# B&R Automation Studio project TD52 (part 147)

### Global_DI.typ
```iecst
TYPE
	Perm_DI_struct : 	STRUCT
		tCtr_ChCW_LT : _tGeACtrPara; (*Para controller charge temperature cooler*) (*OldName:REG9; Cycle:5;*)
		bCtr_ChCW_LT : BOOL; (*PARA [11872]: visibility charge temperature controller*) (*OldName:bPlantCtr9,reg0_visible; Cycle:5;*)
		tCtr_ChCW_HT : _tGeACtrPara; (*Para controller charge temperature cooler*) (*OldName:REG9; Cycle:5;*)
		bCtr_ChCW_HT : BOOL; (*PARA [11872]: visibility charge temperature controller*) (*OldName:bPlantCtr9,reg0_visible; Cycle:5;*)
		tCtr_ChCW_HT_LP : _tGeACtrPara; (*Para controller charge temperature cooler*) (*OldName:REG9; Cycle:5;*)
		bCtr_ChCW_HT_LP : BOOL; (*PARA [11872]: visibility charge temperature controller*) (*OldName:bPlantCtr9,reg0_visible; Cycle:5;*)
		tCtr_ChCW_HT_HP : _tGeACtrPara; (*Para controller charge temperature cooler*) (*OldName:REG9; Cycle:5;*)
		bCtr_ChCW_HT_HP : BOOL; (*PARA [11872]: visibility charge temperature controller*) (*OldName:bPlantCtr9,reg0_visible; Cycle:5;*)
		tCtr_ChCW_LT_LP : _tGeACtrPara; (*Para controller charge temperature cooler*) (*OldName:REG9; Cycle:5;*)
		bCtr_ChCW_LT_LP : BOOL; (*PARA [11872]: visibility charge temperature controller*) (*OldName:bPlantCtr9,reg0_visible; Cycle:5;*)
		tCtr_ChCW_LT_HP : _tGeACtrPara; (*Para controller charge temperature cooler*) (*OldName:REG9; Cycle:5;*)
		bCtr_ChCW_LT_HP : BOOL; (*PARA [11872]: visibility charge temperature controller*) (*OldName:bPlantCtr9,reg0_visible; Cycle:5;*)
		tCtr_ECW : _tGeACtrPara; (*Para controller  engine cooling water temperature cooler*) (*OldName:REG9; Cycle:5;*)
		bCtr_ECW : BOOL; (*PARA [11872]: visibility  engine cooling water temperature controller*) (*OldName:bPlantCtr9,reg0_visible; Cycle:5;*)
		tCtr_OCW : _tGeACtrPara; (*Para controller  oil cooling water temperature cooler*) (*OldName:REG9; Cycle:5;*)
		bCtr_OCW : BOOL; (*PARA [11872]: visibility  oil cooling water temperature controller*) (*OldName:bPlantCtr9,reg0_visible; Cycle:5;*)
		bT_ChCW_Re_LT : BOOL; (*visu aktiv Temp Ladekühlwasser Rücklauf NT*)
		bPr_ChCW_Re_LT : BOOL; (*visu aktiv Druck Ladekühlwasser Rücklauf NT*)
		bT_ChCW_Su_LT : BOOL; (*visu aktiv Temp Ladekühlwasser Vorlauf NT*)
		bPr_ChCW_Su_LT : BOOL; (*visu aktiv Druck Ladekühlwasser Vorlauf NT*)
		bT_ChCW_Re_HT : BOOL; (*visu aktiv Temp Ladekühlwasser Rücklauf NT*)
		bPr_ChCW_Re_HT : BOOL; (*visu aktiv Druck Ladekühlwasser Rücklauf HT*)
		bT_ChCW_Su_HT : BOOL; (*visu aktiv Temp Ladekühlwasser Vorlauf HT*)
		bPr_ChCW_Su_HT : BOOL; (*visu aktiv Druck Ladekühlwasser Vorlauf HT*)
		bT_ChCW_Re_HT_LP : BOOL; (*visu aktiv Temp Ladekühlwasser Rücklauf HT ND*)
		bPr_ChCW_Re_HT_LP : BOOL; (*visu aktiv Druck Ladekühlwasser Rücklauf HT ND*)
		bT_ChCW_Re_HT_HP : BOOL; (*visu aktiv Temp Ladekühlwasser Rücklauf HT HD*)
		bPr_ChCW_Re_HT_HP : BOOL; (*visu aktiv Druck Ladekühlwasser Rücklauf HT HD*)
		bT_ChCW_Su_HT_LP : BOOL; (*visu aktiv Temp Ladekühlwasser Vorlauf HT ND*)
		bPr_ChCW_Su_HT_LP : BOOL; (*visu aktiv Druck Ladekühlwasser Vorlauf HT ND*)
		bT_ChCW_Su_HT_HP : BOOL; (*visu aktiv Temp Ladekühlwasser Vorlauf HT HD*)
		bPr_ChCW_Su_HT_HP : BOOL; (*visu aktiv Druck Ladekühlwasser Vorlauf HT HD*)
		bT_ChCW_Re_LT_LP : BOOL; (*visu aktiv Temp Ladekühlwasser Rücklauf NT ND*)
		bPr_ChCW_Re_LT_LP : BOOL; (*visu aktiv Druck Ladekühlwasser Rücklauf NT ND*)
		bT_ChCW_Re_LT_HP : BOOL; (*visu aktiv Temp Ladekühlwasser Rücklauf NT HD*)
		bPr_ChCW_Re_LT_HP : BOOL; (*visu aktiv Druck Ladekühlwasser Rücklauf NT HD*)
		bT_ChCW_Su_LT_LP : BOOL; (*visu aktiv Temp Ladekühlwasser Vorlauf NT ND*)
		bPr_ChCW_Su_LT_LP : BOOL; (*visu aktiv Druck Ladekühlwasser Vorlauf NT ND*)
		bT_ChCW_Su_LT_HP : BOOL; (*visu aktiv Temp Ladekühlwasser Vorlauf NT HD*)
		bPr_ChCW_Su_LT_HP : BOOL; (*visu aktiv Druck Ladekühlwasser Vorlauf NT HD*)
		bT_OCW_Re : BOOL; (*visu aktiv Temp Ölkühlwasser Rücklauf*)
		bPr_OCW_Re : BOOL; (*visu aktiv Druck Ölkühlwasser Rücklauf*)
		bT_OCW_Su : BOOL; (*visu aktiv Temp Ölkühlwasser Vorlauf*)
		bPr_OCW_Su : BOOL; (*visu aktiv Druck Ölkühlwasser Vorlauf*)
		bT_ECW_Re : BOOL; (*visu aktiv Temp Motorkühlwasser Rücklauf*)
		bPr_ECW_Re : BOOL; (*visu aktiv Druck Motorkühlwasser Rücklauf*)
		bT_ECW_Su : BOOL; (*visu aktiv Temp Motorkühlwasser Vorlauf*)
		bPr_ECW_Su : BOOL; (*visu aktiv Druck Motorkühlwasser Vorlauf*)
		bVol_ChCW_Re_LT : BOOL; (*visu aktiv Durchfluss Ladekühlwasser Rücklauf NT*)
		bVol_ChCW_Su_LT : BOOL; (*visu aktiv Durchfluss Ladekühlwasser Vorlauf NT*)
		bVol_ChCW_Re_HT : BOOL; (*visu aktiv Durchfluss Ladekühlwasser Rücklauf HT*)
		bVol_ChCW_Su_HT : BOOL; (*visu aktiv Durchfluss Ladekühlwasser Vorlauf HT*)
		bVol_ChCW_Re_HT_LP : BOOL; (*visu aktiv Durchfluss Ladekühlwasser Rücklauf HT ND*)
		bVol_ChCW_Su_HT_LP : BOOL; (*visu aktiv Durchfluss Ladekühlwasser Vorlauf HT ND*)
		bVol_ChCW_Re_HT_HP : BOOL; (*visu aktiv Durchfluss Ladekühlwasser Rücklauf HT HD*)
		bVol_ChCW_Su_HT_HP : BOOL; (*visu aktiv Durchfluss Ladekühlwasser Vorlauf HT HD*)
		bVol_ChCW_Re_LT_LP : BOOL; (*visu aktiv Durchfluss Ladekühlwasser Rücklauf NT ND*)
		bVol_ChCW_Su_LT_LP : BOOL; (*visu aktiv Durchfluss Ladekühlwasser Vorlauf NT ND*)
		bVol_ChCW_Re_LT_HP : BOOL; (*visu aktiv Durchfluss Ladekühlwasser Rücklauf NT HD*)
		bVol_ChCW_Su_LT_HP : BOOL; (*visu aktiv Durchfluss Ladekühlwasser Vorlauf NT HD*)
		bVol_ECW_Re : BOOL; (*visu aktiv Durchfluss Motorkühlwasser Rücklauf*)
		bVol_ECW_Su : BOOL; (*visu aktiv Durchfluss Motorkühlwasser Vorlauf*)
		bVol_OCW_Re : BOOL; (*visu aktiv Durchfluss Ölkühlwasser Rücklauf*)
		bVol_OCW_Su : BOOL; (*visu aktiv Durchfluss Ölkühlwasser Vorlauf*)
		bT_ChCW_LT_IC_Re : BOOL; (*visu aktiv Temp Ladekühlewasser NT Zwischenkreis Rücklauf*)
		bPr_ChCW_LT_IC_Re : BOOL; (*visu aktiv Druck Ladekühlewasser NT Zwischenkreis Rücklauf*)
		bT_ChCW_HT_IC_Re : BOOL; (*visu aktiv Temp Ladekühlewasser HT Zwischenkreis Rücklauf*)
		bPr_ChCW_HT_IC_Re : BOOL; (*visu aktiv Druck Ladekühlewasser HT Zwischenkreis Rücklauf*)
		bT_ChCW_LT_LP_IC_Re : BOOL; (*visu aktiv Temp Ladekühlewasser NT ND Zwischenkreis Rücklauf*)
		bPr_ChCW_LT_LP_IC_Re : BOOL; (*visu aktiv Druck Ladekühlewasser NT ND Zwischenkreis Rücklauf*)
		bT_ChCW_LT_HP_IC_Re : BOOL; (*visu aktiv Temp Ladekühlewasser NT HD Zwischenkreis Rücklauf*)
		bPr_ChCW_LT_HP_IC_Re : BOOL; (*visu aktiv Druck Ladekühlewasser NT HD Zwischenkreis Rücklauf*)
		bT_ChCW_HT_LP_IC_Re : BOOL; (*visu aktiv Temp Ladekühlewasser HT ND Zwischenkreis Rücklauf*)
		bPr_ChCW_HT_LP_IC_Re : BOOL; (*visu aktiv Druck Ladekühlewasser HT ND Zwischenkreis Rücklauf*)
		bT_ChCW_HT_HP_IC_Re : BOOL; (*visu aktiv Temp Ladekühlewasser HT HD Zwischenkreis Rücklauf*)
		bPr_ChCW_HT_HP_IC_Re : BOOL; (*visu aktiv Druck Ladekühlewasser HT HD Zwischenkreis Rücklauf*)
		bT_ECW_IC_Re : BOOL; (*visu aktiv Temp Motorkühlwasser Zwischenkreis Rücklauf*)
		bPr_ECW_IC_Re : BOOL; (*visu aktiv Druck Motorkühlwasser Zwischenkreis Rücklauf*)
		bT_OCW_IC_Re : BOOL; (*visu aktiv Temp Ölkühlwasser Zwischenkreis Rücklauf*)
		bPr_OCW_IC_Re : BOOL; (*visu aktiv Druck Ölkühlwasser Zwischenkreis Rücklauf*)
		bT_ChCW_LT_IC_Su : BOOL; (*visu aktiv Temp Ladekühlewasser NT Zwischenkreis Rücklauf*)
		bPr_ChCW_LT_IC_Su : BOOL; (*visu aktiv Druck Ladekühlewasser NT Zwischenkreis Rücklauf*)
		bT_ChCW_HT_IC_Su : BOOL; (*visu aktiv Temp Ladekühlewasser HT Zwischenkreis Rücklauf*)
		bPr_ChCW_HT_IC_Su : BOOL; (*visu aktiv Druck Ladekühlewasser HT Zwischenkreis Rücklauf*)
		bT_ChCW_LT_LP_IC_Su : BOOL; (*visu aktiv Temp Ladekühlewasser NT ND Zwischenkreis Rücklauf*)
		bPr_ChCW_LT_LP_IC_Su : BOOL; (*visu aktiv Druck Ladekühlewasser NT ND Zwischenkreis Rücklauf*)
		bT_ChCW_LT_HP_IC_Su : BOOL; (*visu aktiv Temp Ladekühlewasser NT HD Zwischenkreis Rücklauf*)
		bPr_ChCW_LT_HP_IC_Su : BOOL; (*visu aktiv Druck Ladekühlewasser NT HD Zwischenkreis Rücklauf*)
		bT_ChCW_HT_LP_IC_Su : BOOL; (*visu aktiv Temp Ladekühlewasser HT ND Zwischenkreis Rücklauf*)
		bPr_ChCW_HT_LP_IC_Su : BOOL; (*visu aktiv Druck Ladekühlewasser HT ND Zwischenkreis Rücklauf*)
		bT_ChCW_HT_HP_IC_Su : BOOL; (*visu aktiv Temp Ladekühlewasser HT HD Zwischenkreis Rücklauf*)
		bPr_ChCW_HT_HP_IC_Su : BOOL; (*visu aktiv Druck Ladekühlewasser HT HD Zwischenkreis Rücklauf*)
		bT_ECW_IC_Su : BOOL; (*visu aktiv Temp Motorkühlwasser Zwischenkreis Rücklauf*)
		bPr_ECW_IC_Su : BOOL; (*visu aktiv Druck Motorkühlwasser Zwischenkreis Rücklauf*)
		bT_OCW_IC_Su : BOOL; (*visu aktiv Temp Ölkühlwasser Zwischenkreis Rücklauf*)
		bPr_OCW_IC_Su : BOOL; (*visu aktiv Druck Ölkühlwasser Zwischenkreis Vorlauf*)
		bT_Cooler_ChCW_LT_Re_1 : BOOL; (*visu aktiv Temp Kühler Ladekühlwasser NT Rücklauf*)
		bT_Cooler_ChCW_LT_Re_2 : BOOL; (*visu aktiv Temp Kühler Ladekühlwasser NT Rücklauf*)
		bT_Cooler_ChCW_HT_Re_1 : BOOL; (*visu aktiv Temp Kühler Ladekühlwasser HT Rücklauf*)
		bT_Cooler_ChCW_HT_Re_2 : BOOL; (*visu aktiv Temp Kühler Ladekühlwasser HT Rücklauf*)
		bT_Cooler_ChCW_LT_LP_Re_1 : BOOL; (*visu aktiv Temp Kühler Ladekühlwasser NT ND Rücklauf*)
		bT_Cooler_ChCW_LT_LP_Re_2 : BOOL; (*visu aktiv Temp Kühler Ladekühlwasser NT ND Rücklauf*)
		bT_Cooler_ChCW_LT_HP_Re_1 : BOOL; (*visu aktiv Temp Kühler Ladekühlwasser NT HD Rücklauf*)
		bT_Cooler_ChCW_LT_HP_Re_2 : BOOL; (*visu aktiv Temp Kühler Ladekühlwasser NT HD Rücklauf*)
		bT_Cooler_ChCW_HT_LP_Re_1 : BOOL; (*visu aktiv Temp Kühler Ladekühlwasser HT ND Rücklauf*)
		bT_Cooler_ChCW_HT_LP_Re_2 : BOOL; (*visu aktiv Temp Kühler Ladekühlwasser HT ND Rücklauf*)
		bT_Cooler_ChCW_HT_HP_Re_1 : BOOL; (*visu aktiv Temp Kühler Ladekühlwasser HT HD Rücklauf*)
		bT_Cooler_ChCW_HT_HP_Re_2 : BOOL; (*visu aktiv Temp Kühler Ladekühlwasser HT HD Rücklauf*)
		bT_Cooler_ECW_Re_1 : BOOL; (*visu aktiv Temp Kühler Motorkühlwasser Rücklauf*)
		bT_Cooler_ECW_Re_2 : BOOL; (*visu aktiv Temp Kühler Motorkühlwasser Rücklauf*)
		bT_Cooler_OCW_Re_1 : BOOL; (*visu aktiv Temp Kühler Ölkühlwasser Rücklauf*)
		bT_Cooler_OCW_Re_2 : BOOL; (*visu aktiv Temp Kühler Ölkühlwasser Rücklauf*)
		bPr_Cooler_ChCW_LT_Re_1 : BOOL; (*visu aktiv Druck Kühler Ladekühlwasser NT Rücklauf*)
		bPr_Cooler_ChCW_LT_Re_2 : BOOL; (*visu aktiv Druck Kühler Ladekühlwasser NT Rücklauf*)
		bPr_Cooler_ChCW_HT_Re_1 : BOOL; (*visu aktiv Druck Kühler Ladekühlwasser HT Rücklauf*)
		bPr_Cooler_ChCW_HT_Re_2 : BOOL; (*visu aktiv Druck Kühler Ladekühlwasser HT Rücklauf*)
		bPr_Cooler_ChCW_LT_LP_Re_1 : BOOL; (*visu aktiv Druck Kühler Ladekühlwasser NT ND Rücklauf*)
		bPr_Cooler_ChCW_LT_LP_Re_2 : BOOL; (*visu aktiv Druck Kühler Ladekühlwasser NT ND Rücklauf*)
		bPr_Cooler_ChCW_LT_HP_Re_1 : BOOL; (*visu aktiv Druck Kühler Ladekühlwasser NT HD Rücklauf*)
		bPr_Cooler_ChCW_LT_HP_Re_2 : BOOL; (*visu aktiv Druck Kühler Ladekühlwasser NT HD Rücklauf*)
		bPr_Cooler_ChCW_HT_LP_Re_1 : BOOL; (*visu aktiv Druck Kühler Ladekühlwasser HT ND Rücklauf*)
		bPr_Cooler_ChCW_HT_LP_Re_2 : BOOL; (*visu aktiv Druck Kühler Ladekühlwasser HT ND Rücklauf*)
		bPr_Cooler_ChCW_HT_HP_Re_1 : BOOL; (*visu aktiv Druck Kühler Ladekühlwasser HT HD Rücklauf*)
		bPr_Cooler_ChCW_HT_HP_Re_2 : BOOL; (*visu aktiv Druck Kühler Ladekühlwasser HT HD Rücklauf*)
		bPr_Cooler_ECW_Re_1 : BOOL; (*visu aktiv Druck Kühler Motorkühlwasser Rücklauf*)
		bPr_Cooler_ECW_Re_2 : BOOL; (*visu aktiv Druck Kühler Motorkühlwasser Rücklauf*)
		bPr_Cooler_OCW_Re_1 : BOOL; (*visu aktiv Druck Kühler Ölkühlwasser Rücklauf*)
		bPr_Cooler_OCW_Re_2 : BOOL; (*visu aktiv Druck Kühler Ölkühlwasser Rücklauf*)
		bT_Cooler_ChCW_LT_Su_1 : BOOL; (*visu aktiv Temp Kühler Ladekühlwasser NT Vorlauf*)
		bT_Cooler_ChCW_LT_Su_2 : BOOL; (*visu aktiv Temp Kühler Ladekühlwasser NT Vorlauf*)
		bT_Cooler_ChCW_HT_Su_1 : BOOL; (*visu aktiv Temp Kühler Ladekühlwasser HT Vorlauf*)
		bT_Cooler_ChCW_HT_Su_2 : BOOL; (*visu aktiv Temp Kühler Ladekühlwasser HT Vorlauf*)
		bT_Cooler_ChCW_LT_LP_Su_1 : BOOL; (*visu aktiv Temp Kühler Ladekühlwasser NT ND Vorlauf*)
		bT_Cooler_ChCW_LT_LP_Su_2 : BOOL; (*visu aktiv Temp Kühler Ladekühlwasser NT ND Vorlauf*)
		bT_Cooler_ChCW_LT_HP_Su_1 : BOOL; (*visu aktiv Temp Kühler Ladekühlwasser NT HD Vorlauf*)
		bT_Cooler_ChCW_LT_HP_Su_2 : BOOL; (*visu aktiv Temp Kühler Ladekühlwasser NT HD Vorlauf*)
		bT_Cooler_ChCW_HT_LP_Su_1 : BOOL; (*visu aktiv Temp Kühler Ladekühlwasser HT ND Vorlauf*)
		bT_Cooler_ChCW_HT_LP_Su_2 : BOOL; (*visu aktiv Temp Kühler Ladekühlwasser HT ND Vorlauf*)
		bT_Cooler_ChCW_HT_HP_Su_1 : BOOL; (*visu aktiv Temp Kühler Ladekühlwasser HT HD Vorlauf*)
		bT_Cooler_ChCW_HT_HP_Su_2 : BOOL; (*visu aktiv Temp Kühler Ladekühlwasser HT HD Vorlauf*)
		bT_Cooler_ECW_Su_1 : BOOL; (*visu aktiv Temp Kühler Motorkühlwasser Vorlauf*)
		bT_Cooler_ECW_Su_2 : BOOL; (*visu aktiv Temp Kühler Motorkühlwasser Vorlauf*)
		bT_Cooler_OCW_Su_1 : BOOL; (*visu aktiv Temp Kühler Ölkühlwasser Vorlauf*)
		bT_Cooler_OCW_Su_2 : BOOL; (*visu aktiv Temp Kühler Ölkühlwasser Vorlauf*)
		bPr_Cooler_ChCW_LT_Su_1 : BOOL; (*visu aktiv Druck Kühler Ladekühlwasser NT Vorlauf*)
		bPr_Cooler_ChCW_LT_Su_2 : BOOL; (*visu aktiv Druck Kühler Ladekühlwasser NT Vorlauf*)
		bPr_Cooler_ChCW_HT_Su_1 : BOOL; (*visu aktiv Druck Kühler Ladekühlwasser HT Vorlauf*)
		bPr_Cooler_ChCW_HT_Su_2 : BOOL; (*visu aktiv Druck Kühler Ladekühlwasser HT Vorlauf*)
		bPr_Cooler_ChCW_LT_LP_Su_1 : BOOL; (*visu aktiv Druck Kühler Ladekühlwasser NT ND Vorlauf*)
		bPr_Cooler_ChCW_LT_LP_Su_2 : BOOL; (*visu aktiv Druck Kühler Ladekühlwasser NT ND Vorlauf*)
		bPr_Cooler_ChCW_LT_HP_Su_1 : BOOL; (*visu aktiv Druck Kühler Ladekühlwasser NT HD Vorlauf*)
		bPr_Cooler_ChCW_LT_HP_Su_2 : BOOL; (*visu aktiv Druck Kühler Ladekühlwasser NT HD Vorlauf*)
		bPr_Cooler_ChCW_HT_LP_Su_1 : BOOL; (*visu aktiv Druck Kühler Ladekühlwasser HT ND Vorlauf*)
		bPr_Cooler_ChCW_HT_LP_Su_2 : BOOL; (*visu aktiv Druck Kühler Ladekühlwasser HT ND Vorlauf*)
		bPr_Cooler_ChCW_HT_HP_Su_1 : BOOL; (*visu aktiv Druck Kühler Ladekühlwasser HT HD Vorlauf*)
		bPr_Cooler_ChCW_HT_HP_Su_2 : BOOL; (*visu aktiv Druck Kühler Ladekühlwasser HT HD Vorlauf*)
		bPr_Cooler_ECW_Su_1 : BOOL; (*visu aktiv Druck Kühler Motorkühlwasser Vorlauf*)
		bPr_Cooler_ECW_Su_2 : BOOL; (*visu aktiv Druck Kühler Motorkühlwasser Vorlauf*)
		bPr_Cooler_OCW_Su_1 : BOOL; (*visu aktiv Druck Kühler Ölkühlwasser Vorlauf*)
		bPr_Cooler_OCW_Su_2 : BOOL; (*visu aktiv Druck Kühler Ölkühlwasser Vorlauf*)
		bT_ChCW_LT_bCV : BOOL; (*visu aktiv Temp Ladekühlwasser NT vor Regelventil*)
		bT_ChCW_LT_LP_bCV : BOOL; (*visu aktiv Temp Ladekühlwasser NT ND vor Regelventil*)
		bT_ChCW_LT_HP_bCV : BOOL; (*visu aktiv Temp Ladekühlwasser NT HD vor Regelventil*)
		bT_ChCW_HT_bCV : BOOL; (*visu aktiv Temp Ladekühlwasser NT vor Regelventil*)
		bT_ChCW_HT_LP_bCV : BOOL; (*visu aktiv Temp Ladekühlwasser NT ND vor Regelventil*)
		bT_ChCW_HT_HP_bCV : BOOL; (*visu aktiv Temp Ladekühlwasser NT HD vor Regelventil*)
		bT_ECW_bCV : BOOL; (*visu aktiv Temp Motorkühlwasser vor Regelventil*)
		bT_OCW_bCV : BOOL; (*visu aktiv Temp Ölkühlwasser vor Regelventil*)
		bT_RW_HE_Re : BOOL; (*visu aktiv Temp Rohwasser Wärmetausche Rücklauf*)
		bT_RW_HE_Su : BOOL; (*visu aktiv Temp Rohwasser Wärmetausche Vorlauf*)
		bPr_RW_HE_Re : BOOL; (*visu aktiv Druck Rohwasser Wärmetausche Rücklauf*)
		bPr_RW_HE_Su : BOOL; (*visu aktiv Druck Rohwasser Wärmetausche Vorlauf*)
		bCtr_RW_CV : BOOL; (*visu aktiv Regler Rohwasser Regelventil*)
		bCtr_RW_HE : BOOL; (*visu aktiv Regler Rohwasser Wärmetausche*)
		bFC_ChCW_LT_Pump : BOOL; (*visu aktiv FU Ladekühlewasser NT*)
		bFC_ChCW_HT_Pump : BOOL; (*visu aktiv FU Ladekühlewasser HT*)
		bFC_ChCW_LT_LP_Pump : BOOL; (*visu aktiv FU Ladekühlewasser NT ND*)
		bFC_ChCW_LT_HP_Pump : BOOL; (*visu aktiv FU Ladekühlewasser NT HD*)
		bFC_ChCW_HT_LP_Pump : BOOL; (*visu aktiv FU Ladekühlewasser HT ND*)
		bFC_ChCW_HT_HP_Pump : BOOL; (*visu aktiv FU Ladekühlewasser HT HD*)
		bFC_ECW_Pump : BOOL; (*visu aktiv FU Motorkühlwasser*)
		bFC_OCW_Pump : BOOL; (*visu aktiv FU Ölkühlwasser*)
		bFC_ChCW_LT_Cooler_1 : BOOL; (*visu aktiv FU Ladekühlwasser NT Kühler*)
		bFC_ChCW_LT_Cooler_2 : BOOL; (*visu aktiv FU Ladekühlwasser NT Kühler*)
		bFC_ChCW_HT_Cooler_1 : BOOL; (*visu aktiv FU Ladekühlwasser HT Kühler*)
		bFC_ChCW_HT_Cooler_2 : BOOL; (*visu aktiv FU Ladekühlwasser HT Kühler*)
		bFC_ChCW_LT_LP_Cooler_1 : BOOL; (*visu aktiv FU Ladekühlwasser NT ND Kühler*)
		bFC_ChCW_LT_LP_Cooler_2 : BOOL; (*visu aktiv FU Ladekühlwasser NT ND Kühler*)
		bFC_ChCW_LT_HP_Cooler_1 : BOOL; (*visu aktiv FU Ladekühlwasser NT HD Kühler*)
		bFC_ChCW_LT_HP_Cooler_2 : BOOL; (*visu aktiv FU Ladekühlwasser NT HD Kühler*)
		bFC_ChCW_HT_LP_Cooler_1 : BOOL; (*visu aktiv FU Ladekühlwasser HT ND Kühler*)
		bFC_ChCW_HT_LP_Cooler_2 : BOOL; (*visu aktiv FU Ladekühlwasser HT ND Kühler*)
		bFC_ChCW_HT_HP_Cooler_1 : BOOL; (*visu aktiv FU Ladekühlwasser HT HD Kühler*)
		bFC_ChCW_HT_HP_Cooler_2 : BOOL; (*visu aktiv FU Ladekühlwasser HT HD Kühler*)
		bFC_ECW_Cooler_1 : BOOL; (*visu aktiv FU Motorkühlwasser Kühler*)
		bFC_ECW_Cooler_2 : BOOL; (*visu aktiv FU Motorkühlwasser Kühler*)
		bFC_OCW_Cooler_1 : BOOL; (*visu aktiv FU Ölkühlwasser Kühler*)
		bFC_OCW_Cooler_2 : BOOL; (*visu aktiv FU Ölkühlwasser Kühler*)
		bPs_ChCW_LT_bEngine_Hi : BOOL; (*visu aktiv Druckschalter Ladekühlewasser NT vor Motor max*)
		bPs_ChCW_HT_bEngine_Hi : BOOL; (*visu aktiv Druckschalter Ladekühlewasser HT vor Motor max*)
		bPs_ChCW_LT_LP_bEngine_Hi : BOOL; (*visu aktiv Druckschalter Ladekühlewasser NT ND vor Motor max*)
		bPs_ChCW_LT_HP_bEngine_Hi : BOOL; (*visu aktiv Druckschalter Ladekühlewasser NT HD vor Motor max*)
		bPs_ChCW_HT_LP_bEngine_Hi : BOOL; (*visu aktiv Druckschalter Ladekühlewasser HT ND vor Motor max*)
		bPs_ChCW_HT_HP_bEngine_Hi : BOOL; (*visu aktiv Druckschalter Ladekühlewasser HT HD vor Motor max*)
		bPs_ECW_bEngine_Hi : BOOL; (*visu aktiv Druckschalter Motorkühlwasser vor Motor max*)
		bPs_OCW_bEngine_Hi : BOOL; (*visu aktiv Druckschalter Ölkühlwasser vor Motor max*)
		bPs_ChCW_LT_bPump_Low : BOOL; (*visu aktiv Druckschalter Ladekühlewasser NT vor Pumpe min*)
		bPs_ChCW_HT_bPump_Low : BOOL; (*visu aktiv Druckschalter Ladekühlewasser HT vor Pumpe min*)
		bPs_ChCW_LT_LP_bPump_Low : BOOL; (*visu aktiv Druckschalter Ladekühlewasser NT ND vor Pumpe min*)
		bPs_ChCW_LT_HP_bPump_Low : BOOL; (*visu aktiv Druckschalter Ladekühlewasser NT HD vor Pumpe min*)
		bPs_ChCW_HT_LP_bPump_Low : BOOL; (*visu aktiv Druckschalter Ladekühlewasser HT ND vor Pumpe min*)
		bPs_ChCW_HT_HP_bPump_Low : BOOL; (*visu aktiv Druckschalter Ladekühlewasser HT HD vor Pumpe min*)
		bPs_ECW_bPump_Low : BOOL; (*visu aktiv Druckschalter Motorkühlwasser vor Pumpe min*)
		bPs_OCW_bPump_Low : BOOL; (*visu aktiv Druckschalter Ölkühlwasser vor Pumpe min*)
		bTs_ChCW_LT_bEngine_Hi : BOOL; (*visu aktiv Temperaturschalter Ladekühlewasser NT vor Motor max*)
		bTs_ChCW_HT_bEngine_Hi : BOOL; (*visu aktiv Temperaturschalter Ladekühlewasser HT vor Motor max*)
		bTs_ChCW_LT_LP_bEngine_Hi : BOOL; (*visu aktiv Temperaturschalter Ladekühlewasser NT ND vor Motor max*)
		bTs_ChCW_LT_HP_bEngine_Hi : BOOL; (*visu aktiv Temperaturschalter Ladekühlewasser NT HD vor Motor max*)
		bTs_ChCW_HT_LP_bEngine_Hi : BOOL; (*visu aktiv Temperaturschalter Ladekühlewasser HT ND vor Motor max*)
		bTs_ChCW_HT_HP_bEngine_Hi : BOOL; (*visu aktiv Temperaturschalter Ladekühlewasser HT HD vor Motor max*)
		bTs_ECW_bEngine_Hi : BOOL; (*visu aktiv Temperaturschalter Motorkühlwasser vor Motor max*)
		bTs_OCW_bEngine_Hi : BOOL; (*visu aktiv Temperaturschalter Ölkühlwasser vor Motor max*)
		bDem_Cooler_ChCW_LT_1 : BOOL; (*visu aktiv Anforderung Kühler Ladekühlwasser NT*)
		bDem_Cooler_ChCW_LT_2 : BOOL; (*visu aktiv Anforderung Kühler Ladekühlwasser NT*)
		bDem_Cooler_ChCW_HT_1 : BOOL; (*visu aktiv Anforderung Kühler Ladekühlwasser HT*)
		bDem_Cooler_ChCW_HT_2 : BOOL; (*visu aktiv Anforderung Kühler Ladekühlwasser HT*)
		bDem_Cooler_ChCW_LT_LP_1 : BOOL; (*visu aktiv Anforderung Kühler Ladekühlwasser NT ND*)
		bDem_Cooler_ChCW_LT_LP_2 : BOOL; (*visu aktiv Anforderung Kühler Ladekühlwasser NT ND*)
		bDem_Cooler_ChCW_LT_HP_1 : BOOL; (*visu aktiv Anforderung Kühler Ladekühlwasser NT HD*)
		bDem_Cooler_ChCW_LT_HP_2 : BOOL; (*visu aktiv Anforderung Kühler Ladekühlwasser NT HD*)
		bDem_Cooler_ChCW_HT_LP_1 : BOOL; (*visu aktiv Anforderung Kühler Ladekühlwasser HT ND*)
		bDem_Cooler_ChCW_HT_LP_2 : BOOL; (*visu aktiv Anforderung Kühler Ladekühlwasser HT ND*)
		bDem_Cooler_ChCW_HT_HP_1 : BOOL; (*visu aktiv Anforderung Kühler Ladekühlwasser HT HD*)
		bDem_Cooler_ChCW_HT_HP_2 : BOOL; (*visu aktiv Anforderung Kühler Ladekühlwasser HT HD*)
		bDem_Cooler_ECW_1 : BOOL; (*visu aktiv Anforderung Kühler Motorkühlwasser*)
		bDem_Cooler_ECW_2 : BOOL; (*visu aktiv Anforderung Kühler Motorkühlwasser*)
		bDem_Cooler_OCW_1 : BOOL; (*visu aktiv Anforderung Kühler Ölkühlwasser*)
		bDem_Cooler_OCW_2 : BOOL; (*visu aktiv Anforderung Kühler Ölkühlwasser*)
		bDem_ChCW_LT_Pump : BOOL; (*visu aktiv Anforderung Ladekühlewasser NT Pumpe*)
		bDem_ChCW_HT_Pump : BOOL; (*visu aktiv Anforderung Ladekühlewasser HT Pumpe*)
		bDem_ChCW_LT_LP_Pump : BOOL; (*visu aktiv Anforderung Ladekühlewasser NT ND Pumpe*)
		bDem_ChCW_LT_HP_Pump : BOOL; (*visu aktiv Anforderung Ladekühlewasser NT HD Pumpe*)
		bDem_ChCW_HT_LP_Pump : BOOL; (*visu aktiv Anforderung Ladekühlewasser HT ND Pumpe*)
		bDem_ChCW_HT_HP_Pump : BOOL; (*visu aktiv Anforderung Ladekühlewasser HT HD Pumpe*)
		bDem_ECW_Pump : BOOL; (*visu aktiv Anforderung Motorkühlwasser Pumpe*)
		bDem_OCW_Pump : BOOL; (*visu aktiv Anforderung Ölkühlwasser Pumpe*)
		rT_CtrER_WexRun : REAL; (*engine room temperature controller external setpoint run*)
		rT_ACP_AirER_sp : REAL; (*Active cooling program setpoint temperature engine room ventilation*)
		rT_CtrER_WexStop : REAL; (*engine room temperature controller external setpoint stop*)
		bT_AirER1_Active : BOOL; (*Raumtemperatur 1 aktiv*)
		bT_AirER2_Active : BOOL; (*Raumtemperatur 2 aktiv*)
		bT_AirER3_Active : BOOL; (*Raumtemperatur 3 aktiv*)
		bT_AirER4_Active : BOOL; (*Raumtemperatur 4 aktiv*)
		bT_AirOutdoor_Active : BOOL; (*PARA [11885]: air outdoor temperature measurement enable *) (*OldName:ULT_a; Cycle:5;*)
		bIntakeAirCond : BOOL; (*Zuluftkonditionierung Aktiv*)
		bPrDiff_ER_Active : BOOL; (*Messung Raumdiffernzdruck aktiv*)
		bCtr_ER : BOOL; (*Raumlufttemperaturregler aktiv*)
		bCtr_OutlVE_RDP : BOOL; (*air outlet ventilation controller for room differential pressure enable*)
		tCtr_IntakeAir : _tGeACtrPara; (*Para Regler für Motor Ansaugluft*)
		tCtr_ER : _tGeACtrPara; (*Para controller engine room temperature*)
		tCtr_OutlVE_RDP : _tGeACtrPara; (*Para controller air outlet ventilation (for engine room differential pressure)*)
		tCtr_EG_Flap : _tGeACtrPara; (*Para Abgasklappenregler*)
		rLSCS_MV_Set : REAL; (*Vorgabe LSCS Mischventil*)
		rLSCS_GV_Set : REAL; (*Vorgabe LSCS Gasventil*)
		rSel_LSCS_MV : REAL; (*Vorgabe Koeffizient der Blende vom Mischventil*)
		rSel_LSCS_GV : REAL; (*Vorgabe Koeffizient der Blende vom Gasventil*)
		tCtr_GC_1 : _tGeACtrPara; (*Para Gaskompressorregler 1*)
		tCtr_GC_2 : _tGeACtrPara; (*Para Gaskompressorregler 2*)
		tCtr_MN_MG : _tGeACtrPara; (*Para Gas mischen regler*)
		bSG_active : BOOL; (*Sondergasstrecke aktiv*)
		tPreHeatWDay : ARRAY[0..7]OF PreHeatWDay; (*Variablen für die Zeitsteuerung für Vorwärmung*)
		bPreHeatWDay_CtrActive : BOOL; (*Allgemeine Aktivierung der Zeitsteurerung*)
		bLSCS_GV_active : BOOL; (*LSCS Gasventil aktiv*)
		bLSCS_MV_active : BOOL; (*LSCS Mischventil aktiv*)
		iSel_Cooling : INT; (*Auswahl Srt der Kühlung*)
		bGasCompActive : BOOL; (*Zähler Gascompressor aktiv*)
		bGasCntSensycalActive : BOOL; (*Gaszähler Sensycal aktiv*)
		bGasCntCalcActive : BOOL; (*Gaszähler berechnet aktiv*)
		rCnt_CompOpHoursW : REAL; (* compressor operating hours counter until warning *)
		bH2_Mode : BOOL; (* Gasstrecke 3, TRUE = H2 aktiv *)
		bGasFlowCtr : BOOL; (* Gas flow control via engine controller setpoints for transient mixgas*)
		bSG_MFC_Used : BOOL; (* Special gas MFC used *)
		bPG_MFC_Used : BOOL; (* propan gas MFC used *)
		bBatCtrActive : BOOL; (* Batterieüberwachung wird visualisiert *)
		bIncl_SG_Calc : BOOL; (*Include special gas for MN & CV calculation*)
		bSend_Cv2Eng : BOOL; (*Send calculated CV  to  engine*)
		iNumInlLou : INT; (*Number of Louvers*)
		iNumInlLouRoom : INT; (*Number of Louvers*)
		iNumOutlLou : INT; (*Number of Louvers*)
		iNumCircLou : INT; (*Number of Louvers*)
		iNumInlLouEng : INT; (*Number of Louvers*)
		iNumCircLouEng : INT; (*Number of Louvers*)
		iVisRoomLou : INT; (*indication of room ventilation*)
		bPr_EG_DeflagActive : BOOL; (*Abgasdruck auf Visu aktiv*)
		bEG_SRC_DPF_Active : BOOL; (*Abgasseite für SCR und DPF auf Visu aktiv*)
		rLevel_Oiltank_ScalY1 : REAL; (*Öltankstand min Skalierung*)
		rLevel_Oiltank_ScalY2 : REAL; (*Öltankstand max Skalierung*)
		bAirCondHeaterActive : BOOL; (*Zuluftkonditionierung Heizung aktiv*)
		bTs_bEngineHiActive : BOOL; (*Temperaturschalter Max vor Motor bei Wärmetauscher aktiv (gilt für alle Kühlkreise)*)
		bPs_bEngineHiActive : BOOL; (*Druckschalter Max vor Motor bei Wärmetauscher aktiv (gilt für alle Kühlkreise)*)
		bT_bCV_Active : BOOL; (*Temperatur vor Temperaturregelventil aktiv (gilt für alle Kühlkreise)*)
		bT_Cooler_Re_Active : BOOL; (*Temperatur Rücklauf beim Kühler aktiv (gilt für alle Kühlkreise)*)
		bT_Cooler_Su_Active : BOOL; (*Temperatur Vorlauf beim Kühler aktiv (gilt für alle Kühlkreise)*)
		bPr_Cooler_Re_Active : BOOL; (*Druck Rücklauf beim Kühler aktiv (gilt für alle Kühlkreise)*)
		bPr_Cooler_Su_Active : BOOL; (*Druck Vorlauf beim Kühler aktiv (gilt für alle Kühlkreise)*)
		bExtCtrNOX_Active : BOOL; (*Externe NOX Regelung aktiv*)
		bPs_RW_Active : BOOL; (*Druckschalter Rohwasser Sammelleitung aktiv*)
		bTs_RW_Active : BOOL; (*Temperaturschalter Rohwasser Sammelleitung aktiv*)
		bT_RW_Re_Active : BOOL; (*Temperatur Rohwasser Rücklauf Sammelleitung aktiv*)
		bT_RW_Su_Active : BOOL; (*Temperatur Rohwasser Vorlauf Sammelleitung aktiv*)
		bFB_CC_Active : BOOL; (*Rückmeldung Kühlkreis Regelventile aktiv*)
		bFB_Cooler_Active : BOOL; (*Rückmeldung Kühler aktiv*)
		bFB_AC_Heating_Active : BOOL; (*Rückmeldung Zuluftkonditionierung Heizkreisregelventil aktiv*)
		bFB_AC_Cooling_Active : BOOL; (*Rückmeldung Zuluftkonditionierung Kühlkreisregelventil aktiv*)
		bT_HW_Air_Re_Active : BOOL; (*Zuluftkonditionierung Heizkreitemp. Rücklauf aktiv*)
		bT_HW_Air_Su_Active : BOOL; (*Zuluftkonditionierung Heizkreitemp. Vorlauf aktiv*)
		bCtr_ChCW_LT_Eng : BOOL; (*Regler regelt mit der Temperatur vom Motor*)
		bCtr_ECW_Eng : BOOL; (*Regler regelt mit der Temperatur vom Motor*)
		bCtr_OCW_Eng : BOOL; (*Regler regelt mit der Temperatur vom Motor*)
		bPr_EG_DeflagFastActive : BOOL; (*Visu Abgasdruck schnell aktiv*)
		bPs_aEngineLowActive : BOOL; (*visu aktiv Druckschalter nach Motor min*)
		bPs_bPumpLowActive : BOOL; (*visu aktiv Druckschalter vor Pumpe min*)
		bCircLouActive : BOOL; (*visu aktiv Umluftjalousie im Motorraum*)
		bCircLouEngActive : BOOL; (*visu aktiv Umluftjalousie von Zuluftkonditionierung*)
		bChC_LT_Stages_Active : BOOL; (*Ladekühlerstufen NT Schaltstufen aktiv*)
		rChC_LT_Stages_MaxNum : REAL; (*Anzahl Ladekühlerstufen NT gesamt*)
		bChC_HT_Stages_Active : BOOL; (*Ladekühlerstufen HT Schaltstufen aktiv*)
		rChC_HT_Stages_MaxNum : REAL; (*Anzahl Ladekühlerstufen HT gesamt*)
		bECW_Stages_Active : BOOL; (*Motorkühlwasserstufen Schaltstufen aktiv*)
		rECW_Stages_MaxNum : REAL; (*Anzahl Motorkühlwasserstufen gesamt*)
		bOCW_Stages_Active : BOOL; (*Ölkühlwasserstufen Schaltstufen aktiv*)
		rOCW_Stages_MaxNum : REAL; (*Anzahl Ölkühlwasserstufen gesamt*)
		bT_AirER5_Active : BOOL; (*Raumtemperatur 5 aktiv*)
		bT_AirER6_Active : BOOL; (*Raumtemperatur 6 aktiv*)
		bEG_Flap2_Active : BOOL; (*2. Abgasgegendruckklappe aktiv*)
		bT_EG_PrReliefVa_Active : BOOL; (*Temperatur Abgas Auslassventil aktiv*)
		bFreshAirEngAB_Active : BOOL; (*Ansaugluft A und B Seite aktiv*)
		bPr_Cool_Air_Re_Active : BOOL; (*Druckmessung im Kühlregister aktiv*)
		bPr_HW_Air_Re_Active : BOOL; (*Druckmessung im Heizregister aktiv*)
		bT_Cool_Air_Re_Active : BOOL; (*Rücklauf Temp. Messung im Kühlregister aktiv*)
		bT_Cool_Air_Su_Active : BOOL; (*Vorlauf Temp. Messung im Kühlregister aktiv*)
		bT_CircAirEng_Active : BOOL; (*Umluft Temp. Messung aktiv*)
		rTB_Cust : ARRAY[1..19]OF REAL; (*Parameter die für Tests vom Prüfstand verwendet werden können*)
		rT_PCGAfComp_HiHi : REAL; (*Limit gas temperature after prechamber gascompressor maximum*)
		rT_PCGAfCooler_HiHi : REAL; (*Limit gas temperature after cooler prechamber gascompressor maximum*)
		bPr_GT_NG_used : BOOL; (*Gas pressure natural gas used*)
		bPr_GT_PG_used : BOOL; (*Gas pressure propan gas used*)
		bPr_GT_SG_used : BOOL; (*Gas pressure special gas used*)
		bT_GT_NG_used : BOOL; (*Gas temperature natural gas used*)
		bT_GT_PG_used : BOOL; (*Gas temperature propan gas used*)
		bT_GT_SG_used : BOOL; (*Gas temperature special gas used*)
		bFlow_GT_NG_used : BOOL; (*Gas flow/counter natural gas used*)
		bFlow_GT_PG_used : BOOL; (*Gas flow/counter propan gas used*)
		bFlow_GT_SG_used : BOOL; (*Gas flow/counter special gas used*)
		bPCGC_AirCooler : BOOL; (*Prechamber gascompressor with air-cooler used*)
	END_STRUCT;
	Para_DI_struct : 	STRUCT
		tCtr_ChCW_LT : _tGeACtrPara; (*Para controller charge temperature cooler*) (*OldName:REG9; Cycle:5;*)
		bCtr_ChCW_LT : BOOL; (*PARA [11872]: visibility charge temperature controller*) (*OldName:bPlantCtr9,reg0_visible; Cycle:5;*)
		tCtr_ChCW_HT : _tGeACtrPara; (*Para controller charge temperature cooler*) (*OldName:REG9; Cycle:5;*)
		bCtr_ChCW_HT : BOOL; (*PARA [11872]: visibility charge temperature controller*) (*OldName:bPlantCtr9,reg0_visible; Cycle:5;*)
		tCtr_ChCW_HT_LP : _tGeACtrPara; (*Para controller charge temperature cooler*) (*OldName:REG9; Cycle:5;*)
		bCtr_ChCW_HT_LP : BOOL; (*PARA [11872]: visibility charge temperature controller*) (*OldName:bPlantCtr9,reg0_visible; Cycle:5;*)
		tCtr_ChCW_HT_HP : _tGeACtrPara; (*Para controller charge temperature cooler*) (*OldName:REG9; Cycle:5;*)
		bCtr_ChCW_HT_HP : BOOL; (*PARA [11872]: visibility charge temperature controller*) (*OldName:bPlantCtr9,reg0_visible; Cycle:5;*)
		tCtr_ChCW_LT_LP : _tGeACtrPara; (*Para controller charge temperature cooler*) (*OldName:REG9; Cycle:5;*)
		bCtr_ChCW_LT_LP : BOOL; (*PARA [11872]: visibility charge temperature controller*) (*OldName:bPlantCtr9,reg0_visible; Cycle:5;*)
		tCtr_ChCW_LT_HP : _tGeACtrPara; (*Para controller charge temperature cooler*) (*OldName:REG9; Cycle:5;*)
		bCtr_ChCW_LT_HP : BOOL; (*PARA [11872]: visibility charge temperature controller*) (*OldName:bPlantCtr9,reg0_visible; Cycle:5;*)
		tCtr_ECW : _tGeACtrPara; (*Para controller  engine cooling water temperature cooler*) (*OldName:REG9; Cycle:5;*)
		bCtr_ECW : BOOL; (*PARA [11872]: visibility  engine cooling water temperature controller*) (*OldName:bPlantCtr9,reg0_visible; Cycle:5;*)
		tCtr_OCW : _tGeACtrPara; (*Para controller  oil cooling water temperature cooler*) (*OldName:REG9; Cycle:5;*)
		bCtr_OCW : BOOL; (*PARA [11872]: visibility  oil cooling water temperature controller*) (*OldName:bPlantCtr9,reg0_visible; Cycle:5;*)
		bT_ChCW_Re_LT : BOOL; (*visu aktiv Temp Ladekühlwasser Rücklauf NT*)
		bPr_ChCW_Re_LT : BOOL; (*visu aktiv Druck Ladekühlwasser Rücklauf NT*)
		bT_ChCW_Su_LT : BOOL; (*visu aktiv Temp Ladekühlwasser Vorlauf NT*)
		bPr_ChCW_Su_LT : BOOL; (*visu aktiv Druck Ladekühlwasser Vorlauf NT*)
		bT_ChCW_Re_HT : BOOL; (*visu aktiv Temp Ladekühlwasser Rücklauf NT*)
		bPr_ChCW_Re_HT : BOOL; (*visu aktiv Druck Ladekühlwasser Rücklauf HT*)
		bT_ChCW_Su_HT : BOOL; (*visu aktiv Temp Ladekühlwasser Vorlauf HT*)
		bPr_ChCW_Su_HT : BOOL; (*visu aktiv Druck Ladekühlwasser Vorlauf HT*)
		bT_ChCW_Re_HT_LP : BOOL; (*visu aktiv Temp Ladekühlwasser Rücklauf HT ND*)
		bPr_ChCW_Re_HT_LP : BOOL; (*visu aktiv Druck Ladekühlwasser Rücklauf HT ND*)
		bT_ChCW_Re_HT_HP : BOOL; (*visu aktiv Temp Ladekühlwasser Rücklauf HT HD*)
		bPr_ChCW_Re_HT_HP : BOOL; (*visu aktiv Druck Ladekühlwasser Rücklauf HT HD*)
		bT_ChCW_Su_HT_LP : BOOL; (*visu aktiv Temp Ladekühlwasser Vorlauf HT ND*)
		bPr_ChCW_Su_HT_LP : BOOL; (*visu aktiv Druck Ladekühlwasser Vorlauf HT ND*)
		bT_ChCW_Su_HT_HP : BOOL; (*visu aktiv Temp Ladekühlwasser Vorlauf HT HD*)
		bPr_ChCW_Su_HT_HP : BOOL; (*visu aktiv Druck Ladekühlwasser Vorlauf HT HD*)
		bT_ChCW_Re_LT_LP : BOOL; (*visu aktiv Temp Ladekühlwasser Rücklauf NT ND*)
		bPr_ChCW_Re_LT_LP : BOOL; (*visu aktiv Druck Ladekühlwasser Rücklauf NT ND*)
		bT_ChCW_Re_LT_HP : BOOL; (*visu aktiv Temp Ladekühlwasser Rücklauf NT HD*)
		bPr_ChCW_Re_LT_HP : BOOL; (*visu aktiv Druck Ladekühlwasser Rücklauf NT HD*)
		bT_ChCW_Su_LT_LP : BOOL; (*visu aktiv Temp Ladekühlwasser Vorlauf NT ND*)
		bPr_ChCW_Su_LT_LP : BOOL; (*visu aktiv Druck Ladekühlwasser Vorlauf NT ND*)
		bT_ChCW_Su_LT_HP : BOOL; (*visu aktiv Temp Ladekühlwasser Vorlauf NT HD*)
		bPr_ChCW_Su_LT_HP : BOOL; (*visu aktiv Druck Ladekühlwasser Vorlauf NT HD*)
		bT_OCW_Re : BOOL; (*visu aktiv Temp Ölkühlwasser Rücklauf*)
		bPr_OCW_Re : BOOL; (*visu aktiv Druck Ölkühlwasser Rücklauf*)
		bT_OCW_Su : BOOL; (*visu aktiv Temp Ölkühlwasser Vorlauf*)
		bPr_OCW_Su : BOOL; (*visu aktiv Druck Ölkühlwasser Vorlauf*)
		bT_ECW_Re : BOOL; (*visu aktiv Temp Motorkühlwasser Rücklauf*)
		bPr_ECW_Re : BOOL; (*visu aktiv Druck Motorkühlwasser Rücklauf*)
		bT_ECW_Su : BOOL; (*visu aktiv Temp Motorkühlwasser Vorlauf*)
		bPr_ECW_Su : BOOL; (*visu aktiv Druck Motorkühlwasser Vorlauf*)
		bVol_ChCW_Re_LT : BOOL; (*visu aktiv Durchfluss Ladekühlwasser Rücklauf NT*)
		bVol_ChCW_Su_LT : BOOL; (*visu aktiv Durchfluss Ladekühlwasser Vorlauf NT*)
		bVol_ChCW_Re_HT : BOOL; (*visu aktiv Durchfluss Ladekühlwasser Rücklauf HT*)
		bVol_ChCW_Su_HT : BOOL; (*visu aktiv Durchfluss Ladekühlwasser Vorlauf HT*)
		bVol_ChCW_Re_HT_LP : BOOL; (*visu aktiv Durchfluss Ladekühlwasser Rücklauf HT ND*)
		bVol_ChCW_Su_HT_LP : BOOL; (*visu aktiv Durchfluss Ladekühlwasser Vorlauf HT ND*)
		bVol_ChCW_Re_HT_HP : BOOL; (*visu aktiv Durchfluss Ladekühlwasser Rücklauf HT HD*)
		bVol_ChCW_Su_HT_HP : BOOL; (*visu aktiv Durchfluss Ladekühlwasser Vorlauf HT HD*)
		bVol_ChCW_Re_LT_LP : BOOL; (*visu aktiv Durchfluss Ladekühlwasser Rücklauf NT ND*)
		bVol_ChCW_Su_LT_LP : BOOL; (*visu aktiv Durchfluss Ladekühlwasser Vorlauf NT ND*)
		bVol_ChCW_Re_LT_HP : BOOL; (*visu aktiv Durchfluss Ladekühlwasser Rücklauf NT HD*)
		bVol_ChCW_Su_LT_HP : BOOL; (*visu aktiv Durchfluss Ladekühlwasser Vorlauf NT HD*)
		bVol_ECW_Re : BOOL; (*visu aktiv Durchfluss Motorkühlwasser Rücklauf*)
		bVol_ECW_Su : BOOL; (*visu aktiv Durchfluss Motorkühlwasser Vorlauf*)
		bVol_OCW_Re : BOOL; (*visu aktiv Durchfluss Ölkühlwasser Rücklauf*)
		bVol_OCW_Su : BOOL; (*visu aktiv Durchfluss Ölkühlwasser Vorlauf*)
		bT_ChCW_LT_IC_Re : BOOL; (*visu aktiv Temp Ladekühlewasser NT Zwischenkreis Rücklauf*)
		bPr_ChCW_LT_IC_Re : BOOL; (*visu aktiv Druck Ladekühlewasser NT Zwischenkreis Rücklauf*)
		bT_ChCW_HT_IC_Re : BOOL; (*visu aktiv Temp Ladekühlewasser HT Zwischenkreis Rücklauf*)
		bPr_ChCW_HT_IC_Re : BOOL; (*visu aktiv Druck Ladekühlewasser HT Zwischenkreis Rücklauf*)
		bT_ChCW_LT_LP_IC_Re : BOOL; (*visu aktiv Temp Ladekühlewasser NT ND Zwischenkreis Rücklauf*)
		bPr_ChCW_LT_LP_IC_Re : BOOL; (*visu aktiv Druck Ladekühlewasser NT ND Zwischenkreis Rücklauf*)
		bT_ChCW_LT_HP_IC_Re : BOOL; (*visu aktiv Temp Ladekühlewasser NT HD Zwischenkreis Rücklauf*)
		bPr_ChCW_LT_HP_IC_Re : BOOL; (*visu aktiv Druck Ladekühlewasser NT HD Zwischenkreis Rücklauf*)
		bT_ChCW_HT_LP_IC_Re : BOOL; (*visu aktiv Temp Ladekühlewasser HT ND Zwischenkreis Rücklauf*)
		bPr_ChCW_HT_LP_IC_Re : BOOL; (*visu aktiv Druck Ladekühlewasser HT ND Zwischenkreis Rücklauf*)
		bT_ChCW_HT_HP_IC_Re : BOOL; (*visu aktiv Temp Ladekühlewasser HT HD Zwischenkreis Rücklauf*)
		bPr_ChCW_HT_HP_IC_Re : BOOL; (*visu aktiv Druck Ladekühlewasser HT HD Zwischenkreis Rücklauf*)
		bT_ECW_IC_Re : BOOL; (*visu aktiv Temp Motorkühlwasser Zwischenkreis Rücklauf*)
		bPr_ECW_IC_Re : BOOL; (*visu aktiv Druck Motorkühlwasser Zwischenkreis Rücklauf*)
		bT_OCW_IC_Re : BOOL; (*visu aktiv Temp Ölkühlwasser Zwischenkreis Rücklauf*)
		bPr_OCW_IC_Re : BOOL; (*visu aktiv Druck Ölkühlwasser Zwischenkreis Rücklauf*)
		bT_ChCW_LT_IC_Su : BOOL; (*visu aktiv Temp Ladekühlewasser NT Zwischenkreis Rücklauf*)
		bPr_ChCW_LT_IC_Su : BOOL; (*visu aktiv Druck Ladekühlewasser NT Zwischenkreis Rücklauf*)
		bT_ChCW_HT_IC_Su : BOOL; (*visu aktiv Temp Ladekühlewasser HT Zwischenkreis Rücklauf*)
		bPr_ChCW_HT_IC_Su : BOOL; (*visu aktiv Druck Ladekühlewasser HT Zwischenkreis Rücklauf*)
		bT_ChCW_LT_LP_IC_Su : BOOL; (*visu aktiv Temp Ladekühlewasser NT ND Zwischenkreis Rücklauf*)
		bPr_ChCW_LT_LP_IC_Su : BOOL; (*visu aktiv Druck Ladekühlewasser NT ND Zwischenkreis Rücklauf*)
		bT_ChCW_LT_HP_IC_Su : BOOL; (*visu aktiv Temp Ladekühlewasser NT HD Zwischenkreis Rücklauf*)
		bPr_ChCW_LT_HP_IC_Su : BOOL; (*visu aktiv Druck Ladekühlewasser NT HD Zwischenkreis Rücklauf*)
		bT_ChCW_HT_LP_IC_Su : BOOL; (*visu aktiv Temp Ladekühlewasser HT ND Zwischenkreis Rücklauf*)
		bPr_ChCW_HT_LP_IC_Su : BOOL; (*visu aktiv Druck Ladekühlewasser HT ND Zwischenkreis Rücklauf*)
		bT_ChCW_HT_HP_IC_Su : BOOL; (*visu aktiv Temp Ladekühlewasser HT HD Zwischenkreis Rücklauf*)
		bPr_ChCW_HT_HP_IC_Su : BOOL; (*visu aktiv Druck Ladekühlewasser HT HD Zwischenkreis Rücklauf*)
		bT_ECW_IC_Su : BOOL; (*visu aktiv Temp Motorkühlwasser Zwischenkreis Rücklauf*)
		bPr_ECW_IC_Su : BOOL; (*visu aktiv Druck Motorkühlwasser Zwischenkreis Rücklauf*)
		bT_OCW_IC_Su : BOOL; (*visu aktiv Temp Ölkühlwasser Zwischenkreis Rücklauf*)
		bPr_OCW_IC_Su : BOOL; (*visu aktiv Druck Ölkühlwasser Zwischenkreis Vorlauf*)
		bT_Cooler_ChCW_LT_Re_1 : BOOL; (*visu aktiv Temp Kühler Ladekühlwasser NT Rücklauf*)
		bT_Cooler_ChCW_LT_Re_2 : BOOL; (*visu aktiv Temp Kühler Ladekühlwasser NT Rücklauf*)
		bT_Cooler_ChCW_HT_Re_1 : BOOL; (*visu aktiv Temp Kühler Ladekühlwasser HT Rücklauf*)
		bT_Cooler_ChCW_HT_Re_2 : BOOL; (*visu aktiv Temp Kühler Ladekühlwasser HT Rücklauf*)
		bT_Cooler_ChCW_LT_LP_Re_1 : BOOL; (*visu aktiv Temp Kühler Ladekühlwasser NT ND Rücklauf*)
		bT_Cooler_ChCW_LT_LP_Re_2 : BOOL; (*visu aktiv Temp Kühler Ladekühlwasser NT ND Rücklauf*)
		bT_Cooler_ChCW_LT_HP_Re_1 : BOOL; (*visu aktiv Temp Kühler Ladekühlwasser NT HD Rücklauf*)
		bT_Cooler_ChCW_LT_HP_Re_2 : BOOL; (*visu aktiv Temp Kühler Ladekühlwasser NT HD Rücklauf*)
		bT_Cooler_ChCW_HT_LP_Re_1 : BOOL; (*visu aktiv Temp Kühler Ladekühlwasser HT ND Rücklauf*)
		bT_Cooler_ChCW_HT_LP_Re_2 : BOOL; (*visu aktiv Temp Kühler Ladekühlwasser HT ND Rücklauf*)
		bT_Cooler_ChCW_HT_HP_Re_1 : BOOL; (*visu aktiv Temp Kühler Ladekühlwasser HT HD Rücklauf*)
		bT_Cooler_ChCW_HT_HP_Re_2 : BOOL; (*visu aktiv Temp Kühler Ladekühlwasser HT HD Rücklauf*)
		bT_Cooler_ECW_Re_1 : BOOL; (*visu aktiv Temp Kühler Motorkühlwasser Rücklauf*)
		bT_Cooler_ECW_Re_2 : BOOL; (*visu aktiv Temp Kühler Motorkühlwasser Rücklauf*)
		bT_Cooler_OCW_Re_1 : BOOL; (*visu aktiv Temp Kühler Ölkühlwasser Rücklauf*)
		bT_Cooler_OCW_Re_2 : BOOL; (*visu aktiv Temp Kühler Ölkühlwasser Rücklauf*)
		bPr_Cooler_ChCW_LT_Re_1 : BOOL; (*visu aktiv Druck Kühler Ladekühlwasser NT Rücklauf*)
		bPr_Cooler_ChCW_LT_Re_2 : BOOL; (*visu aktiv Druck Kühler Ladekühlwasser NT Rücklauf*)
		bPr_Cooler_ChCW_HT_Re_1 : BOOL; (*visu aktiv Druck Kühler Ladekühlwasser HT Rücklauf*)
		bPr_Cooler_ChCW_HT_Re_2 : BOOL; (*visu aktiv Druck Kühler Ladekühlwasser HT Rücklauf*)
		bPr_Cooler_ChCW_LT_LP_Re_1 : BOOL; (*visu aktiv Druck Kühler Ladekühlwasser NT ND Rücklauf*)
		bPr_Cooler_ChCW_LT_LP_Re_2 : BOOL; (*visu aktiv Druck Kühler Ladekühlwasser NT ND Rücklauf*)
		bPr_Cooler_ChCW_LT_HP_Re_1 : BOOL; (*visu aktiv Druck Kühler Ladekühlwasser NT HD Rücklauf*)
		bPr_Cooler_ChCW_LT_HP_Re_2 : BOOL; (*visu aktiv Druck Kühler Ladekühlwasser NT HD Rücklauf*)
		bPr_Cooler_ChCW_HT_LP_Re_1 : BOOL; (*visu aktiv Druck Kühler Ladekühlwasser HT ND Rücklauf*)
		bPr_Cooler_ChCW_HT_LP_Re_2 : BOOL; (*visu aktiv Druck Kühler Ladekühlwasser HT ND Rücklauf*)
		bPr_Cooler_ChCW_HT_HP_Re_1 : BOOL; (*visu aktiv Druck Kühler Ladekühlwasser HT HD Rücklauf*)
		bPr_Cooler_ChCW_HT_HP_Re_2 : BOOL; (*visu aktiv Druck Kühler Ladekühlwasser HT HD Rücklauf*)
		bPr_Cooler_ECW_Re_1 : BOOL; (*visu aktiv Druck Kühler Motorkühlwasser Rücklauf*)
		bPr_Cooler_ECW_Re_2 : BOOL; (*visu aktiv Druck Kühler Motorkühlwasser Rücklauf*)
		bPr_Cooler_OCW_Re_1 : BOOL; (*visu aktiv Druck Kühler Ölkühlwasser Rücklauf*)
		bPr_Cooler_OCW_Re_2 : BOOL; (*visu aktiv Druck Kühler Ölkühlwasser Rücklauf*)
		bT_Cooler_ChCW_LT_Su_1 : BOOL; (*visu aktiv Temp Kühler Ladekühlwasser NT Vorlauf*)
		bT_Cooler_ChCW_LT_Su_2 : BOOL; (*visu aktiv Temp Kühler Ladekühlwasser NT Vorlauf*)
		bT_Cooler_ChCW_HT_Su_1 : BOOL; (*visu aktiv Temp Kühler Ladekühlwasser HT Vorlauf*)
		bT_Cooler_ChCW_HT_Su_2 : BOOL; (*visu aktiv Temp Kühler Ladekühlwasser HT Vorlauf*)
		bT_Cooler_ChCW_LT_LP_Su_1 : BOOL; (*visu aktiv Temp Kühler Ladekühlwasser NT ND Vorlauf*)
		bT_Cooler_ChCW_LT_LP_Su_2 : BOOL; (*visu aktiv Temp Kühler Ladekühlwasser NT ND Vorlauf*)
		bT_Cooler_ChCW_LT_HP_Su_1 : BOOL; (*visu aktiv Temp Kühler Ladekühlwasser NT HD Vorlauf*)
		bT_Cooler_ChCW_LT_HP_Su_2 : BOOL; (*visu aktiv Temp Kühler Ladekühlwasser NT HD Vorlauf*)
		bT_Cooler_ChCW_HT_LP_Su_1 : BOOL; (*visu aktiv Temp Kühler Ladekühlwasser HT ND Vorlauf*)
		bT_Cooler_ChCW_HT_LP_Su_2 : BOOL; (*visu aktiv Temp Kühler Ladekühlwasser HT ND Vorlauf*)
		bT_Cooler_ChCW_HT_HP_Su_1 : BOOL; (*visu aktiv Temp Kühler Ladekühlwasser HT HD Vorlauf*)
		bT_Cooler_ChCW_HT_HP_Su_2 : BOOL; (*visu aktiv Temp Kühler Ladekühlwasser HT HD Vorlauf*)
		bT_Cooler_ECW_Su_1 : BOOL; (*visu aktiv Temp Kühler Motorkühlwasser Vorlauf*)
		bT_Cooler_ECW_Su_2 : BOOL; (*visu aktiv Temp Kühler Motorkühlwasser Vorlauf*)
		bT_Cooler_OCW_Su_1 : BOOL; (*visu aktiv Temp Kühler Ölkühlwasser Vorlauf*)
		bT_Cooler_OCW_Su_2 : BOOL; (*visu aktiv Temp Kühler Ölkühlwasser Vorlauf*)
		bPr_Cooler_ChCW_LT_Su_1 : BOOL; (*visu aktiv Druck Kühler Ladekühlwasser NT Vorlauf*)
		bPr_Cooler_ChCW_LT_Su_2 : BOOL; (*visu aktiv Druck Kühler Ladekühlwasser NT Vorlauf*)
		bPr_Cooler_ChCW_HT_Su_1 : BOOL; (*visu aktiv Druck Kühler Ladekühlwasser HT Vorlauf*)
		bPr_Cooler_ChCW_HT_Su_2 : BOOL; (*visu aktiv Druck Kühler Ladekühlwasser HT Vorlauf*)
		bPr_Cooler_ChCW_LT_LP_Su_1 : BOOL; (*visu aktiv Druck Kühler Ladekühlwasser NT ND Vorlauf*)
		bPr_Cooler_ChCW_LT_LP_Su_2 : BOOL; (*visu aktiv Druck Kühler Ladekühlwasser NT ND Vorlauf*)
		bPr_Cooler_ChCW_LT_HP_Su_1 : BOOL; (*visu aktiv Druck Kühler Ladekühlwasser NT HD Vorlauf*)
		bPr_Cooler_ChCW_LT_HP_Su_2 : BOOL; (*visu aktiv Druck Kühler Ladekühlwasser NT HD Vorlauf*)
		bPr_Cooler_ChCW_HT_LP_Su_1 : BOOL; (*visu aktiv Druck Kühler Ladekühlwasser HT ND Vorlauf*)
		bPr_Cooler_ChCW_HT_LP_Su_2 : BOOL; (*visu aktiv Druck Kühler Ladekühlwasser HT ND Vorlauf*)
		bPr_Cooler_ChCW_HT_HP_Su_1 : BOOL; (*visu aktiv Druck Kühler Ladekühlwasser HT HD Vorlauf*)
		bPr_Cooler_ChCW_HT_HP_Su_2 : BOOL; (*visu aktiv Druck Kühler Ladekühlwasser HT HD Vorlauf*)
		bPr_Cooler_ECW_Su_1 : BOOL; (*visu aktiv Druck Kühler Motorkühlwasser Vorlauf*)
		bPr_Cooler_ECW_Su_2 : BOOL; (*visu aktiv Druck Kühler Motorkühlwasser Vorlauf*)
		bPr_Cooler_OCW_Su_1 : BOOL; (*visu aktiv Druck Kühler Ölkühlwasser Vorlauf*)
		bPr_Cooler_OCW_Su_2 : BOOL; (*visu aktiv Druck Kühler Ölkühlwasser Vorlauf*)
		bT_ChCW_LT_bCV : BOOL; (*visu aktiv Temp Ladekühlwasser NT vor Regelventil*)
		bT_ChCW_LT_LP_bCV : BOOL; (*visu aktiv Temp Ladekühlwasser NT ND vor Regelventil*)
		bT_ChCW_LT_HP_bCV : BOOL; (*visu aktiv Temp Ladekühlwasser NT HD vor Regelventil*)
		bT_ChCW_HT_bCV : BOOL; (*visu aktiv Temp Ladekühlwasser NT vor Regelventil*)
		bT_ChCW_HT_LP_bCV : BOOL; (*visu aktiv Temp Ladekühlwasser NT ND vor Regelventil*)
		bT_ChCW_HT_HP_bCV : BOOL; (*visu aktiv Temp Ladekühlwasser NT HD vor Regelventil*)
		bT_ECW_bCV : BOOL; (*visu aktiv Temp Motorkühlwasser vor Regelventil*)
		bT_OCW_bCV : BOOL; (*visu aktiv Temp Ölkühlwasser vor Regelventil*)
		bT_RW_HE_Re : BOOL; (*visu aktiv Temp Rohwasser Wärmetausche Rücklauf*)
		bT_RW_HE_Su : BOOL; (*visu aktiv Temp Rohwasser Wärmetausche Vorlauf*)
		bPr_RW_HE_Re : BOOL; (*visu aktiv Druck Rohwasser Wärmetausche Rücklauf*)
		bPr_RW_HE_Su : BOOL; (*visu aktiv Druck Rohwasser Wärmetausche Vorlauf*)
		bCtr_RW_CV : BOOL; (*visu aktiv Regler Rohwasser Regelventil*)
		bCtr_RW_HE : BOOL; (*visu aktiv Regler Rohwasser Wärmetausche*)
		bFC_ChCW_LT_Pump : BOOL; (*visu aktiv FU Ladekühlewasser NT*)
		bFC_ChCW_HT_Pump : BOOL; (*visu aktiv FU Ladekühlewasser HT*)
		bFC_ChCW_LT_LP_Pump : BOOL; (*visu aktiv FU Ladekühlewasser NT ND*)
		bFC_ChCW_LT_HP_Pump : BOOL; (*visu aktiv FU Ladekühlewasser NT HD*)
		bFC_ChCW_HT_LP_Pump : BOOL; (*visu aktiv FU Ladekühlewasser HT ND*)
		bFC_ChCW_HT_HP_Pump : BOOL; (*visu aktiv FU Ladekühlewasser HT HD*)
		bFC_ECW_Pump : BOOL; (*visu aktiv FU Motorkühlwasser*)
		bFC_OCW_Pump : BOOL; (*visu aktiv FU Ölkühlwasser*)
		bFC_ChCW_LT_Cooler_1 : BOOL; (*visu aktiv FU Ladekühlwasser NT Kühler*)
		bFC_ChCW_LT_Cooler_2 : BOOL; (*visu aktiv FU Ladekühlwasser NT Kühler*)
		bFC_ChCW_HT_Cooler_1 : BOOL; (*visu aktiv FU Ladekühlwasser HT Kühler*)
		bFC_ChCW_HT_Cooler_2 : BOOL; (*visu aktiv FU Ladekühlwasser HT Kühler*)
		bFC_ChCW_LT_LP_Cooler_1 : BOOL; (*visu aktiv FU Ladekühlwasser NT ND Kühler*)
		bFC_ChCW_LT_LP_Cooler_2 : BOOL; (*visu aktiv FU Ladekühlwasser NT ND Kühler*)
		bFC_ChCW_LT_HP_Cooler_1 : BOOL; (*visu aktiv FU Ladekühlwasser NT HD Kühler*)
		bFC_ChCW_LT_HP_Cooler_2 : BOOL; (*visu aktiv FU Ladekühlwasser NT HD Kühler*)
		bFC_ChCW_HT_LP_Cooler_1 : BOOL; (*visu aktiv FU Ladekühlwasser HT ND Kühler*)
		bFC_ChCW_HT_LP_Cooler_2 : BOOL; (*visu aktiv FU Ladekühlwasser HT ND Kühler*)
		bFC_ChCW_HT_HP_Cooler_1 : BOOL; (*visu aktiv FU Ladekühlwasser HT HD Kühler*)
		bFC_ChCW_HT_HP_Cooler_2 : BOOL; (*visu aktiv FU Ladekühlwasser HT HD Kühler*)
		bFC_ECW_Cooler_1 : BOOL; (*visu aktiv FU Motorkühlwasser Kühler*)
		bFC_ECW_Cooler_2 : BOOL; (*visu aktiv FU Motorkühlwasser Kühler*)
		bFC_OCW_Cooler_1 : BOOL; (*visu aktiv FU Ölkühlwasser Kühler*)
		bFC_OCW_Cooler_2 : BOOL; (*visu aktiv FU Ölkühlwasser Kühler*)
		bPs_ChCW_LT_bEngine_Hi : BOOL; (*visu aktiv Druckschalter Ladekühlewasser NT vor Motor max*)
		bPs_ChCW_HT_bEngine_Hi : BOOL; (*visu aktiv Druckschalter Ladekühlewasser HT vor Motor max*)
		bPs_ChCW_LT_LP_bEngine_Hi : BOOL; (*visu aktiv Druckschalter Ladekühlewasser NT ND vor Motor max*)
		bPs_ChCW_LT_HP_bEngine_Hi : BOOL; (*visu aktiv Druckschalter Ladekühlewasser NT HD vor Motor max*)
		bPs_ChCW_HT_LP_bEngine_Hi : BOOL; (*visu aktiv Druckschalter Ladekühlewasser HT ND vor Motor max*)
		bPs_ChCW_HT_HP_bEngine_Hi : BOOL; (*visu aktiv Druckschalter Ladekühlewasser HT HD vor Motor max*)
		bPs_ECW_bEngine_Hi : BOOL; (*visu aktiv Druckschalter Motorkühlwasser vor Motor max*)
		bPs_OCW_bEngine_Hi : BOOL; (*visu aktiv Druckschalter Ölkühlwasser vor Motor max*)
		bPs_ChCW_LT_bPump_Low : BOOL; (*visu aktiv Druckschalter Ladekühlewasser NT vor Pumpe min*)
		bPs_ChCW_HT_bPump_Low : BOOL; (*visu aktiv Druckschalter Ladekühlewasser HT vor Pumpe min*)
		bPs_ChCW_LT_LP_bPump_Low : BOOL; (*visu aktiv Druckschalter Ladekühlewasser NT ND vor Pumpe min*)
		bPs_ChCW_LT_HP_bPump_Low : BOOL; (*visu aktiv Druckschalter Ladekühlewasser NT HD vor Pumpe min*)
		bPs_ChCW_HT_LP_bPump_Low : BOOL; (*visu aktiv Druckschalter Ladekühlewasser HT ND vor Pumpe min*)
		bPs_ChCW_HT_HP_bPump_Low : BOOL; (*visu aktiv Druckschalter Ladekühlewasser HT HD vor Pumpe min*)
		bPs_ECW_bPump_Low : BOOL; (*visu aktiv Druckschalter Motorkühlwasser vor Pumpe min*)
		bPs_OCW_bPump_Low : BOOL; (*visu aktiv Druckschalter Ölkühlwasser vor Pumpe min*)
		bTs_ChCW_LT_bEngine_Hi : BOOL; (*visu aktiv Temperaturschalter Ladekühlewasser NT vor Motor max*)
		bTs_ChCW_HT_bEngine_Hi : BOOL; (*visu aktiv Temperaturschalter Ladekühlewasser HT vor Motor max*)
		bTs_ChCW_LT_LP_bEngine_Hi : BOOL; (*visu aktiv Temperaturschalter Ladekühlewasser NT ND vor Motor max*)
		bTs_ChCW_LT_HP_bEngine_Hi : BOOL; (*visu aktiv Temperaturschalter Ladekühlewasser NT HD vor Motor max*)
		bTs_ChCW_HT_LP_bEngine_Hi : BOOL; (*visu aktiv Temperaturschalter Ladekühlewasser HT ND vor Motor max*)
		bTs_ChCW_HT_HP_bEngine_Hi : BOOL; (*visu aktiv Temperaturschalter Ladekühlewasser HT HD vor Motor max*)
		bTs_ECW_bEngine_Hi : BOOL; (*visu aktiv Temperaturschalter Motorkühlwasser vor Motor max*)
		bTs_OCW_bEngine_Hi : BOOL; (*visu aktiv Temperaturschalter Ölkühlwasser vor Motor max*)
		bDem_Cooler_ChCW_LT_1 : BOOL; (*visu aktiv Anforderung Kühler Ladekühlwasser NT*)
		bDem_Cooler_ChCW_LT_2 : BOOL; (*visu aktiv Anforderung Kühler Ladekühlwasser NT*)
		bDem_Cooler_ChCW_HT_1 : BOOL; (*visu aktiv Anforderung Kühler Ladekühlwasser HT*)
		bDem_Cooler_ChCW_HT_2 : BOOL; (*visu aktiv Anforderung Kühler Ladekühlwasser HT*)
		bDem_Cooler_ChCW_LT_LP_1 : BOOL; (*visu aktiv Anforderung Kühler Ladekühlwasser NT ND*)
		bDem_Cooler_ChCW_LT_LP_2 : BOOL; (*visu aktiv Anforderung Kühler Ladekühlwasser NT ND*)
		bDem_Cooler_ChCW_LT_HP_1 : BOOL; (*visu aktiv Anforderung Kühler Ladekühlwasser NT HD*)
		bDem_Cooler_ChCW_LT_HP_2 : BOOL; (*visu aktiv Anforderung Kühler Ladekühlwasser NT HD*)
		bDem_Cooler_ChCW_HT_LP_1 : BOOL; (*visu aktiv Anforderung Kühler Ladekühlwasser HT ND*)
		bDem_Cooler_ChCW_HT_LP_2 : BOOL; (*visu aktiv Anforderung Kühler Ladekühlwasser HT ND*)
		bDem_Cooler_ChCW_HT_HP_1 : BOOL; (*visu aktiv Anforderung Kühler Ladekühlwasser HT HD*)
		bDem_Cooler_ChCW_HT_HP_2 : BOOL; (*visu aktiv Anforderung Kühler Ladekühlwasser HT HD*)
		bDem_Cooler_ECW_1 : BOOL; (*visu aktiv Anforderung Kühler Motorkühlwasser*)
		bDem_Cooler_ECW_2 : BOOL; (*visu aktiv Anforderung Kühler Motorkühlwasser*)
		bDem_Cooler_OCW_1 : BOOL; (*visu aktiv Anforderung Kühler Ölkühlwasser*)
		bDem_Cooler_OCW_2 : BOOL; (*visu aktiv Anforderung Kühler Ölkühlwasser*)
		bDem_ChCW_LT_Pump : BOOL; (*visu aktiv Anforderung Ladekühlewasser NT Pumpe*)
		bDem_ChCW_HT_Pump : BOOL; (*visu aktiv Anforderung Ladekühlewasser HT Pumpe*)
		bDem_ChCW_LT_LP_Pump : BOOL; (*visu aktiv Anforderung Ladekühlewasser NT ND Pumpe*)
		bDem_ChCW_LT_HP_Pump : BOOL; (*visu aktiv Anforderung Ladekühlewasser NT HD Pumpe*)
		bDem_ChCW_HT_LP_Pump : BOOL; (*visu aktiv Anforderung Ladekühlewasser HT ND Pumpe*)
		bDem_ChCW_HT_HP_Pump : BOOL; (*visu aktiv Anforderung Ladekühlewasser HT HD Pumpe*)
		bDem_ECW_Pump : BOOL; (*visu aktiv Anforderung Motorkühlwasser Pumpe*)
		bDem_OCW_Pump : BOOL; (*visu aktiv Anforderung Ölkühlwasser Pumpe*)
		rT_CtrER_WexRun : REAL; (*engine room temperature controller external setpoint run*)
		rT_ACP_AirER_sp : REAL; (*Active cooling program setpoint temperature engine room ventilation*)
		rT_CtrER_WexStop : REAL; (*engine room temperature controller external setpoint stop*)
		bT_AirER1_Active : BOOL; (*Raumtemperatur 1 aktiv*)
		bT_AirER2_Active : BOOL; (*Raumtemperatur 2 aktiv*)
		bT_AirER3_Active : BOOL; (*Raumtemperatur 3 aktiv*)
		bT_AirER4_Active : BOOL; (*Raumtemperatur 4 aktiv*)
		bT_AirOutdoor_Active : BOOL; (*PARA [11885]: air outdoor temperature measurement enable *) (*OldName:ULT_a; Cycle:5;*)
		bIntakeAirCond : BOOL; (*Zuluftkonditionierung Aktiv*)
		bPrDiff_ER_Active : BOOL; (*Messung Raumdiffernzdruck aktiv*)
		bCtr_ER : BOOL; (*Raumlufttemperaturregler aktiv*)
		bCtr_OutlVE_RDP : BOOL; (*air outlet ventilation controller for room differential pressure enable*)
		tCtr_IntakeAir : _tGeACtrPara; (*Para Regler für Motor Ansaugluft*)
		tCtr_ER : _tGeACtrPara; (*Para controller engine room temperature*)
		tCtr_OutlVE_RDP : _tGeACtrPara; (*Para controller air outlet ventilation (for engine room differential pressure)*)
		tCtr_EG_Flap : _tGeACtrPara; (*Para Abgasklappenregler*)
		rLSCS_MV_Set : REAL; (*Vorgabe LSCS Mischventil*)
		rLSCS_GV_Set : REAL; (*Vorgabe LSCS Gasventil*)
		rSel_LSCS_MV : REAL; (*Vorgabe Koeffizient der Blende vom Mischventil*)
		rSel_LSCS_GV : REAL; (*Vorgabe Koeffizient der Blende vom Gasventil*)
		tCtr_GC_1 : _tGeACtrPara; (*Para Gaskompressorregler 1*)
		tCtr_GC_2 : _tGeACtrPara; (*Para Gaskompressorregler 2*)
		tCtr_MN_MG : _tGeACtrPara; (*Para Gas mischen regler*)
		bSG_active : BOOL; (*Sondergasstrecke aktiv*)
		tPreHeatWDay : ARRAY[0..7]OF PreHeatWDay; (*Variablen für die Zeitsteuerung für Vorwärmung*)
		bPreHeatWDay_CtrActive : BOOL; (*Allgemeine Aktivierung der Zeitsteurerung*)
		bLSCS_GV_active : BOOL; (*LSCS Gasventil aktiv*)
		bLSCS_MV_active : BOOL; (*LSCS Mischventil aktiv*)
		iSel_Cooling : INT; (*Auswahl Srt der Kühlung*)
		bGasCompActive : BOOL; (*Zähler Gascompressor aktiv*)
		bGasCntSensycalActive : BOOL; (*Gaszähler Sensycal aktiv*)
		bGasCntCalcActive : BOOL; (*Gaszähler berechnet aktiv*)
		rCnt_CompOpHoursW : REAL; (* compressor operating hours counter until warning *)
		bH2_Mode : BOOL; (* Gasstrecke 3, TRUE = H2 aktiv *)
		bGasFlowCtr : BOOL; (* Gas flow control via engine controller setpoints for transient mixgas*)
		bSG_MFC_Used : BOOL; (* Special gas MFC used *)
		bPG_MFC_Used : BOOL; (* propan gas MFC used *)
		bBatCtrActive : BOOL; (* Batterieüberwachung wird visualisiert *)
		bIncl_SG_Calc : BOOL; (*Include special gas for MN & CV calculation*)
		bSend_Cv2Eng : BOOL; (*Send calculated CV  to  engine*)
		iNumInlLou : INT; (*Number of Louvers*)
		iNumInlLouRoom : INT; (*Number of Louvers*)
		iNumOutlLou : INT; (*Number of Louvers*)
		iNumCircLou : INT; (*Number of Louvers*)
		iNumInlLouEng : INT; (*Number of Louvers*)
		iNumCircLouEng : INT; (*Number of Louvers*)
		iVisRoomLou : INT; (*indication of room ventilation*)
		bPr_EG_DeflagActive : BOOL; (*Abgasdruck auf Visu aktiv*)
		bEG_SRC_DPF_Active : BOOL; (*Abgasseite für SCR und DPF auf Visu aktiv*)
		rLevel_Oiltank_ScalY1 : REAL; (*Öltankstand min Skalierung*)
		rLevel_Oiltank_ScalY2 : REAL; (*Öltankstand max Skalierung*)
		bAirCondHeaterActive : BOOL; (*Zuluftkonditionierung Heizung aktiv*)
		bTs_bEngineHiActive : BOOL; (*Temperaturschalter Max vor Motor bei Wärmetauscher aktiv (gilt für alle Kühlkreise)*)
		bPs_bEngineHiActive : BOOL; (*Druckschalter Max vor Motor bei Wärmetauscher aktiv (gilt für alle Kühlkreise)*)
		bT_bCV_Active : BOOL; (*Temperatur vor Temperaturregelventil aktiv (gilt für alle Kühlkreise)*)
		bT_Cooler_Re_Active : BOOL; (*Temperatur Rücklauf beim Kühler aktiv (gilt für alle Kühlkreise)*)
		bT_Cooler_Su_Active : BOOL; (*Temperatur Vorlauf beim Kühler aktiv (gilt für alle Kühlkreise)*)
		bPr_Cooler_Re_Active : BOOL; (*Druck Rücklauf beim Kühler aktiv (gilt für alle Kühlkreise)*)
		bPr_Cooler_Su_Active : BOOL; (*Druck Vorlauf beim Kühler aktiv (gilt für alle Kühlkreise)*)
		bExtCtrNOX_Active : BOOL; (*Externe NOX Regelung aktiv*)
		bPs_RW_Active : BOOL; (*Druckschalter Rohwasser Sammelleitung aktiv*)
		bTs_RW_Active : BOOL; (*Temperaturschalter Rohwasser Sammelleitung aktiv*)
		bT_RW_Re_Active : BOOL; (*Temperatur Rohwasser Rücklauf Sammelleitung aktiv*)
		bT_RW_Su_Active : BOOL; (*Temperatur Rohwasser Vorlauf Sammelleitung aktiv*)
		bFB_CC_Active : BOOL; (*Rückmeldung Kühlkreis Regelventile aktiv*)
		bFB_Cooler_Active : BOOL; (*Rückmeldung Kühler aktiv*)
		bFB_AC_Heating_Active : BOOL; (*Rückmeldung Zuluftkonditionierung Heizkreisregelventil aktiv*)
		bFB_AC_Cooling_Active : BOOL; (*Rückmeldung Zuluftkonditionierung Kühlkreisregelventil aktiv*)
		bT_HW_Air_Re_Active : BOOL; (*Zuluftkonditionierung Heizkreitemp. Rücklauf aktiv*)
		bT_HW_Air_Su_Active : BOOL; (*Zuluftkonditionierung Heizkreitemp. Vorlauf aktiv*)
		bCtr_ChCW_LT_Eng : BOOL; (*Regler regelt mit der Temperatur vom Motor*)
		bCtr_ECW_Eng : BOOL; (*Regler regelt mit der Temperatur vom Motor*)
		bCtr_OCW_Eng : BOOL; (*Regler regelt mit der Temperatur vom Motor*)
		bPr_EG_DeflagFastActive : BOOL; (*Visu Abgasdruck schnell aktiv*)
		bPs_aEngineLowActive : BOOL; (*visu aktiv Druckschalter nach Motor min*)
		bPs_bPumpLowActive : BOOL; (*visu aktiv Druckschalter vor Pumpe min*)
		bCircLouActive : BOOL; (*visu aktiv Umluftjalousie im Motorraum*)
		bCircLouEngActive : BOOL; (*visu aktiv Umluftjalousie von Zuluftkonditionierung*)
		bChC_LT_Stages_Active : BOOL; (*Ladekühlerstufen NT Schaltstufen aktiv*)
		rChC_LT_Stages_MaxNum : REAL; (*Anzahl Ladekühlerstufen NT gesamt*)
		bChC_HT_Stages_Active : BOOL; (*Ladekühlerstufen HT Schaltstufen aktiv*)
		rChC_HT_Stages_MaxNum : REAL; (*Anzahl Ladekühlerstufen HT gesamt*)
		bECW_Stages_Active : BOOL; (*Motorkühlwasserstufen Schaltstufen aktiv*)
		rECW_Stages_MaxNum : REAL; (*Anzahl Motorkühlwasserstufen gesamt*)
		bOCW_Stages_Active : BOOL; (*Ölkühlwasserstufen Schaltstufen aktiv*)
		rOCW_Stages_MaxNum : REAL; (*Anzahl Ölkühlwasserstufen gesamt*)
		bT_AirER5_Active : BOOL; (*Raumtemperatur 5 aktiv*)
		bT_AirER6_Active : BOOL; (*Raumtemperatur 6 aktiv*)
		bEG_Flap2_Active : BOOL; (*2. Abgasgegendruckklappe aktiv*)
		bT_EG_PrReliefVa_Active : BOOL; (*Temperatur Abgas Auslassventil aktiv*)
		bFreshAirEngAB_Active : BOOL; (*Ansaugluft A und B Seite aktiv*)
		bPr_Cool_Air_Re_Active : BOOL; (*Druckmessung im Kühlregister aktiv*)
		bPr_HW_Air_Re_Active : BOOL; (*Druckmessung im Heizregister aktiv*)
		bT_Cool_Air_Re_Active : BOOL; (*Rücklauf Temp. Messung im Kühlregister aktiv*)
		bT_Cool_Air_Su_Active : BOOL; (*Vorlauf Temp. Messung im Kühlregister aktiv*)
		bT_CircAirEng_Active : BOOL; (*Umluft Temp. Messung aktiv*)
		rTB_Cust : ARRAY[1..19]OF REAL; (*Parameter die für Tests vom Prüfstand verwendet werden können*)
		rT_PCGAfComp_HiHi : REAL; (*Limit gas temperature after prechamber gascompressor maximum*)
		rT_PCGAfCooler_HiHi : REAL; (*Limit gas temperature after cooler prechamber gascompressor maximum*)
		bPr_GT_NG_used : BOOL; (*Gas pressure natural gas used*)
		bPr_GT_PG_used : BOOL; (*Gas pressure propan gas used*)
		bPr_GT_SG_used : BOOL; (*Gas pressure special gas used*)
		bT_GT_NG_used : BOOL; (*Gas temperature natural gas used*)
		bT_GT_PG_used : BOOL; (*Gas temperature propan gas used*)
		bT_GT_SG_used : BOOL; (*Gas temperature special gas used*)
		bFlow_GT_NG_used : BOOL; (*Gas flow/counter natural gas used*)
		bFlow_GT_PG_used : BOOL; (*Gas flow/counter propan gas used*)
		bFlow_GT_SG_used : BOOL; (*Gas flow/counter special gas used*)
		bPCGC_AirCooler : BOOL; (*Prechamber gascompressor with air-cooler used*)
	END_STRUCT;
	MM2VIS_DI_struct : 	STRUCT
		stDI_Version : STRING[6]; (*DataInterface Version*)
		rT_ChCW_Re_LT : REAL; (*Temp. Ladekühlwasser Rücklauf Niedertemp. skaliert*)
		rPr_ChCW_Re_LT : REAL; (*Druck Ladekühlwasser Rücklauf Niedertemp. skaliert*)
		rT_ChCW_Su_LT : REAL; (*Temp. Ladekühlwasser Vorlauf Nidertemp. skaliert*)
		rPr_ChCW_Su_LT : REAL; (*Druck Ladekühlwasser Vorlauf Nidertemp. skaliert*)
		rT_ChCW_Re_HT : REAL; (*Temp. Ladekühlwasser Rücklauf Hochtemp. skaliert*)
		rPr_ChCW_Re_HT : REAL; (*Druck Ladekühlwasser Rücklauf Hochtemp. skaliert*)
		rT_ChCW_Su_HT : REAL; (*Temp. Ladekühlwasser Vorlauf Hochtemp. skaliert*)
		rPr_ChCW_Su_HT : REAL; (*Druck Ladekühlwasser Vorlauf Hochtemp. skaliert*)
		rT_ChCW_Re_HT_LP : REAL; (*Temp. Ladekühlwasser Rücklauf Hochtemp. Niederdruck skaliert*)
		rPr_ChCW_Re_HT_LP : REAL; (*Druck Ladekühlwasser Rücklauf Hochtemp. Niederdruck skaliert*)
		rT_ChCW_Re_HT_HP : REAL; (*Temp. Ladekühlwasser Rücklauf Hochtemp. Hochdruck skaliert*)
		rPr_ChCW_Re_HT_HP : REAL; (*Druck Ladekühlwasser Rücklauf Hochtemp. Hochdruck skaliert*)
		rT_ChCW_Su_HT_LP : REAL; (*Temp. Ladekühlwasser Vorlauf Hochtemp. Niederdruck skaliert*)
		rPr_ChCW_Su_HT_LP : REAL; (*Druck Ladekühlwasser Vorlauf Hochtemp. Niederdruck skaliert*)
		rT_ChCW_Su_HT_HP : REAL; (*Temp. Ladekühlwasser Vorlauf Hochtemp. Hochdruck skaliert*)
		rPr_ChCW_Su_HT_HP : REAL; (*Druck Ladekühlwasser Vorlauf Hochtemp. Hochdruck skaliert*)
		rT_ChCW_Re_LT_LP : REAL; (*Temp. Ladekühlwasser Rücklauf Niedertemp. Niederdruck skaliert*)
		rPr_ChCW_Re_LT_LP : REAL; (*Druck Ladekühlwasser Rücklauf Niedertemp. Niederdruck skaliert*)
		rT_ChCW_Re_LT_HP : REAL; (*Temp. Ladekühlwasser Rücklauf Niedertemp. Hochdruck skaliert*)
		rPr_ChCW_Re_LT_HP : REAL; (*Druck Ladekühlwasser Rücklauf Niedertemp. Hochdruck skaliert*)
		rT_ChCW_Su_LT_LP : REAL; (*Temp. Ladekühlwasser Vorlauf Niedertemp. Niederdruck skaliert*)
		rPr_ChCW_Su_LT_LP : REAL; (*Druck Ladekühlwasser Vorlauf Niedertemp. Niederdruck skaliert*)
		rT_ChCW_Su_LT_HP : REAL; (*Temp. Ladekühlwasser Vorlauf Niedertemp. Hochdruck skaliert*)
		rPr_ChCW_Su_LT_HP : REAL; (*Druck Ladekühlwasser Vorlauf Niedertemp. Hochdruck skaliert*)
		rT_OCW_Re : REAL; (*Temp. Ölkühlwasser Rücklauf skaliert*)
		rPr_OCW_Re : REAL; (*Druck Ölkühlwasser Rücklauf skaliert*)
		rT_OCW_Su : REAL; (*Temp. Ölkühlwasser Vorlauf skaliert*)
		rPr_OCW_Su : REAL; (*Druck Ölkühlwasser Vorlauf skaliert*)
		rT_ECW_Re : REAL; (*Temp. Motorkühlwasser Rücklauf skaliert*)
		rPr_ECW_Re : REAL; (*Druck Motorkühlwasser Rücklauf skaliert*)
		rT_ECW_Su : REAL; (*Temp. Motorkühlwasser Vorlauf skaliert*)
		rPr_ECW_Su : REAL; (*Druck Motorkühlwasser Vorlauf skaliert*)
		rVol_ChCW_Re_LT : REAL; (*Durchfluss Ladekühlwasser Rücklauf Niedertemp. scaliert*)
		rVol_ChCW_Su_LT : REAL; (*Durchfluss Ladekühlwasser Vorlauf Niedertemp. scaliert*)
		rVol_ChCW_Re_HT : REAL; (*Durchfluss Ladekühlwasser Rücklauf Hochtemp. scaliert*)
		rVol_ChCW_Su_HT : REAL; (*Durchfluss Ladekühlwasser Vorlauf Hochtemp. scaliert*)
		rVol_ChCW_Re_HT_LP : REAL; (*Durchfluss Ladekühlwasser Rücklauf Hochtemp. Niederdruck scaliert*)
		rVol_ChCW_Su_HT_LP : REAL; (*Durchfluss Ladekühlwasser Vorlauf Hochtemp. Niederdruck scaliert*)
		rVol_ChCW_Re_HT_HP : REAL; (*Durchfluss Ladekühlwasser Rücklauf Hochtemp. Hochdruck scaliert*)
		rVol_ChCW_Su_HT_HP : REAL; (*Durchfluss Ladekühlwasser Vorlauf Hochtemp. Hochdruck scaliert*)
		rVol_ChCW_Re_LT_LP : REAL; (*Durchfluss Ladekühlwasser Rücklauf Niedertemp. Niederdruck scaliert*)
		rVol_ChCW_Su_LT_LP : REAL; (*Durchfluss Ladekühlwasser Vorlauf Niedertemp. Niederdruck scaliert*)
		rVol_ChCW_Re_LT_HP : REAL; (*Durchfluss Ladekühlwasser Rücklauf Niedertemp. Hochdruck scaliert*)
		rVol_ChCW_Su_LT_HP : REAL; (*Durchfluss Ladekühlwasser Vorlauf Niedertemp. Hochdruck scaliert*)
		rVol_ECW_Re : REAL; (*Durchfluss Motorkühlwasser Rücklauf scaliert*)
		rVol_ECW_Su : REAL; (*Durchfluss Motorkühlwasser Vorlauf scaliert*)
		rVol_OCW_Re : REAL; (*Durchfluss Ölkühlwasser Rücklauf skaliert*)
		rVol_OCW_Su : REAL; (*Durchfluss Ölkühlwasser Vorlauf skaliert*)
		rCtr_ChCW_LT_In_X : REAL; (*Regler In X für Anzeige auf Visu*)
		tCtr_ChCW_LT_Out : _tGeACtrOut; (*charge cooler*)
		rCtr_ChCW_HT_In_X : REAL; (*Regler In X für Anzeige auf Visu*)
		tCtr_ChCW_HT_Out : _tGeACtrOut; (*charge cooler*)
		rCtr_ChCW_HT_LP_In_X : REAL; (*Regler In X für Anzeige auf Visu*)
		tCtr_ChCW_HT_LP_Out : _tGeACtrOut; (*charge cooler*)
		rCtr_ChCW_HT_HP_In_X : REAL; (*Regler In X für Anzeige auf Visu*)
		tCtr_ChCW_HT_HP_Out : _tGeACtrOut; (*charge cooler*)
		rCtr_ChCW_LT_LP_In_X : REAL; (*Regler In X für Anzeige auf Visu*)
		tCtr_ChCW_LT_LP_Out : _tGeACtrOut; (*charge cooler*)
		rCtr_ChCW_LT_HP_In_X : REAL; (*Regler In X für Anzeige auf Visu*)
		tCtr_ChCW_LT_HP_Out : _tGeACtrOut; (*charge cooler*)
		rCtr_ECW_In_X : REAL; (*Regler In X für Anzeige auf Visu*)
		tCtr_ECW_Out : _tGeACtrOut; (*engine cooling water cooler*)
		rCtr_OCW_In_X : REAL; (*Regler In X für Anzeige auf Visu*)
		tCtr_OCW_Out : _tGeACtrOut; (*oil cooling water cooler*)
		rT_ChCW_LT_IC_Re : REAL; (*Temp Laderkühlwasser Niedertemp Zwischenkreis Rücklauf skaliert*)
		rPr_ChCW_LT_IC_Re : REAL; (*Druck Laderkühlwasser Niedertemp Zwischenkreis Rücklauf skaliert*)
		rT_ChCW_HT_IC_Re : REAL; (*Temp Laderkühlwasser Hochtemp Zwischenkreis Rücklauf skaliert*)
		rPr_ChCW_HT_IC_Re : REAL; (*Druck Laderkühlwasser Hochtemp Zwischenkreis Rücklauf skaliert*)
		rT_ChCW_LT_LP_IC_Re : REAL; (*Temp Laderkühlwasser Niedertemp Niederdruck Zwischenkreis Rücklauf skaliert*)
		rPr_ChCW_LT_LP_IC_Re : REAL; (*Druck Laderkühlwasser Niedertemp Niederdruck Zwischenkreis Rücklauf skaliert*)
		rT_ChCW_LT_HP_IC_Re : REAL; (*Temp Laderkühlwasser Niedertemp Hochdruck Zwischenkreis Rücklauf skaliert*)
		rPr_ChCW_LT_HP_IC_Re : REAL; (*Druck Laderkühlwasser Niedertemp Hochdruck Zwischenkreis Rücklauf skaliert*)
		rT_ChCW_HT_LP_IC_Re : REAL; (*Temp Laderkühlwasser Hochtemp Niederdruck Zwischenkreis Rücklauf skaliert*)
		rPr_ChCW_HT_LP_IC_Re : REAL; (*Druck Laderkühlwasser Hochtemp Niederdruck Zwischenkreis Rücklauf skaliert*)
		rT_ChCW_HT_HP_IC_Re : REAL; (*Temp Laderkühlwasser Hochdruck Hochtemp Zwischenkreis Rücklauf skaliert*)
		rPr_ChCW_HT_HP_IC_Re : REAL; (*Druck Laderkühlwasser Hochtemp Hochdruck Zwischenkreis Rücklauf skaliert*)
		rT_ECW_IC_Re : REAL; (*Temp Motorkühlwasser Zwischenkreis Rücklauf skaliert*)
		rPr_ECW_IC_Re : REAL; (*Druck Motorkühlwasser Zwischenkreis Rücklauf skaliert*)
		rT_OCW_IC_Re : REAL; (*Temp Ölühlwasser Zwischenkreis Rücklauf skaliert*)
		rPr_OCW_IC_Re : REAL; (*Druck Ölühlwasser Zwischenkreis Rücklauf skaliert*)
		rT_ChCW_LT_IC_Su : REAL; (*Temp Laderkühlwasser Niedertemp Zwischenkreis Vorlauf skaliert*)
		rPr_ChCW_LT_IC_Su : REAL; (*Druck Laderkühlwasser Niedertemp Zwischenkreis Vorlauf skaliert*)
		rT_ChCW_HT_IC_Su : REAL; (*Temp Laderkühlwasser Hochtemp Zwischenkreis Vorlauf skaliert*)
		rPr_ChCW_HT_IC_Su : REAL; (*Druck Laderkühlwasser Hochtemp Zwischenkreis Vorlauf skaliert*)
		rT_ChCW_LT_LP_IC_Su : REAL; (*Temp Laderkühlwasser Niedertemp Niederdruck Zwischenkreis Vorlauf skaliert*)
		rPr_ChCW_LT_LP_IC_Su : REAL; (*Druck Laderkühlwasser Niedertemp Niederdruck Zwischenkreis Vorlauf skaliert*)
		rT_ChCW_LT_HP_IC_Su : REAL; (*Temp Laderkühlwasser Niedertemp Hochdruck Zwischenkreis Vorlauf skaliert*)
		rPr_ChCW_LT_HP_IC_Su : REAL; (*Druck Laderkühlwasser Niedertemp Hochdruck Zwischenkreis Vorlauf skaliert*)
		rT_ChCW_HT_LP_IC_Su : REAL; (*Temp Laderkühlwasser Hochtemp Niederdruck Zwischenkreis Vorlauf skaliert*)
		rPr_ChCW_HT_LP_IC_Su : REAL; (*Druck Laderkühlwasser Hochtemp Niederdruck Zwischenkreis Vorlauf skaliert*)
		rT_ChCW_HT_HP_IC_Su : REAL; (*Temp Laderkühlwasser Hochdruck Hochtemp Zwischenkreis Vorlauf skaliert*)
		rPr_ChCW_HT_HP_IC_Su : REAL; (*Druck Laderkühlwasser Hochtemp Hochdruck Zwischenkreis Vorlauf skaliert*)
		rT_ECW_IC_Su : REAL; (*Temp Motorkühlwasser Zwischenkreis Vorlauf skaliert*)
		rPr_ECW_IC_Su : REAL; (*Druck Motorkühlwasser Zwischenkreis Vorlauf skaliert*)
		rT_OCW_IC_Su : REAL; (*Temp Ölkühlwasser Zwischenkreis Vorlauf skaliert*)
		rPr_OCW_IC_Su : REAL; (*Druck Ölkühlwasser Zwischenkreis Vorlauf skaliert*)
		rT_Cooler_ChCW_LT_Re_1 : REAL; (*Temp Ladekühler 1 NT Rücklauf skaliert*)
		rT_Cooler_ChCW_HT_Re_1 : REAL; (*Temp Ladekühler 1 HT Rücklauf skaliert*)
		rT_Cooler_ChCW_LT_LP_Re_1 : REAL; (*Temp Ladekühler 1 NT ND Rücklauf skaliert*)
		rT_Cooler_ChCW_LT_HP_Re_1 : REAL; (*Temp Ladekühler 1 NT HD Rücklauf skaliert*)
		rT_Cooler_ChCW_HT_LP_Re_1 : REAL; (*Temp Ladekühler 1 HT ND Rücklauf skaliert*)
		rT_Cooler_ChCW_HT_HP_Re_1 : REAL; (*Temp Ladekühler 1 HT HD Rücklauf skaliert*)
		rT_Cooler_ChCW_LT_Re_2 : REAL; (*Temp Ladekühler 2 NT Rücklauf skaliert*)
		rT_Cooler_ChCW_HT_Re_2 : REAL; (*Temp Ladekühler 2 HT Rücklauf skaliert*)
		rT_Cooler_ChCW_LT_LP_Re_2 : REAL; (*Temp Ladekühler 2 NT ND Rücklauf skaliert*)
		rT_Cooler_ChCW_LT_HP_Re_2 : REAL; (*Temp Ladekühler 2 NT HD Rücklauf skaliert*)
		rT_Cooler_ChCW_HT_LP_Re_2 : REAL; (*Temp Ladekühler 2 HT ND Rücklauf skaliert*)
		rT_Cooler_ChCW_HT_HP_Re_2 : REAL; (*Temp Ladekühler 2 HT HD Rücklauf skaliert*)
		rPr_Cooler_ChCW_LT_Re_1 : REAL; (*Druck Ladekühler 1 NT Rücklauf skaliert*)
		rPr_Cooler_ChCW_HT_Re_1 : REAL; (*Druck Ladekühler 1 HT Rücklauf skaliert*)
		rPr_Cooler_ChCW_LT_LP_Re_1 : REAL; (*Druck Ladekühler 1 NT ND Rücklauf skaliert*)
		rPr_Cooler_ChCW_LT_HP_Re_1 : REAL; (*Druck Ladekühler 1 NT HD Rücklauf skaliert*)
		rPr_Cooler_ChCW_HT_LP_Re_1 : REAL; (*Druck Ladekühler 1 HT ND Rücklauf skaliert*)
		rPr_Cooler_ChCW_HT_HP_Re_1 : REAL; (*Druck Ladekühler 1 HT HD Rücklauf skaliert*)
		rPr_Cooler_ChCW_LT_Re_2 : REAL; (*Druck Ladekühler 2 NT Rücklauf skaliert*)
		rPr_Cooler_ChCW_HT_Re_2 : REAL; (*Druck Ladekühler 2 HT Rücklauf skaliert*)
		rPr_Cooler_ChCW_LT_LP_Re_2 : REAL; (*Druck Ladekühler 2 NT ND Rücklauf skaliert*)
		rPr_Cooler_ChCW_LT_HP_Re_2 : REAL; (*Druck Ladekühler 2 NT HD Rücklauf skaliert*)
		rPr_Cooler_ChCW_HT_LP_Re_2 : REAL; (*Druck Ladekühler 2 HT ND Rücklauf skaliert*)
		rPr_Cooler_ChCW_HT_HP_Re_2 : REAL; (*Druck Ladekühler 2 HT HD Rücklauf skaliert*)
		rT_Cooler_ChCW_LT_Su_1 : REAL; (*Temp Ladekühler 1 NT Vorlauf skaliert*)
		rT_Cooler_ChCW_HT_Su_1 : REAL; (*Temp Ladekühler 1 HT Vorlauf skaliert*)
		rT_Cooler_ChCW_LT_LP_Su_1 : REAL; (*Temp Ladekühler 1 NT ND Vorlauf skaliert*)
		rT_Cooler_ChCW_LT_HP_Su_1 : REAL; (*Temp Ladekühler 1 NT HD Vorlauf skaliert*)
		rT_Cooler_ChCW_HT_LP_Su_1 : REAL; (*Temp Ladekühler 1 HT ND Vorlauf skaliert*)
		rT_Cooler_ChCW_HT_HP_Su_1 : REAL; (*Temp Ladekühler 1 HT HD Vorlauf skaliert*)
		rT_Cooler_ChCW_LT_Su_2 : REAL; (*Temp Ladekühler 2 NT Vorlauf skaliert*)
		rT_Cooler_ChCW_HT_Su_2 : REAL; (*Temp Ladekühler 2 HT Vorlauf skaliert*)
		rT_Cooler_ChCW_LT_LP_Su_2 : REAL; (*Temp Ladekühler 2 NT ND Vorlauf skaliert*)
		rT_Cooler_ChCW_LT_HP_Su_2 : REAL; (*Temp Ladekühler 2 NT HD Vorlauf skaliert*)
		rT_Cooler_ChCW_HT_LP_Su_2 : REAL; (*Temp Ladekühler 2 HT ND Vorlauf skaliert*)
		rT_Cooler_ChCW_HT_HP_Su_2 : REAL; (*Temp Ladekühler 2 HT HD Vorlauf skaliert*)
		rPr_Cooler_ChCW_LT_Su_1 : REAL; (*Druck Ladekühler 1 NT Vorlauf skaliert*)
		rPr_Cooler_ChCW_HT_Su_1 : REAL; (*Druck Ladekühler 1 HT Vorlauf skaliert*)
		rPr_Cooler_ChCW_LT_LP_Su_1 : REAL; (*Druck Ladekühler 1 NT ND Vorlauf skaliert*)
		rPr_Cooler_ChCW_LT_HP_Su_1 : REAL; (*Druck Ladekühler 1 NT HD Vorlauf skaliert*)
		rPr_Cooler_ChCW_HT_LP_Su_1 : REAL; (*Druck Ladekühler 1 HT ND Vorlauf skaliert*)
		rPr_Cooler_ChCW_HT_HP_Su_1 : REAL; (*Druck Ladekühler 1 HT HD Vorlauf skaliert*)
		rPr_Cooler_ChCW_LT_Su_2 : REAL; (*Druck Ladekühler 2 NT Vorlauf skaliert*)
		rPr_Cooler_ChCW_HT_Su_2 : REAL; (*Druck Ladekühler 2 HT Vorlauf skaliert*)
		rPr_Cooler_ChCW_LT_LP_Su_2 : REAL; (*Druck Ladekühler 2 NT ND Vorlauf skaliert*)
		rPr_Cooler_ChCW_LT_HP_Su_2 : REAL; (*Druck Ladekühler 2 NT HD Vorlauf skaliert*)
		rPr_Cooler_ChCW_HT_LP_Su_2 : REAL; (*Druck Ladekühler 2 HT ND Vorlauf skaliert*)
		rPr_Cooler_ChCW_HT_HP_Su_2 : REAL; (*Druck Ladekühler 2 HT HD Vorlauf skaliert*)
		rT_Cooler_ECW_Re_1 : REAL; (*Temp Motorkühlwasserkühler 1 Rücklauf skaliert*)
		rT_Cooler_ECW_Re_2 : REAL; (*Temp Motorkühlwasserkühler 2 Rücklauf skaliert*)
		rT_Cooler_OCW_Re_1 : REAL; (*Temp Ölkühlwasserkühler 1 Rücklauf skaliert*)
		rT_Cooler_OCW_Re_2 : REAL; (*Temp Ölkühlwasserkühler 2 Rücklauf skaliert*)
		rT_Cooler_ECW_Su_1 : REAL; (*Temp Motorkühlwasserkühler 1 Vorlauf skaliert*)
		rT_Cooler_ECW_Su_2 : REAL; (*Temp Motorkühlwasserkühler 2 Vorlauf skaliert*)
		rT_Cooler_OCW_Su_1 : REAL; (*Temp Ölkühlwasserkühler 1 Vorlauf skaliert*)
		rT_Cooler_OCW_Su_2 : REAL; (*Temp Ölkühlwasserkühler 2 Vorlauf skaliert*)
		rT_ChCW_LT_bCV : REAL; (*Temp Ladekühlwasser NT vor Regelventil skaliert*)
		rT_RW_HE_Re : REAL; (*Temp Rohwasser Wärmetauscher Rücklauf skaliert*)
		rT_RW_HE_Su : REAL; (*Temp Rohwasser Wärmetauscher Vorlauf skaliert*)
		rT_RW_Re : REAL; (*Temp Rohwasser NT Rücklauf skaliert*)
		rT_RW_Su : REAL; (*Temp Rohwasser NT Vorlauf skaliert*)
		rT_RW_LT_Re_1 : REAL; (*Temp Rohwasser NT 1 Rücklauf skaliert*)
		rT_RW_LT_Re_2 : REAL; (*Temp Rohwasser NT 2 Rücklauf skaliert*)
		rT_RW_HT_Re_1 : REAL; (*Temp Rohwasser HT 1 Rücklauf skaliert*)
		rT_RW_HT_Re_2 : REAL; (*Temp Rohwasser HT 2 Rücklauf skaliert*)
		rT_RW_ECW_Re_1 : REAL; (*Temp Rohwasser MKW 1 Rücklauf skaliert*)
		rT_RW_ECW_Re_2 : REAL; (*Temp Rohwasser MKW 2 Rücklauf skaliert*)
		rT_RW_OCW_Re_1 : REAL; (*Temp Rohwasser OKW 1 Rücklauf skaliert*)
		rT_RW_OCW_Re_2 : REAL; (*Temp Rohwasser OKW 2 Rücklauf skaliert*)
		rPr_Cooler_ECW_Re_1 : REAL; (*Temp Motorkühlwasserkühler 1 Rücklauf skaliert*)
		rPr_Cooler_ECW_Re_2 : REAL; (*Temp Motorkühlwasserkühler 2 Rücklauf skaliert*)
		rPr_Cooler_OCW_Re_1 : REAL; (*Temp Ölkühlwasserkühler 1 Rücklauf skaliert*)
		rPr_Cooler_OCW_Re_2 : REAL; (*Temp Ölkühlwasserkühler 2 Rücklauf skaliert*)
		rPr_Cooler_ECW_Su_1 : REAL; (*Temp Motorkühlwasserkühler 1 Vorlauf skaliert*)
		rPr_Cooler_ECW_Su_2 : REAL; (*Temp Motorkühlwasserkühler 2 Vorlauf skaliert*)
		rPr_Cooler_OCW_Su_1 : REAL; (*Temp Ölkühlwasserkühler 1 Vorlauf skaliert*)
		rPr_Cooler_OCW_Su_2 : REAL; (*Temp Ölkühlwasserkühler 2 Vorlauf skaliert*)
		rPr_RW_HE_Re : REAL; (*Druck Rohwasser Wärmetauscher Rücklauf skaliert*)
		rPr_RW_HE_Su : REAL; (*Druck Rohwasser Wärmetauscher Vorlauf skaliert*)
		rPr_RW_LT_Re_1 : REAL; (*Druck Rohwasser NT Rücklauf skaliert*)
		rPr_RW_LT_Su_1 : REAL; (*Druck Rohwasser NT Vorlauf skaliert*)
		rPr_RW_HT_Re_1 : REAL; (*Druck Rohwarser HT Rücklauf skaliert*)
		rPr_RW_HT_Su_1 : REAL; (*Druck Rohwasser HT Vorlauf skaliert*)
		rPr_RW_LT_Re_2 : REAL; (*Druck Rohwasser NT Rücklauf skaliert*)
		rPr_RW_LT_Su_2 : REAL; (*Druck Rohwasser NT Vorlauf skaliert*)
		rPr_RW_HT_Re_2 : REAL; (*Druck Rohwarser HT Rücklauf skaliert*)
		rPr_RW_HT_Su_2 : REAL; (*Druck Rohwasser HT Vorlauf skaliert*)
		rPr_RW_ECW_Re_1 : REAL; (*Druck Rohwasser Motorkühlwasser Rücklauf skaliert*)
		rPr_RW_ECW_Su_1 : REAL; (*Druck Rohwasser Motorkühlwasser Vorlauf skaliert*)
		rPr_RW_OCW_Re_1 : REAL; (*Druck Rohwasser Ölkühlwasser Rücklauf skaliert*)
		rPr_RW_OCW_Su_1 : REAL; (*Druck Rohwasser Ölkühlwasser Vorlauf skaliert*)
		rPr_RW_ECW_Re_2 : REAL; (*Druck Rohwasser Motorkühlwasser Rücklauf skaliert*)
		rPr_RW_ECW_Su_2 : REAL; (*Druck Rohwasser Motorkühlwasser Vorlauf skaliert*)
		rPr_RW_OCW_Re_2 : REAL; (*Druck Rohwasser Ölkühlwasser Rücklauf skaliert*)
		rPr_RW_OCW_Su_2 : REAL; (*Druck Rohwasser Ölkühlwasser Vorlauf skaliert*)
		rCtr_ChCW_LT_Set : REAL; (*Regler Ladekühlwasser Niedertemp. skaliert*)
		rCtr_ChCW_HT_Set : REAL; (*Regler Ladekühlwasser Hochtemp. skaliert*)
		rCtr_ChCW_HT_LP_Set : REAL; (*Regler Ladekühlwasser Hochtemp. Niederdruck skaliert*)
		rCtr_ChCW_HT_HP_Set : REAL; (*Regler Ladekühlwasser Hochtemp. Hochdruck skaliert*)
		rCtr_ChCW_LT_LP_Set : REAL; (*Regler Ladekühlwasser Niedertemp. Niederdruck skaliert*)
		rCtr_ChCW_LT_HP_Set : REAL; (*Regler Ladekühlwasser Niedertemp. Hochdruck skaliert*)
		rCtr_OCW_Set : REAL; (*Regler Kühlkreis Öltemp. skaliert*)
		rCtr_RW_CV : REAL; (*Kühlkreis Regelventil Rohwassser skaliert*)
		rCtr_RW_HE : REAL; (*Kühlkreis Regelventil Rohwasser Wärmetauscher skaliert*)
		rFC_ChCW_LT_Pump : REAL; (*FU Ladekühwasser Niedertemp. Pumpe skaliert*)
		rFC_ChCW_HT_Pump : REAL; (*FU Ladekühwasser Hochtemp. Pumpe skaliert*)
		rFC_ChCW_LT_LP_Pump : REAL; (*FU Ladekühwasser Niedertemp. Niederdruck Pumpe skaliert*)
		rFC_ChCW_LT_HP_Pump : REAL; (*FU Ladekühwasser Niedertemp. Hochdruck Pumpe skaliert*)
		rFC_ChCW_HT_LP_Pump : REAL; (*FU Ladekühwasser Hochtemp. Niederdruck Pumpe skaliert*)
		rFC_ChCW_HT_HP_Pump : REAL; (*FU Ladekühwasser Hochtemp. Hochdruck Pumpe skaliert*)
		rFC_ECW_Pump : REAL; (*FU Motorkühlwasser Pumpe skaliert*)
		rFC_OCW_Pump : REAL; (*FU Ölkühlwasser Pumpe skaliert*)
		rFC_ChCW_LT_Cooler_1 : REAL; (*FU Ladekühwasser Niedertemp. Kühler skaliert*)
		rFC_ChCW_HT_Cooler_1 : REAL; (*FU Ladekühwasser Hochtemp. Kühler skaliert*)
		rFC_ChCW_LT_LP_Cooler_1 : REAL; (*FU Ladekühwasser Niedertemp. Niederdruck Kühler skaliert*)
		rFC_ChCW_LT_HP_Cooler_1 : REAL; (*FU Ladekühwasser Niedertemp. Hochdruck Kühler skaliert*)
		rFC_ChCW_HT_LP_Cooler_1 : REAL; (*FU Ladekühwasser Hochtemp. Niederdruck Kühler skaliert*)
		rFC_ChCW_HT_HP_Cooler_1 : REAL; (*FU Ladekühwasser Hochtemp. Hochdruck Kühler skaliert*)
		rFC_ChCW_LT_Cooler_2 : REAL; (*FU Ladekühwasser Niedertemp. Kühler skaliert*)
		rFC_ChCW_HT_Cooler_2 : REAL; (*FU Ladekühwasser Hochtemp. Kühler skaliert*)
		rFC_ChCW_LT_LP_Cooler_2 : REAL; (*FU Ladekühwasser Niedertemp. Niederdruck Kühler skaliert*)
		rFC_ChCW_LT_HP_Cooler_2 : REAL; (*FU Ladekühwasser Niedertemp. Hochdruck Kühler skaliert*)
		rFC_ChCW_HT_LP_Cooler_2 : REAL; (*FU Ladekühwasser Hochtemp. Niederdruck Kühler skaliert*)
		rFC_ChCW_HT_HP_Cooler_2 : REAL; (*FU Ladekühwasser Hochtemp. Hochdruck Kühler skaliert*)
		rFC_ECW_Cooler_1 : REAL; (*FU Motorkühlwasser Kühler skaliert*)
		rFC_OCW_Cooler_1 : REAL; (*FU Ölkühlwasser Kühler skaliert*)
		rFC_ECW_Cooler_2 : REAL; (*FU Motorkühlwasser Kühler skaliert*)
		rFC_OCW_Cooler_2 : REAL; (*FU Ölkühlwasser Kühler skaliert*)
		bDem_Cooler_ChCW_LT_1 : BOOL; (*visu aktiv Anforderung Kühler Ladekühlwasser NT*)
		bDem_Cooler_ChCW_LT_2 : BOOL; (*visu aktiv Anforderung Kühler Ladekühlwasser NT*)
		bDem_Cooler_ChCW_HT_1 : BOOL; (*visu aktiv Anforderung Kühler Ladekühlwasser HT*)
		bDem_Cooler_ChCW_HT_2 : BOOL; (*visu aktiv Anforderung Kühler Ladekühlwasser HT*)
		bDem_Cooler_ChCW_LT_LP_1 : BOOL; (*visu aktiv Anforderung Kühler Ladekühlwasser NT ND*)
		bDem_Cooler_ChCW_LT_LP_2 : BOOL; (*visu aktiv Anforderung Kühler Ladekühlwasser NT ND*)
		bDem_Cooler_ChCW_LT_HP_1 : BOOL; (*visu aktiv Anforderung Kühler Ladekühlwasser NT HD*)
		bDem_Cooler_ChCW_LT_HP_2 : BOOL; (*visu aktiv Anforderung Kühler Ladekühlwasser NT HD*)
		bDem_Cooler_ChCW_HT_LP_1 : BOOL; (*visu aktiv Anforderung Kühler Ladekühlwasser HT ND*)
		bDem_Cooler_ChCW_HT_LP_2 : BOOL; (*visu aktiv Anforderung Kühler Ladekühlwasser HT ND*)
		bDem_Cooler_ChCW_HT_HP_1 : BOOL; (*visu aktiv Anforderung Kühler Ladekühlwasser HT HD*)
		bDem_Cooler_ChCW_HT_HP_2 : BOOL; (*visu aktiv Anforderung Kühler Ladekühlwasser HT HD*)
		bDem_Cooler_ECW_1 : BOOL; (*visu aktiv Anforderung Kühler Motorkühlwasser*)
		bDem_Cooler_ECW_2 : BOOL; (*visu aktiv Anforderung Kühler Motorkühlwasser*)
		bDem_Cooler_OCW_1 : BOOL; (*visu aktiv Anforderung Kühler Ölkühlwasser*)
		bDem_Cooler_OCW_2 : BOOL; (*visu aktiv Anforderung Kühler Ölkühlwasser*)
		bDem_ChCW_LT_Pump : BOOL; (*visu aktiv Anforderung Ladekühlwasser NT Pumpe*)
		bDem_ChCW_HT_Pump : BOOL; (*visu aktiv Anforderung Ladekühlwasser HT Pumpe*)
		bDem_ChCW_LT_LP_Pump : BOOL; (*visu aktiv Anforderung Ladekühlwasser NT ND Pumpe*)
		bDem_ChCW_LT_HP_Pump : BOOL; (*visu aktiv Anforderung Ladekühlwasser NT HD Pumpe*)
		bDem_ChCW_HT_LP_Pump : BOOL; (*visu aktiv Anforderung Ladekühlwasser HT ND Pumpe*)
		bDem_ChCW_HT_HP_Pump : BOOL; (*visu aktiv Anforderung Ladekühlwasser HT HD Pumpe*)
		bDem_ECW_Pump : BOOL; (*visu aktiv Anforderung Motorkühlwasser Pumpe*)
		bDem_OCW_Pump : BOOL; (*visu aktiv Anforderung Ölkühlwasser Pumpe*)
		bPs_ChCW_LT_bEngine_Hi : BOOL; (*Druckschalter Ladekühwasser LT vor Motor ausgelöst*)
		bPs_ChCW_HT_bEngine_Hi : BOOL; (*Druckschalter Ladekühwasser HT vor Motor ausgelöst*)
		bPs_ChCW_LT_LP_bEngine_Hi : BOOL; (*Druckschalter Ladekühwasser NT ND vor Motor ausgelöst*)
		bPs_ChCW_LT_HP_bEngine_Hi : BOOL; (*Druckschalter Ladekühwasser NT HD vor Motor ausgelöst*)
		bPs_ChCW_HT_LP_bEngine_Hi : BOOL; (*Druckschalter Ladekühwasser HT ND vor Motor ausgelöst*)
		bPs_ChCW_HT_HP_bEngine_Hi : BOOL; (*Druckschalter Ladekühwasser HT HD vor Motor ausgelöst*)
		bPs_ECW_bEngine_Hi : BOOL; (*Druckschalter Motorkühlwasser vor Motor ausgelöst*)
		bPs_OCW_bEngine_Hi : BOOL; (*Druckschalter Ölkühlwasser vor Motor ausgelöst*)
		bPs_ChCW_LT_aEngine_Low : BOOL; (*Druckschalter Ladekühwasser NT nach Motor ausgelöst*)
		bPs_ChCW_HT_aEngine_Low : BOOL; (*Druckschalter Ladekühwasser HT nach Motor ausgelöst*)
		bPs_ChCW_LT_LP_aEngine_Low : BOOL; (*Druckschalter Ladekühwasser NT ND nach Motor ausgelöst*)
		bPs_ChCW_LT_HP_aEngine_Low : BOOL; (*Druckschalter Ladekühwasser NT HD nach Motor ausgelöst*)
		bPs_ChCW_HT_LP_aEngine_Low : BOOL; (*Druckschalter Ladekühwasser HT ND nach Motor ausgelöst*)
		bPs_ChCW_HT_HP_aEngine_Low : BOOL; (*Druckschalter Ladekühwasser HT HD nach Motor ausgelöst*)
		bPs_ECW_aEngine_Low : BOOL; (*Druckschalter Motorkühlwasser nach Motor ausgelöst*)
		bPs_OCW_aEngine_Low : BOOL; (*Druckschalter Ölkühlwasser nach Motor ausgelöst*)
		bPs_ChCW_LT_bPump_Low : BOOL; (*Druckschalter Ladekühwasser NT vor Pumpe ausgelöst*)
		bPs_ChCW_HT_bPump_Low : BOOL; (*Druckschalter Ladekühwasser HT vor Pumpe ausgelöst*)
		bPs_ChCW_LT_LP_bPump_Low : BOOL; (*Druckschalter Ladekühwasser NT ND vor Pumpe ausgelöst*)
		bPs_ChCW_LT_HP_bPump_Low : BOOL; (*Druckschalter Ladekühwasser NT HD vor Pumpe ausgelöst*)
		bPs_ChCW_HT_LP_bPump_Low : BOOL; (*Druckschalter Ladekühwasser HT ND vor Pumpe ausgelöst*)
		bPs_ChCW_HT_HP_bPump_Low : BOOL; (*Druckschalter Ladekühwasser HT HD vor Pumpe ausgelöst*)
		bPs_ECW_bPump_Low : BOOL; (*Druckschalter Motorkühlwasser vor Pumpe ausgelöst*)
		bPs_OCW_bPump_Low : BOOL; (*Druckschalter Ölkühlwasser vor Pumpe ausgelöst*)
		bPs_RW_Low : BOOL; (*Druckschalter Rohwasser zu nieder*)
		bTs_ChCW_LT_bEngine_Hi : BOOL; (*Temperaturschalter Ladekühwasser NT vor Motor ausgelöst*)
		bTs_ChCW_HT_bEngine_Hi : BOOL; (*Temperaturschalter Ladekühwasser HT vor Motor ausgelöst*)
		bTs_ChCW_LT_LP_bEngine_Hi : BOOL; (*Temperaturschalter Ladekühwasser NT ND vor Motor ausgelöst*)
		bTs_ChCW_LT_HP_bEngine_Hi : BOOL; (*Temperaturschalter Ladekühwasser NT HD vor Motor ausgelöst*)
		bTs_ChCW_HT_LP_bEngine_Hi : BOOL; (*Temperaturschalter Ladekühwasser HT ND vor Motor ausgelöst*)
		bTs_ChCW_HT_HP_bEngine_Hi : BOOL; (*Temperaturschalter Ladekühwasser HT HD vor Motor ausgelöst*)
		bTs_ECW_bEngine_Hi : BOOL; (*Temperaturschalter Motorkühlwasser vor Motor ausgelöst*)
		bTs_OCW_bEngine_Hi : BOOL; (*Temperaturschalter Ölkühlwasser vor Motor ausgelöst*)
		bTs_RW_Hi : BOOL; (*Temperaturschalter Rohwasser zu hoch*)
		bCooler_ChCW_LT_1_Op : BOOL; (*Status Kühler Ladekühlwasser NT in Betrieb*)
		bCooler_ChCW_LT_2_Op : BOOL; (*Status Kühler Ladekühlwasser NT in Betrieb*)
		bCooler_ChCW_HT_1_Op : BOOL; (*Status Kühler Ladekühlwasser HT in Betrieb*)
		bCooler_ChCW_HT_2_Op : BOOL; (*Status Kühler Ladekühlwasser HT in Betrieb*)
		bCooler_ChCW_LT_LP_1_Op : BOOL; (*Status Kühler Ladekühlwasser NT ND in Betrieb*)
		bCooler_ChCW_LT_LP_2_Op : BOOL; (*Status Kühler Ladekühlwasser NT ND in Betrieb*)
		bCooler_ChCW_LT_HP_1_Op : BOOL; (*Status Kühler Ladekühlwasser NT ND in Betrieb*)
		bCooler_ChCW_LT_HP_2_Op : BOOL; (*Status Kühler Ladekühlwasser NT HD in Betrieb*)
		bCooler_ChCW_HT_LP_1_Op : BOOL; (*Status Kühler Ladekühlwasser HT ND in Betrieb*)
		bCooler_ChCW_HT_LP_2_Op : BOOL; (*Status Kühler Ladekühlwasser HT ND in Betrieb*)
		bCooler_ChCW_HT_HP_1_Op : BOOL; (*Status Kühler Ladekühlwasser HT HD in Betrieb*)
		bCooler_ChCW_HT_HP_2_Op : BOOL; (*Status Kühler Ladekühlwasser HT HD in Betrieb*)
		bCooler_ECW_1_Op : BOOL; (*Status Kühler Motorkühlwasser in Betrieb*)
		bCooler_ECW_2_Op : BOOL; (*Status Kühler Motorkühlwasser in Betrieb*)
		bCooler_OCW_1_Op : BOOL; (*Status Kühler Ölkühlwasser in Betrieb*)
		bCooler_OCW_2_Op : BOOL; (*Status Kühler Ölkühlwasser in Betrieb*)
		rT_ChCW_LT_LP_bCV : REAL; (*Temp Ladekühlwasser NT ND vor Regelventil skaliert*)
		rT_ChCW_LT_HP_bCV : REAL; (*Temp Ladekühlwasser NT HD vor Regelventil skaliert*)
		rT_ChCW_HT_bCV : REAL; (*Temp Ladekühlwasser HT vor Regelventil skaliert*)
		rT_ChCW_HT_LP_bCV : REAL; (*Temp Ladekühlwasser HT ND vor Regelventil skaliert*)
		rT_ChCW_HT_HP_bCV : REAL; (*Temp Ladekühlwasser HT HD vor Regelventil skaliert*)
		rT_ECW_bCV : REAL; (*Temp Motorkühlwasser vor Regelventil skaliert*)
		rT_OCW_bCV : REAL; (*Temp Ölkühlwasser vor Regelventil skaliert*)
		rPosAct_ChCW_LT : REAL; (*Regler Ladekühlwasser Niedertemp. Rückmeldung*)
		rPosAct_ChCW_HT : REAL; (*Regler Ladekühlwasser Hochtemp. Rückmeldung*)
		rPosAct_ChCW_HT_LP : REAL; (*Regler Ladekühlwasser Hochtemp. Niederdruck Rückmeldung*)
		rPosAct_ChCW_HT_HP : REAL; (*Regler Ladekühlwasser Hochtemp. Hochdruck Rückmeldung*)
		rPosAct_ChCW_LT_LP : REAL; (*Regler Ladekühlwasser Niedertemp. Niederdruck Rückmeldung*)
		rPosAct_ChCW_LT_HP : REAL; (*Regler Ladekühlwasser Niedertemp. Hochdruck Rückmeldung*)
		rPosAct_ECW : REAL; (*Regler Motorkühlwasser Rückmeldung*)
		rPosAct_OCW : REAL; (*Regler Ölkühlwasser Rückmeldung*)
		rPosAct_RW_CV : REAL; (*Regler Rohwasser Regelventil Rückmeldung*)
		rPosAct_RW_HE : REAL; (*Regler Rohwasser Wärmetauscher Rückmeldung*)
		rPosAct_RW_LT_1 : REAL; (*Regler Rohwasser NT Rückmeldung*)
		rPosAct_RW_HT_1 : REAL; (*Regler Rohwasser HT Rückmeldung*)
		rPosAct_RW_LT_2 : REAL; (*Regler Rohwasser NT Rückmeldung*)
		rPosAct_RW_HT_2 : REAL; (*Regler Rohwasser HT Rückmeldung*)
		rPosAct_RW_ECW_1 : REAL; (*Regler Rohwasser Motorkühlwasser Rückmeldung*)
		rPosAct_RW_OCW_1 : REAL; (*Regler Rohwasser Ölkühlwasser Rückmeldung*)
		rPosAct_RW_ECW_2 : REAL; (*Regler Rohwasser Motorkühlwasser Rückmeldung*)
		rPosAct_RW_OCW_2 : REAL; (*Regler Rohwasser Ölkühlwasser Rückmeldung*)
		rSumChC_LT_Stages : REAL; (*Summer der Kühlerstufen NT*)
		rSumChC_HT_Stages : REAL; (*Summer der Kühlerstufen HT*)
		rSumECW_Stages : REAL; (*Summer der Motorkühlwasser Kühlerstufen*)
		rSumOCW_Stages : REAL; (*Summer der Ölkühlwasser Kühlerstufen*)
		rT_SecCirc_Su : REAL; (*Temperatur Sekundärkreis Vorlauf*)
		rT_BoilerHouse_Su : REAL; (*Temperatur Heizhaus Vorlauf*)
		rT_Cooler_ChCW_HT_Re_1_1 : REAL; (*Temp Ladekühler 1 1 HT Rücklauf*)
		rT_Cooler_ChCW_HT_Re_1_2 : REAL; (*Temp Ladekühler 1 2 HT Rücklauf*)
		rT_Cooler_ChCW_HT_Re_1_3 : REAL; (*Temp Ladekühler 1 3 HT Rücklauf*)
		rT_Cooler_ChCW_HT_Re_1_4 : REAL; (*Temp Ladekühler 1 4 HT Rücklauf*)
		rT_Cooler_OCW_Re_1_1 : REAL; (*Temp Ölkühler 1 1 Rücklauf*)
		rT_Cooler_OCW_Re_1_2 : REAL; (*Temp Ölkühler 1 2 Rücklauf*)
		rT_Cooler_ECW_Re_1_1 : REAL; (*Temp Motorkühlwasserkühler 1 1 Rücklauf*)
		rT_Cooler_ECW_Re_1_2 : REAL; (*Temp Motorkühlwasserkühler 1 2 Rücklauf*)
		rT_Cooler_ChCW_LT_Re_1_1 : REAL; (*Temp Ladekühler 1 1 NT Rücklauf*)
		rT_Cooler_ChCW_LT_Re_1_2 : REAL; (*Temp Ladekühler 1 2 NT Rücklauf*)
		bFlow_BoilerHouse_Lo : BOOL; (*DI Durchfluss Heizhaus zu nieder*)
		bPs_BoilerHouse_Hi : BOOL; (*DI Druck Heizhaus zu hoch*)
		bPs_BoilerHouse_Lo : BOOL; (*DI Druck Heizhaus zu nieder*)
		bTs_BoilerHouse_Hi : BOOL; (*DI Temp. Heizhaus zu hoch*)
		bFlow_SecCirc_Lo : BOOL; (*DI Durchfluss Sekundärkreis zu nieder*)
		bPs_SecCirc_Hi : BOOL; (*DI Druck Sekundärkreis zu hoch*)
		bPs_SecCirc_Lo : BOOL; (*DI Druck Sekundärkreis zu nieder*)
		bTs_SecCirc_Hi : BOOL; (*DI Temp. Sekundärkreis zu hoch*)
		bDem_BoilerHouse_Pump : BOOL; (*DO Anforderung Heizhauspumpe*)
		bDem_SecCirc_Pump : BOOL; (*DO Anforderung Sekundärkreispumpe*)
		rPr_RW_Su : REAL; (*Druck Rohwasser Vorlauf*)
		rT_Cooler_ChCW_HT_Re_3 : REAL; (*Temp Ladekühler 3 HT Rücklauf*)
		rT_Cooler_ChCW_HT_Re_4 : REAL; (*Temp Ladekühler 4 HT Rücklauf*)
		rT_Cooler_ChCW_HT_Re_5 : REAL; (*Temp Ladekühler 4 HT Rücklauf*)
		rT_Cooler_ChCW_HT_Su_3 : REAL; (*Temp Ladekühler 3 HT Vorlauf*)
		rT_Cooler_ChCW_HT_Su_4 : REAL; (*Temp Ladekühler 4 HT Vorlauf*)
		rT_Cooler_ChCW_HT_Su_5 : REAL; (*Temp Ladekühler 5 HT Vorlauf*)
		rT_CoolerCabinet_HT_1 : REAL; (*Temp Kühler Schaltschrank HT 1*)
		rT_CoolerCabinet_HT_2 : REAL; (*Temp Kühler Schaltschrank HT 2*)
		rT_CoolerCabinet_HT_3 : REAL; (*Temp Kühler Schaltschrank HT 3*)
		rT_CoolerCabinet_HT_4 : REAL; (*Temp Kühler Schaltschrank HT 4*)
		rT_CoolerCabinet_HT_5 : REAL; (*Temp Kühler Schaltschrank HT 5*)
		rT_Cooler_OCW_Re_3 : REAL; (*Temp Ölkühlwasserkühler 3 Rücklauf*)
		rT_Cooler_OCW_Su_3 : REAL; (*Temp Ölkühlwasserkühler 3 Vorlauf*)
		rT_CoolerCabinet_OCW_1 : REAL; (*Temp Ölkühlwasserkühler Schaltschrank 1*)
		rT_CoolerCabinet_OCW_2 : REAL; (*Temp Ölkühlwasserkühler Schaltschrank 2*)
		rT_CoolerCabinet_OCW_3 : REAL; (*Temp Ölkühlwasserkühler Schaltschrank 3*)
		rT_Cooler_ECW_Re_3 : REAL; (*Temp Motorkühlwasserkühler 3 Rücklauf*)
		rT_Cooler_ECW_Re_4 : REAL; (*Temp Motorkühlwasserkühler 4 Rücklauf*)
		rT_Cooler_ECW_Su_3 : REAL; (*Temp Motorkühlwasserkühler 3 Vorlauf*)
		rT_Cooler_ECW_Su_4 : REAL; (*Temp Motorkühlwasserkühler 4 Vorlauf*)
		rT_CoolerCabinet_ECW_1 : REAL; (*Temp Motorkühlwasserkühler Schaltschrank 1*)
		rT_CoolerCabinet_ECW_2 : REAL; (*Temp Motorkühlwasserkühler Schaltschrank 2*)
		rT_CoolerCabinet_ECW_3 : REAL; (*Temp Motorkühlwasserkühler Schaltschrank 3*)
		rT_CoolerCabinet_ECW_4 : REAL; (*Temp Motorkühlwasserkühler Schaltschrank 4*)
		rT_Cooler_ChCW_LT_Re_3 : REAL; (*Temp Ladekühler 3 NT Rücklauf*)
		rT_Cooler_ChCW_LT_Re_4 : REAL; (*Temp Ladekühler 4 NT Rücklauf*)
		rT_Cooler_ChCW_LT_Re_5 : REAL; (*Temp Ladekühler 5 NT Rücklauf*)
		rT_Cooler_ChCW_LT_Su_3 : REAL; (*Temp Ladekühler 3 NT Vorlauf*)
		rT_Cooler_ChCW_LT_Su_4 : REAL; (*Temp Ladekühler 4 NT Vorlauf*)
		rT_Cooler_ChCW_LT_Su_5 : REAL; (*Temp Ladekühler 5 NT Vorlauf*)
		rT_CoolerCabinet_LT_1 : REAL; (*Temp Kühler Schaltschrank NT 1*)
		rT_CoolerCabinet_LT_2 : REAL; (*Temp Kühler Schaltschrank NT 2*)
		rT_CoolerCabinet_LT_3 : REAL; (*Temp Kühler Schaltschrank NT 3*)
		rT_CoolerCabinet_LT_4 : REAL; (*Temp Kühler Schaltschrank NT 4*)
		rT_CoolerCabinet_LT_5 : REAL; (*Temp Kühler Schaltschrank NT 5*)
		bDem_LT_HP_PreHeat : BOOL; (*Anforderung Vorwärmung NT HD Kühlkreis*)
		bDem_LT_LP_PreHeat : BOOL; (*Anforderung Vorwärmung NT ND Kühlkreis*)
		bLT_HP_Flap_C : BOOL; (*Rückmeldung NT HD Klappe geschlossen*)
		bLT_HP_Flap_O : BOOL; (*Rückmeldung NT ND Klappe offen*)
		bLT_LP_Flap_C : BOOL; (*Rückmeldung NT HD Klappe geschlossen*)
		bLT_LP_Flap_O : BOOL; (*Rückmeldung NT ND Klappe offen*)
		bMsg7000 : BOOL; (*OPC-Verbindung zum Prüfstand ist unterbrochen*)
		bMsg7001 : BOOL; (*Temp. Ladekühlwasser Rücklauf Niedertemp. max Warnung*)
		bMsg7002 : BOOL; (*Temp. Ladekühlwasser Rücklauf Niedertemp. max Abstellung*)
		bMsg7003 : BOOL; (*Temp. Ladekühlwasser Vorlauf Niedertemp. max Warnung*)
		bMsg7004 : BOOL; (*Temp. Ladekühlwasser Vorlauf Niedertemp. max Abstellung*)
		bMsg7005 : BOOL; (*Temp. Ladekühlwasser Rücklauf Hochtemp. max Warnung*)
		bMsg7006 : BOOL; (*Temp. Ladekühlwasser Rücklauf Hochtemp. max Abstellung*)
		bMsg7007 : BOOL; (*Temp. Ladekühlwasser Vorlauf Hochtemp. max Warnung*)
		bMsg7008 : BOOL; (*Temp. Ladekühlwasser Vorlauf Hochtemp. max Abstellung*)
		bMsg7009 : BOOL; (*Temp. Ladekühlwasser Rücklauf Hochtemp. Niederdruck max Warnung*)
		bMsg7010 : BOOL; (*Temp. Ladekühlwasser Rücklauf Hochtemp. Niederdruck max Abstellung*)
		bMsg7011 : BOOL; (*Temp. Ladekühlwasser Rücklauf Hochtemp. Hochdruck max Warnung*)
		bMsg7012 : BOOL; (*Temp. Ladekühlwasser Rücklauf Hochtemp. Hochdruck max Abstellung*)
		bMsg7013 : BOOL; (*Temp. Ladekühlwasser Vorlauf Hochtemp. Niederdruck max Warnung*)
		bMsg7014 : BOOL; (*Temp. Ladekühlwasser Vorlauf Hochtemp. Niederdruck max Abstellung*)
		bMsg7015 : BOOL; (*Temp. Ladekühlwasser Vorlauf Hochtemp. Hochdruck max Warnung*)
		bMsg7016 : BOOL; (*Temp. Ladekühlwasser Vorlauf Hochtemp. Hochdruck max Abstellung*)
		bMsg7017 : BOOL; (*Temp. Ladekühlwasser Rücklauf Niedertemp. Niederdruck max Warnung*)
		bMsg7018 : BOOL; (*Temp. Ladekühlwasser Rücklauf Niedertemp. Niederdruck max Abstellung*)
		bMsg7019 : BOOL; (*Temp. Ladekühlwasser Rücklauf Niedertemp. Hochdruck max Warnung*)
		bMsg7020 : BOOL; (*Temp. Ladekühlwasser Rücklauf Niedertemp. Hochdruck max Abstellung*)
		bMsg7021 : BOOL; (*Temp. Ladekühlwasser Vorlauf Niedertemp. Niederdruck max Warnung*)
		bMsg7022 : BOOL; (*Temp. Ladekühlwasser Vorlauf Niedertemp. Niederdruck max Abstellung*)
		bMsg7023 : BOOL; (*Temp. Ladekühlwasser Vorlauf Niedertemp. Hochdruck max Warnung*)
		bMsg7024 : BOOL; (*Temp. Ladekühlwasser Vorlauf Niedertemp. Hochdruck max Abstellung*)
		bMsg7025 : BOOL; (*Temp. Ölkühlwasser Rücklauf max Warnung*)
		bMsg7026 : BOOL; (*Temp. Ölkühlwasser Rücklauf max Abstellung*)
		bMsg7027 : BOOL; (*Temp. Ölkühlwasser Vorlauf max Warnung*)
		bMsg7028 : BOOL; (*Temp. Ölkühlwasser Vorlauf max Abstellung*)
		bMsg7029 : BOOL; (*Temp. Motorkühlwasser Rücklauf max Warnung*)
		bMsg7030 : BOOL; (*Temp. Motorkühlwasser Rücklauf max Abstellung*)
		bMsg7031 : BOOL; (*Temp. Motorkühlwasser Vorlauf max Warnung*)
		bMsg7032 : BOOL; (*Temp. Motorkühlwasser Vorlauf max Abstellung*)
		bMsg7033 : BOOL; (*Druck min Rohwasserkühler 1 LT Warnung*)
		bMsg7034 : BOOL; (*Druck min Rohwasserkühler 1 HT Warnung*)
		bMsg7035 : BOOL; (*Temp. max Rohwasser Warnung*)
		bMsg7036 : BOOL; (*Temp. max Rohwasser Abstellung*)
		bMsg7037 : BOOL; (*Diff-Drucküberwachung der Kühler HT HP 1*)
		bMsg7038 : BOOL; (*Diff-Drucküberwachung der Kühler HT HP 2*)
		bMsg7039 : BOOL; (*Diff-Drucküberwachung der Kühler HT LP 1*)
		bMsg7040 : BOOL; (*Diff-Drucküberwachung der Kühler HT LP 2*)
		bMsg7041 : BOOL; (*Diff-Drucküberwachung der Kühler LT HP 1*)
		bMsg7042 : BOOL; (*Diff-Drucküberwachung der Kühler LT HP 2*)
		bMsg7043 : BOOL; (*Diff-Drucküberwachung der Kühler LT LP 1*)
		bMsg7044 : BOOL; (*Diff-Drucküberwachung der Kühler LT LP 2*)
		bMsg7045 : BOOL; (*Diff-Drucküberwachung der Kühler HT 1*)
		bMsg7046 : BOOL; (*Diff-Drucküberwachung der Kühler HT 2*)
		bMsg7047 : BOOL; (*Diff-Drucküberwachung der Kühler LT 1*)
		bMsg7048 : BOOL; (*Diff-Drucküberwachung der Kühler LT 2*)
		bMsg7049 : BOOL; (*Diff-Drucküberwachung der Kühler ECW 1*)
		bMsg7050 : BOOL; (*Diff-Drucküberwachung der Kühler ECW 2*)
		bMsg7051 : BOOL; (*Diff-Drucküberwachung der Kühler OCW 1*)
		bMsg7052 : BOOL; (*Diff-Drucküberwachung der Kühler OCW 2*)
		bMsg7053 : BOOL; (*Diff-Drucküberwachung des Rohwasserkühler LT 1*)
		bMsg7054 : BOOL; (*Diff-Drucküberwachung des Rohwasserkühler HT 1*)
		bMsg7055 : BOOL; (*Messsignalstörung Ladekühlwassertemp. Rücklauf NT*)
		bMsg7056 : BOOL; (*Messsignalstörung Ladekühlwasserdruck Rücklauf NT*)
		bMsg7057 : BOOL; (*Messsignalstörung Ladekühlwassertemp. Rücklauf HT*)
		bMsg7058 : BOOL; (*Messsignalstörung Ladekühlwasserdruck Rücklauf HT*)
		bMsg7059 : BOOL; (*Messsignalstörung Ladekühlwassertemp. Rücklauf HT ND*)
		bMsg7060 : BOOL; (*Messsignalstörung Ladekühlwasserdruck Rücklauf HT ND*)
		bMsg7061 : BOOL; (*Messsignalstörung Ladekühlwassertemp. Rücklauf HT HD*)
		bMsg7062 : BOOL; (*Messsignalstörung Ladekühlwasserdruck Rücklauf HT HD*)
		bMsg7063 : BOOL; (*Messsignalstörung Ladekühlwassertemp. Rücklauf NT ND*)
		bMsg7064 : BOOL; (*Messsignalstörung Ladekühlwasserdruck Rücklauf NT ND*)
		bMsg7065 : BOOL; (*Messsignalstörung Ladekühlwassertemp. Rücklauf NT HD*)
		bMsg7066 : BOOL; (*Messsignalstörung Ladekühlwasserdruck Rücklauf NT HD*)
		bMsg7067 : BOOL; (*Messsignalstörung Ölkühlwassertemp. Rücklauf*)
		bMsg7068 : BOOL; (*Messsignalstörung Ölkühlwasserdruck Rücklauf*)
		bMsg7069 : BOOL; (*Messsignalstörung Motorkühlwassertemp. Rücklauf*)
		bMsg7070 : BOOL; (*Messsignalstörung Motorkühlwasserdruck Rücklauf*)
		bMsg7071 : BOOL; (*Diff-Drucküberwachung des Rohwasserkühler LT 2*)
		bMsg7072 : BOOL; (*Diff-Drucküberwachung des Rohwasserkühler HT 2*)
		bMsg7073 : BOOL; (*Druckschalter Ladekühlwasser HT vor Motor ausgelöst*)
		bMsg7074 : BOOL; (*Druckschalter Ladekühlwasser NT ND vor Motor ausgelöst*)
		bMsg7075 : BOOL; (*Druckschalter Ladekühlwasser NT HD vor Motor ausgelöst*)
		bMsg7076 : BOOL; (*Druckschalter Ladekühlwasser HT ND vor Motor ausgelöst*)
		bMsg7077 : BOOL; (*Druckschalter Ladekühlwasser HT HD vor Motor ausgelöst*)
		bMsg7078 : BOOL; (*Druckschalter Ladekühlwasser NT vor Motor ausgelöst*)
		bMsg7079 : BOOL; (*Druckschalter Kühlwasser vor Motor ausgelöst*)
		bMsg7080 : BOOL; (*Druckschalter Motorkühlwasser vor Motor ausgelöst*)
		bMsg7081 : BOOL; (*Druckschalter Ölkühlwasser vor Motor ausgelöst*)
		bMsg7082 : BOOL; (*Druckschalter Ladekühlwasser NT vor Pumpe ausgelöst*)
		bMsg7083 : BOOL; (*Druckschalter Ladekühlwasser HT vor Pumpe ausgelöst*)
		bMsg7084 : BOOL; (*Druckschalter Ladekühlwasser NT ND vor Pumpe ausgelöst*)
		bMsg7085 : BOOL; (*Druckschalter Ladekühlwasser NT HD vor Pumpe ausgelöst*)
		bMsg7086 : BOOL; (*Druckschalter Ladekühlwasser HT ND vor Pumpe ausgelöst*)
		bMsg7087 : BOOL; (*Druckschalter Ladekühlwasser HT HD vor Pumpe ausgelöst*)
		bMsg7088 : BOOL; (*Temperatur max Rohwasser LT 1*)
		bMsg7089 : BOOL; (*Druckschalter Motorkühlwasser vor Pumpe ausgelöst*)
		bMsg7090 : BOOL; (*Druckschalter Ölkühlwasser vor Pumpe ausgelöst*)
		bMsg7091 : BOOL; (*Temperaturschalter Ladekühlwasser NT vor Motor ausgelöst*)
		bMsg7092 : BOOL; (*Temperaturschalter Ladekühlwasser HT vor Motor ausgelöst*)
		bMsg7093 : BOOL; (*Temperaturschalter Ladekühlwasser NT ND vor Motor ausgelöst*)
		bMsg7094 : BOOL; (*Temperaturschalter Ladekühlwasser NT HD vor Motor ausgelöst*)
		bMsg7095 : BOOL; (*Temperaturschalter Ladekühlwasser HT ND vor Motor ausgelöst*)
		bMsg7096 : BOOL; (*Temperaturschalter Ladekühlwasser HT HD vor Motor ausgelöst*)
		bMsg7097 : BOOL; (*Temperatur max Rohwasser LT 2*)
		bMsg7098 : BOOL; (*Temperaturschalter Motorkühlwasser vor Motor ausgelöst*)
		bMsg7099 : BOOL; (*Temperaturschalter Ölkühlwasser vor Motor ausgelöst*)
		bMsg7100 : BOOL; (*Ruhestromschleife vom Heizkreis nicht unterbrochen*)
		bMsg7101 : BOOL; (*Betriebsmedlung Ladekühlwasserkühler NT 1 fehlt*)
		bMsg7102 : BOOL; (*Störung Ladekühlwasserkühler NT 1*)
		bMsg7103 : BOOL; (*Betriebsmedlung Ladekühlwasserkühler NT 2 fehlt*)
		bMsg7104 : BOOL; (*Störung Ladekühlwasserkühler NT 2*)
		bMsg7105 : BOOL; (*Betriebsmedlung Ladekühlwasserkühler HT 1 fehlt*)
		bMsg7106 : BOOL; (*Störung Ladekühlwasserkühler HT 1*)
		bMsg7107 : BOOL; (*Betriebsmedlung Ladekühlwasserkühler HT 2 fehlt*)
		bMsg7108 : BOOL; (*Störung Ladekühlwasserkühler HT 2*)
		bMsg7109 : BOOL; (*Betriebsmedlung Ladekühlwasserkühler NT 3 fehlt*)
		bMsg7110 : BOOL; (*Störung Ladekühlwasserkühler NT 3*)
		bMsg7111 : BOOL; (*Betriebsmedlung Ladekühlwasserkühler NT 4 fehlt*)
		bMsg7112 : BOOL; (*Störung Ladekühlwasserkühler NT 4*)
		bMsg7113 : BOOL; (*Betriebsmedlung Ladekühlwasserkühler NT 5 fehlt*)
		bMsg7114 : BOOL; (*Störung Ladekühlwasserkühler NT 5*)
		bMsg7115 : BOOL; (*Betriebsmedlung Ladekühlwasserkühler HT 3 fehlt*)
		bMsg7116 : BOOL; (*Störung Ladekühlwasserkühler HT 3*)
		bMsg7117 : BOOL; (*Betriebsmedlung Ladekühlwasserkühler HT 4 fehlt*)
		bMsg7118 : BOOL; (*Störung Ladekühlwasserkühler HT 4*)
		bMsg7119 : BOOL; (*Betriebsmedlung Ladekühlwasserkühler HT 5 fehlt*)
		bMsg7120 : BOOL; (*Störung Ladekühlwasserkühler HT 5*)
		bMsg7121 : BOOL; (*Betriebsmedlung Motorkühlwasserkühler 3 fehlt*)
		bMsg7122 : BOOL; (*Störung Motorkühlwasserkühler 3*)
		bMsg7123 : BOOL; (*Betriebsmedlung Motorkühlwasserkühler 4 fehlt*)
		bMsg7124 : BOOL; (*Störung Motorkühlwasserkühler 4*)
		bMsg7125 : BOOL; (*Diff-Drucküberwachung des Rohwasserkühler Motorkühlwasser 1*)
		bMsg7126 : BOOL; (*Diff-Drucküberwachung des Rohwasserkühler Motorkühlwasser 2*)
		bMsg7127 : BOOL; (*Diff-Drucküberwachung des Rohwasserkühler Ölkühlwasser 1*)
		bMsg7128 : BOOL; (*Diff-Drucküberwachung des Rohwasserkühler Ölkühlwasser 2*)
		bMsg7129 : BOOL; (*Betriebsmedlung Motorkühlwasserkühler 1 fehlt*)
		bMsg7130 : BOOL; (*Störung Motorkühlwasserkühler 1*)
		bMsg7131 : BOOL; (*Betriebsmedlung Motorkühlwasserkühler 2 fehlt*)
		bMsg7132 : BOOL; (*Störung Motorkühlwasserkühler 2*)
		bMsg7133 : BOOL; (*Betriebsmedlung Ölkühlwasserkühler 1 fehlt*)
		bMsg7134 : BOOL; (*Störung Ölkühlwasserkühler 1*)
		bMsg7135 : BOOL; (*Betriebsmedlung Ölkühlwasserkühler 2 fehlt*)
		bMsg7136 : BOOL; (*Störung Ölkühlwasserkühler 2*)
		bMsg7137 : BOOL; (*Druck min Rohwasserkühler 2 LT Rücklauf Warnung*)
		bMsg7138 : BOOL; (*Druck min Rohwasserkühler 2 HT Rücklauf Warnung*)
		bMsg7139 : BOOL; (*Druck min Rohwasserkühler 1 Motorkühlwasser Warnung*)
		bMsg7140 : BOOL; (*Druck min Rohwasserkühler 1 Ölkühlwasser Warnung*)
		bMsg7141 : BOOL; (*Druck min Rohwasserkühler 2 Motorkühlwasser Warnung*)
		bMsg7142 : BOOL; (*Druck min Rohwasserkühler 2 Ölkühlwasser Warnung*)
		bMsg7143 : BOOL; (*Temp. Ladekühlwasser NT nach Rohwasserregelventil max Warnung*)
		bMsg7144 : BOOL; (*Temp. Ladekühlwasser NT nach Rohwasserregelventil max Abstellung*)
		bMsg7145 : BOOL; (*Temp. Rohwasser Wärmetauscher Rücklauf max Warnung*)
		bMsg7146 : BOOL; (*Temp. Rohwasser Wärmetauscher Rücklauf max Abstellung*)
		bMsg7147 : BOOL; (*Temp. Wärmetauscher Vorlauf max Warnung*)
		bMsg7148 : BOOL; (*Temp. Wärmetauscher Vorlauf max Abstellung*)
		bMsg7149 : BOOL; (*Druck Ladekühlwasser Rücklauf Niedertemp. min Warnung*)
		bMsg7150 : BOOL; (*Druck Ladekühlwasser Rücklauf Niedertemp. min Abstellung*)
		bMsg7151 : BOOL; (*Druck Ladekühlwasser Rücklauf Niedertemp. max Warnung*)
		bMsg7152 : BOOL; (*Druck Ladekühlwasser Rücklauf Niedertemp. max Abstellung*)
		bMsg7153 : BOOL; (*Druck Ladekühlwasser Vorlauf Niedertemp. min Warnung*)
		bMsg7154 : BOOL; (*Druck Ladekühlwasser Vorlauf Niedertemp. min Abstellung*)
		bMsg7155 : BOOL; (*Druck Ladekühlwasser Vorlauf Niedertemp. max Warnung*)
		bMsg7156 : BOOL; (*Druck Ladekühlwasser Vorlauf Niedertemp. max Abstellung*)
		bMsg7157 : BOOL; (*Druck Ladekühlwasser Rücklauf Hochtemp. min Warnung*)
		bMsg7158 : BOOL; (*Druck Ladekühlwasser Rücklauf Hochtemp. min Abstellung*)
		bMsg7159 : BOOL; (*Druck Ladekühlwasser Rücklauf Hochtemp. max Warnung*)
		bMsg7160 : BOOL; (*Druck Ladekühlwasser Rücklauf Hochtemp. max Abstellung*)
		bMsg7161 : BOOL; (*Druck Ladekühlwasser Vorlauf Hochtemp. min Warnung*)
		bMsg7162 : BOOL; (*Druck Ladekühlwasser Vorlauf Hochtemp. min Abstellung*)
		bMsg7163 : BOOL; (*Druck Ladekühlwasser Vorlauf Hochtemp. max Warnung*)
		bMsg7164 : BOOL; (*Druck Ladekühlwasser Vorlauf Hochtemp. max Abstellung*)
		bMsg7165 : BOOL; (*Druck Ladekühlwasser Rücklauf Hochtemp. Niederdruck min Warnung*)
		bMsg7166 : BOOL; (*Druck Ladekühlwasser Rücklauf Hochtemp. Niederdruck min Abstellung*)
		bMsg7167 : BOOL; (*Druck Ladekühlwasser Rücklauf Hochtemp. Niederdruck max Warnung*)
		bMsg7168 : BOOL; (*Druck Ladekühlwasser Rücklauf Hochtemp. Niederdruck max Abstellung*)
		bMsg7169 : BOOL; (*Druck Ladekühlwasser Rücklauf Hochtemp. Hochdruck min Warnung*)
		bMsg7170 : BOOL; (*Druck Ladekühlwasser Rücklauf Hochtemp. Hochdruck min Abstellung*)
		bMsg7171 : BOOL; (*Druck Ladekühlwasser Rücklauf Hochtemp. Hochdruck max Warnung*)
		bMsg7172 : BOOL; (*Druck Ladekühlwasser Rücklauf Hochtemp. Hochdruck max Abstellung*)
		bMsg7173 : BOOL; (*Druck Ladekühlwasser Vorlauf Hochtemp. Niederdruck min Warnung*)
		bMsg7174 : BOOL; (*Druck Ladekühlwasser Vorlauf Hochtemp. Niederdruck min Abstellung*)
		bMsg7175 : BOOL; (*Druck Ladekühlwasser Vorlauf Hochtemp. Niederdruck max Warnung*)
		bMsg7176 : BOOL; (*Druck Ladekühlwasser Vorlauf Hochtemp. Niederdruck max Abstellung*)
		bMsg7177 : BOOL; (*Druck Ladekühlwasser Vorlauf Hochtemp. Hochdruck min Warnung*)
		bMsg7178 : BOOL; (*Druck Ladekühlwasser Vorlauf Hochtemp. Hochdruck min Abstellung*)
		bMsg7179 : BOOL; (*Druck Ladekühlwasser Vorlauf Hochtemp. Hochdruck max Warnung*)
		bMsg7180 : BOOL; (*Druck Ladekühlwasser Vorlauf Hochtemp. Hochdruck max Abstellung*)
		bMsg7181 : BOOL; (*Druck Ladekühlwasser Rücklauf Niedertemp. Niederdruck min Warnung*)
		bMsg7182 : BOOL; (*Druck Ladekühlwasser Rücklauf Niedertemp. Niederdruck min Abstellung*)
		bMsg7183 : BOOL; (*Druck Ladekühlwasser Rücklauf Niedertemp. Niederdruck max Warnung*)
		bMsg7184 : BOOL; (*Druck Ladekühlwasser Rücklauf Niedertemp. Niederdruck max Abstellung*)
		bMsg7185 : BOOL; (*Druck Ladekühlwasser Rücklauf Niedertemp. Hochdruck min Warnung*)
		bMsg7186 : BOOL; (*Druck Ladekühlwasser Rücklauf Niedertemp. Hochdruck min Abstellung*)
		bMsg7187 : BOOL; (*Druck Ladekühlwasser Rücklauf Niedertemp. Hochdruck max Warnung*)
		bMsg7188 : BOOL; (*Druck Ladekühlwasser Rücklauf Niedertemp. Hochdruck max Abstellung*)
		bMsg7189 : BOOL; (*Druck Ladekühlwasser Vorlauf Niedertemp. Niederdruck min Warnung*)
		bMsg7190 : BOOL; (*Druck Ladekühlwasser Vorlauf Niedertemp. Niederdruck min Abstellung*)
		bMsg7191 : BOOL; (*Druck Ladekühlwasser Vorlauf Niedertemp. Niederdruck max Warnung*)
		bMsg7192 : BOOL; (*Druck Ladekühlwasser Vorlauf Niedertemp. Niederdruck max Abstellung*)
		bMsg7193 : BOOL; (*Druck Ladekühlwasser Vorlauf Niedertemp. Hochdruck min Warnung*)
		bMsg7194 : BOOL; (*Druck Ladekühlwasser Vorlauf Niedertemp. Hochdruck min Abstellung*)
		bMsg7195 : BOOL; (*Druck Ladekühlwasser Vorlauf Niedertemp. Hochdruck max Warnung*)
		bMsg7196 : BOOL; (*Druck Ladekühlwasser Vorlauf Niedertemp. Hochdruck max Abstellung*)
		bMsg7197 : BOOL; (*Druck Ölkühlwasser Rücklauf min Warnung*)
		bMsg7198 : BOOL; (*Druck Ölkühlwasser Rücklauf min Abstellung*)
		bMsg7199 : BOOL; (*Druck Ölkühlwasser Rücklauf max Warnung*)
		bMsg7200 : BOOL; (*Druck Ölkühlwasser Rücklauf max Abstellung*)
		bMsg7201 : BOOL; (*Druck Ölkühlwasser Vorlauf min Warnung*)
		bMsg7202 : BOOL; (*Druck Ölkühlwasser Vorlauf min Abstellung*)
		bMsg7203 : BOOL; (*Druck Ölkühlwasser Vorlauf max Warnung*)
		bMsg7204 : BOOL; (*Druck Ölkühlwasser Vorlauf max Abstellung*)
		bMsg7205 : BOOL; (*Druck Motorkühlwasser Rücklauf min Warnung*)
		bMsg7206 : BOOL; (*Druck Motorkühlwasser Rücklauf min Abstellung*)
		bMsg7207 : BOOL; (*Druck Motorkühlwasser Rücklauf max Warnung*)
		bMsg7208 : BOOL; (*Druck Motorkühlwasser Rücklauf max Abstellung*)
		bMsg7209 : BOOL; (*Druck Motorkühlwasser Vorlauf min Warnung*)
		bMsg7210 : BOOL; (*Druck Motorkühlwasser Vorlauf min Abstellung*)
		bMsg7211 : BOOL; (*Druck Motorkühlwasser Vorlauf max Warnung*)
		bMsg7212 : BOOL; (*Druck Motorkühlwasser Vorlauf max Abstellung*)
		bMsg7213 : BOOL; (*Positionsfehler Rohwasserkühler Ventil NT 1*)
		bMsg7214 : BOOL; (*Positionsfehler Rohwasserkühler Ventil NT 2*)
		bMsg7215 : BOOL; (*Positionsfehler Rohwasserkühler Ventil HT 1*)
		bMsg7216 : BOOL; (*Positionsfehler Rohwasserkühler Ventil HT 2*)
		bMsg7217 : BOOL; (*Positionsfehler Rohwasserkühler Ventil MKW 1*)
		bMsg7218 : BOOL; (*Positionsfehler Rohwasserkühler Ventil MKW 2*)
		bMsg7219 : BOOL; (*Positionsfehler Rohwasserkühler Ventil OKW 1*)
		bMsg7220 : BOOL; (*Positionsfehler Rohwasserkühler Ventil OKW 2*)
		bMsg7221 : BOOL; (*Betriebsmedlung Ölkühlwasserkühler 3 fehlt*)
		bMsg7222 : BOOL; (*Störung Ökühlwasserkühler 3*)
		bMsg7223 : BOOL; (*400V Versorgung Ladekühler fehlt*)
		bMsg7224 : BOOL; (*400V Versorgung OKW MKW Kühler fehlt*)
		bMsg7225 : BOOL; (*NT HD Klappe für Vorwärmung nicht geschlossen*)
		bMsg7226 : BOOL; (*NT ND Klappe für Vorwärmung nicht geschlossen*)
		bMsg7227 : BOOL; (*NT HD Klappe für Motorbetrieb nicht offen*)
		bMsg7228 : BOOL; (*NT ND Klappe für Motorbetrieb nicht offen*)
		bMsg7229 : BOOL; (*Störung Vorwärmung NT HD*)
		bMsg7230 : BOOL; (*Störung Vorwärmung NT ND*)
		bMsg7231 : BOOL; (*Druck Ladekühlwasser NT LP Zwischenkreis Rücklauf max Warnung*)
		bMsg7232 : BOOL; (*Druck Ladekühlwasser NT LP Zwischenkreis Rücklauf max Abstellung*)
		bMsg7233 : BOOL; (*Druck Ladekühlwasser NT HP Zwischenkreis Rücklauf min Warnung*)
		bMsg7234 : BOOL; (*Druck Ladekühlwasser NT HP Zwischenkreis Rücklauf min Abstellung*)
		bMsg7235 : BOOL; (*Druck Ladekühlwasser NT HP Zwischenkreis Rücklauf max Warnung*)
		bMsg7236 : BOOL; (*Druck Ladekühlwasser NT HP Zwischenkreis Rücklauf max Abstellung*)
		bMsg7237 : BOOL; (*Druck Ladekühlwasser HT LP Zwischenkreis Rücklauf min Warnung*)
		bMsg7238 : BOOL; (*Druck Ladekühlwasser HT LP Zwischenkreis Rücklauf min Abstellung*)
		bMsg7239 : BOOL; (*Druck Ladekühlwasser HT LP Zwischenkreis Rücklauf max Warnung*)
		bMsg7240 : BOOL; (*Druck Ladekühlwasser HT LP Zwischenkreis Rücklauf max Abstellung*)
		bMsg7241 : BOOL; (*Druck Ladekühlwasser HT HP Zwischenkreis Rücklauf min Warnung*)
		bMsg7242 : BOOL; (*Druck Ladekühlwasser HT HP Zwischenkreis Rücklauf min Abstellung*)
		bMsg7243 : BOOL; (*Druck Ladekühlwasser HT HP Zwischenkreis Rücklauf max Warnung*)
		bMsg7244 : BOOL; (*Druck Ladekühlwasser HT HP Zwischenkreis Rücklauf max Abstellung*)
		bMsg7245 : BOOL; (*Temperatur max Rohwasser HT 1*)
		bMsg7246 : BOOL; (*Temperatur max Rohwasser HT 2*)
		bMsg7247 : BOOL; (*Temperatur max Rohwasser MKW 1*)
		bMsg7248 : BOOL; (*Temperatur max Rohwasser MKW 2*)
		bMsg7249 : BOOL; (*Druck Motorkühlwasser Zwischenkreis Rücklauf min Warnung*)
		bMsg7250 : BOOL; (*Druck Motorkühlwasser Zwischenkreis Rücklauf min Abstellung*)
		bMsg7251 : BOOL; (*Druck Motorkühlwasser Zwischenkreis Rücklauf max Warnung*)
		bMsg7252 : BOOL; (*Druck Motorkühlwasser Zwischenkreis Rücklauf max Abstellung*)
		bMsg7253 : BOOL; (*Druck Ölkühlwasser Zwischenkreis Rücklauf min Warnung*)
		bMsg7254 : BOOL; (*Druck Ölkühlwasser Zwischenkreis Rücklauf min Abstellung*)
		bMsg7255 : BOOL; (*Druck Ölkühlwasser Zwischenkreis Rücklauf max Warnung*)
		bMsg7256 : BOOL; (*Druck Ölkühlwasser Zwischenkreis Rücklauf max Abstellung*)
		bMsg7257 : BOOL; (*Messsignalstörung Ladekühlwassertemp. NT Zwischenkreis Rücklauf*)
		bMsg7258 : BOOL; (*Messsignalstörung Ladekühlwassertemp. HT Zwischenkreis Rücklauf*)
		bMsg7259 : BOOL; (*Messsignalstörung Ladekühlwassertemp. NT ND Zwischenkreis Rücklauf*)
		bMsg7260 : BOOL; (*Messsignalstörung Ladekühlwassertemp. NT HD Zwischenkreis Rücklauf*)
		bMsg7261 : BOOL; (*Messsignalstörung Ladekühlwassertemp. HT ND Zwischenkreis Rücklauf*)
		bMsg7262 : BOOL; (*Messsignalstörung Ladekühlwassertemp. HT ND Zwischenkreis Rücklauf*)
		bMsg7263 : BOOL; (*Temperatur max Rohwasser OKW 1*)
		bMsg7264 : BOOL; (*Messsignalstörung Motorkühlwassertemp. Zwischenkreis Rücklauf*)
		bMsg7265 : BOOL; (*Messsignalstörung Ölkühlwassertemp. Zwischenkreis Rücklauf*)
		bMsg7266 : BOOL; (*FU Ladekühlwasser NT nicht bereit*)
		bMsg7267 : BOOL; (*FU Ladekühlwasser HT nicht bereit*)
		bMsg7268 : BOOL; (*FU Ladekühlwasser NT ND nicht bereit*)
		bMsg7269 : BOOL; (*FU Ladekühlwasser NT HD nicht bereit*)
		bMsg7270 : BOOL; (*FU Ladekühlwasser HT ND nicht bereit*)
		bMsg7271 : BOOL; (*FU Ladekühlwasser HT HD nicht bereit*)
		bMsg7272 : BOOL; (*FU Motorkühlwasser nicht bereit*)
		bMsg7273 : BOOL; (*FU Ölkühlwasser nicht bereit*)
		bMsg7274 : BOOL; (*Temperatur max Rohwasser OKW 2*)
		bMsg7275 : BOOL; (*Ausdehnungsautomat Ladekühlwasser NT ausgelöst*)
		bMsg7276 : BOOL; (*Ausdehnungsautomat Ladekühlwasser HT ausgelöst*)
		bMsg7277 : BOOL; (*Ausdehnungsautomat Ladekühlwasser NT ND ausgelöst*)
		bMsg7278 : BOOL; (*Ausdehnungsautomat Ladekühlwasser NT HD ausgelöst*)
		bMsg7279 : BOOL; (*Ausdehnungsautomat Ladekühlwasser HT ND ausgelöst*)
		bMsg7280 : BOOL; (*Ausdehnungsautomat Ladekühlwasser HT HD ausgelöst*)
		bMsg7281 : BOOL; (*Ausdehnungsautomat Motorkühlwasser ausgelöst*)
		bMsg7282 : BOOL; (*Ausdehnungsautomat Ölkühlwasser ausgelöst*)
		bMsg7283 : BOOL; (*Druckschalter Rohwasser zu nieder*)
		bMsg7284 : BOOL; (*Temperaturschalter Rohwasser zu hoch*)
		bMsg7285 : BOOL; (*Druckschalter Ladekühlwasser NT nach Motor ausgelöst*)
		bMsg7286 : BOOL; (*Druckschalter Ladekühlwasser HT nach Motor ausgelöst*)
		bMsg7287 : BOOL; (*Druckschalter Ladekühlwasser NT ND nach Motor ausgelöst*)
		bMsg7288 : BOOL; (*Druckschalter Ladekühlwasser NT HD nach Motor ausgelöst*)
		bMsg7289 : BOOL; (*Druckschalter Ladekühlwasser HT ND nach Motor ausgelöst*)
		bMsg7290 : BOOL; (*Druckschalter Ladekühlwasser HT HD nach Motor ausgelöst*)
		bMsg7291 : BOOL; (*Druckschalter Motorkühlwasser nach Motor ausgelöst*)
		bMsg7292 : BOOL; (*Druckschalter Ölkühlwasser nach Motor ausgelöst*)
		bMsg7293 : BOOL; (*Störung Ladekühlwasserventilatoren NT*)
		bMsg7294 : BOOL; (*Störung Ladekühlwasserventilatoren HT*)
		bMsg7295 : BOOL; (*Störung Motorkühlwasserventilatoren*)
		bMsg7296 : BOOL; (*Störung Ölkühlwasserventilatoren*)
		bMsg7297 : BOOL; (*Störung Sekundärkreis Pumpe*)
		bMsg7298 : BOOL; (*Störung Heizhaus Pumpe*)
		bMsg7299 : BOOL; (*Störung NT Pumpe*)
		bMsg7300 : BOOL; (*Störung HT Pumpe*)
		bMsg7301 : BOOL; (*Störung MKW Pumpe*)
		bMsg7302 : BOOL; (*Störung OKW Pumpe*)
		bMsg7303 : BOOL; (*Durchfluss Heizhaus zu nieder*)
		bMsg7304 : BOOL; (*Druck Heizhaus zu hoch*)
		bMsg7305 : BOOL; (*Druck Heizhaus zu nieder*)
		bMsg7306 : BOOL; (*Temp. Heizhaus zu hoch*)
		bMsg7307 : BOOL; (*Durchfluss Sekundärkreis zu nieder*)
		bMsg7308 : BOOL; (*Druck Sekundärkreis zu hoch*)
		bMsg7309 : BOOL; (*Druck Sekundärkreis zu nieder*)
		bMsg7310 : BOOL; (*Temp. Sekundärkreis zu hoch*)
		bMsg7311 : BOOL;
		bMsg7312 : BOOL;
		bMsg7313 : BOOL;
		bMsg7314 : BOOL;
		bMsg7315 : BOOL;
		bMsg7316 : BOOL;
		bMsg7317 : BOOL;
		bMsg7318 : BOOL;
		bMsg7319 : BOOL;
		bMsg7320 : BOOL;
		bMsg7321 : BOOL;
		bMsg7322 : BOOL;
		bMsg7323 : BOOL;
		bMsg7324 : BOOL;
		bMsg7325 : BOOL;
		bMsg7326 : BOOL;
		bMsg7327 : BOOL;
		bMsg7328 : BOOL;
		bMsg7329 : BOOL;
		bMsg7330 : BOOL;
		bMsg7331 : BOOL;
		bMsg7332 : BOOL;
		bMsg7333 : BOOL;
		bMsg7334 : BOOL;
		bMsg7335 : BOOL;
		bMsg7336 : BOOL;
		bMsg7337 : BOOL;
		bMsg7338 : BOOL;
		bMsg7339 : BOOL;
		bMsg7340 : BOOL;
		bMsg7341 : BOOL;
		bMsg7342 : BOOL;
		bMsg7343 : BOOL;
		bMsg7344 : BOOL;
		bMsg7345 : BOOL;
		bMsg7346 : BOOL;
		bMsg7347 : BOOL;
		bMsg7348 : BOOL;
		bMsg7349 : BOOL;
		bMsg7350 : BOOL;
		bMsg7351 : BOOL;
		bMsg7352 : BOOL;
		bMsg7353 : BOOL;
		bMsg7354 : BOOL;
		bMsg7355 : BOOL;
		bMsg7356 : BOOL;
		bMsg7357 : BOOL;
		bMsg7358 : BOOL;
		bMsg7359 : BOOL;
		bMsg7360 : BOOL;
		bMsg7361 : BOOL;
		bMsg7362 : BOOL;
		bMsg7363 : BOOL;
		bMsg7364 : BOOL;
		bMsg7365 : BOOL;
		bMsg7366 : BOOL;
		bMsg7367 : BOOL;
		bMsg7368 : BOOL;
		bMsg7369 : BOOL;
		bMsg7370 : BOOL;
		bMsg7371 : BOOL;
		bMsg7372 : BOOL;
		bMsg7373 : BOOL;
		bMsg7374 : BOOL;
		bMsg7375 : BOOL;
		bMsg7376 : BOOL;
		bMsg7377 : BOOL;
		bMsg7378 : BOOL;
		bMsg7379 : BOOL;
		bMsg7380 : BOOL;
		bMsg7381 : BOOL;
		bMsg7382 : BOOL;
		bMsg7383 : BOOL;
		bMsg7384 : BOOL;
		bMsg7385 : BOOL;
		bMsg7386 : BOOL;
		bMsg7387 : BOOL;
		bMsg7388 : BOOL;
		bMsg7389 : BOOL;
		bMsg7390 : BOOL;
		bMsg7391 : BOOL;
		bMsg7392 : BOOL;
		bMsg7393 : BOOL;
		bMsg7394 : BOOL;
		bMsg7395 : BOOL;
		bMsg7396 : BOOL;
		bMsg7397 : BOOL;
		bMsg7398 : BOOL;
		bMsg7399 : BOOL;
		rSet_InLou : REAL; (*Sollwert Zuluftjalousie*)
		rSet_InLouRoom : REAL; (*Sollwert Zuluftjalousie Raum*)
		rSet_OutLou : REAL; (*Sollwert Abluftjalousie*)
		rSet_CircLou : REAL; (*Sollwert Umluftjalousie*)
		rSet_InLouEng : REAL; (*Sollwert Zuluftjalousie Motor*)
		rSet_CircLouEng : REAL; (*Sollwert Umluftjalousie Motor*)
		rCtr_InER_FC : REAL; (*Sollwert Frequnzumrichter Zuluftventilator 1-4*)
		rCtr_OutER_FC : REAL; (*Sollwert Frequnzumrichter Abluftventilator 1-4*)
		rCtr_InEngER_FC : REAL; (*Sollwert Frequnzumrichter Motor Frischluft Ventilator*)
		rCtr_CV_InAirHeat : REAL; (*Sollwert Motor Frischluft Temperaturregelventil Heizkreis*)
		rCtr_CV_InAirCool : REAL; (*Sollwert Motor Frischluft Temperaturregelventil Kühlkreis*)
		bInAirER_Fan1DemOn : BOOL; (*Anforderung Freuquenzumformer Zuluftventilatoren*)
		bOutAirER_Fan1DemOn : BOOL; (*Anforderung Freuquenzumformer Abluftventilatoren*)
		bInAirEng_FanDemOn : BOOL; (*Anforderung Freuquenzumformer Motor Frischluftventilator*)
		bDem_HeaterInAirEng : BOOL; (*Anforderung Heizstäbe Motorzuluft*)
		bDem_PumpInAirEng : BOOL; (*Anforderung Umwälzpumpe Motorzuluft*)
		bDem_EmptyInAirCool : BOOL; (*Anforderung Motor Frischluft Entleerlungsventil Kühlregister*)
		bTS_FrostProtection : BOOL; (*Frostschutzschalter hat ausgelöst*)
		bDem_ERV_Aut_Exist : BOOL; (*HW-Schalter Anforderung Lüftung Motorraum Automatik vorhanden*)
		rT_AirER_Avg : REAL; (*Durchschnitswert aller Raumtemperaturen*)
		rPos_InlLou1 : REAL; (*AI position air inlet louver 1 [%]*)
		rPos_InlLou2 : REAL; (*AI position air inlet louver 2 [%]*)
		rPos_OutlLou1 : REAL; (*AI position air outlet louver 1 [%]*)
		rPos_OutlLou2 : REAL; (*AI position air outlet louver 2 [%]*)
		rPos_CircLou1 : REAL; (*AI position air circulation louver 1 [%]*)
		rPos_CircLou2 : REAL; (*AI position air circulation louver 2 [%]*)
		rPos_InLouEng1 : REAL; (*Position Zuluftjalousie Motor Frischluft 1*)
		rPos_CircLouEng1 : REAL; (*Position Umluftjalousie Motor Frischluft 1*)
		rPos_InlLouRoom1 : REAL; (*AI: position air inlet louver room 1*)
		rPos_InlLouRoom2 : REAL; (*AI: position air inlet louver room 2*)
		rPos_InlLouRoom3 : REAL; (*AI: position air inlet louver room 3*)
		rPos_InlLouRoom4 : REAL; (*AI: position air inlet louver room 4*)
		rPos_OutlLou3 : REAL; (*AI: position air outlet louver 3*)
		rPos_OutlLou4 : REAL; (*AI: position air outlet louver 4*)
		rPos_InLouEng2 : REAL; (*Position Zuluftjalousie Motor Frischluft 2*)
		rPos_CircLouEng2 : REAL; (*Position Umluftjalousie Motor Frischluft 2*)
		rPos_CV_InAirHeat : REAL; (*Position Motor Frischluft Temperaturregelventil Heizkreis*)
		rPos_CV_InAirCool : REAL; (*Position Motor Frischluft Temperaturregelventil Kühlkreis*)
		rT_AirER1 : REAL; (*Raumtemperatur 1*)
		rT_AirER2 : REAL; (*Raumtemperatur 2*)
		rT_AirER3 : REAL; (*Raumtemperatur 3*)
		rT_AirER4 : REAL; (*Raumtemperatur 4*)
		rT_AirOutdoor : REAL; (*Außentemperatur*)
		rT_FreshAirIn : REAL; (*Temperatur Zuluftkanal Motorfrischluft*)
		rT_FreshAirEng : REAL; (*Temperatur Zuluftkanal Motorfrischluft (vor Motor)*)
		rT_HW_Air_Re : REAL; (*Temperatur Rücklauf Heizkreis*)
		rT_HW_Air_Su : REAL; (*Temperatur Vorlauf Heizkreis*)
		rPrDiff_ER : REAL; (*Raumdiffernzdruck*)
		rPr_Cool_Air_Re : REAL; (*Druck Rücklauf Kühlkreis*)
		rPr_HW_Air_Re : REAL; (*Druck Rücklauf Heizkreis*)
		rT_Cool_Air_Re : REAL; (*Temperatur Rücklauf Kühlkreis*)
		rT_Cool_Air_Su : REAL; (*Temperatur Vorlauf Kühlkreis*)
		rT_FreshAirEngA : REAL; (*Temperatur Zuluftkanal Motorfrischluft A (vor Motor)*)
		rT_FreshAirEngB : REAL; (*Temperatur Zuluftkanal Motorfrischluft B (vor Motor)*)
		rT_CircAirEng : REAL; (*Temperatur Umluft Zuluftkonditionierung*)
		rT_AirER5 : REAL; (*Raumtemperatur 5*)
		rT_AirER6 : REAL; (*Raumtemperatur 6*)
		bMsg7400 : BOOL; (*MSS Raumtemp 1*)
		bMsg7401 : BOOL; (*MSS Raumtemp 2*)
		bMsg7402 : BOOL; (*MSS Raumtemp 3*)
		bMsg7403 : BOOL; (*MSS Raumtemp 4*)
		bMsg7404 : BOOL; (*Lüftungswahlschalter ist nicht auf Automatik*)
		bMsg7405 : BOOL; (*Positionsfehler Zuluftjalousie 1*)
		bMsg7406 : BOOL; (*Positionsfehler Zuluftjalousie 2*)
		bMsg7407 : BOOL; (*Positionsfehler Abluftjalousie 1*)
		bMsg7408 : BOOL; (*Positionsfehler Abluftjalousie 2*)
		bMsg7409 : BOOL; (*Messsignalstörung Raumdifferenzdruck*)
		bMsg7410 : BOOL; (*Messsignalstörung Position Zuluftjalousie Motor*)
		bMsg7411 : BOOL; (*Messsignalstörung Position Umluftjalousie Motor*)
		bMsg7412 : BOOL; (*Messsignalstörung Außentemperatur*)
		bMsg7413 : BOOL; (*Warnung, dass der Frostschutzschalter ausgelöst hat*)
		bMsg7414 : BOOL; (*Sicherungsfall 24VDC Stützpunkt (Control Room Ventilation)*)
		bMsg7415 : BOOL; (*Störung Frequenzumformer Zuluftventilatoren 1&2*)
		bMsg7416 : BOOL; (*Motorschutz Zuluftventilator 1 ausgelöst*)
		bMsg7417 : BOOL; (*Motorschutz Zuluftventilator 2 ausgelöst*)
		bMsg7418 : BOOL; (*Störung Frequenzumformer Zuluftventilatoren 3&4*)
		bMsg7419 : BOOL; (*Motorschutz Zuluftventilator 3 ausgelöst*)
		bMsg7420 : BOOL; (*Motorschutz Zuluftventilator 4 ausgelöst*)
		bMsg7421 : BOOL; (*Störung Frequenzumformer Abluftventilatoren 1&2*)
		bMsg7422 : BOOL; (*Motorschutz Abluftventilator 1 ausgelöst*)
		bMsg7423 : BOOL; (*Motorschutz Abluftventilator 2 ausgelöst*)
		bMsg7424 : BOOL; (*Störung Frequenzumformer Abluftventilatoren 3&4*)
		bMsg7425 : BOOL; (*Motorschutz Abluftventilator 3 ausgelöst*)
		bMsg7426 : BOOL; (*Motorschutz Abluftventilator 2 ausgelöst*)
		bMsg7427 : BOOL; (*Positionsfehler Umluftjalousie 1*)
		bMsg7428 : BOOL; (*Positionsfehler Umluftjalousie 2*)
		bMsg7429 : BOOL; (*Positionsfehler Zuluftjalousie Motor*)
		bMsg7430 : BOOL; (*Positionsfehler Umluftjalousie Motor*)
		bMsg7431 : BOOL; (*Differenzdruckschalter Raum Luftilter 1*)
		bMsg7432 : BOOL; (*Differenzdruckschalter Raum Luftilter 2*)
		bMsg7433 : BOOL; (*Differenzdruckschalter Luftilter Motor Frischluft*)
		bMsg7434 : BOOL; (*Temperatur max Heizstäbe Motorzuluft*)
		bMsg7435 : BOOL; (*Störung Umwälzpumpe Motorzuluft*)
		bMsg7436 : BOOL; (*Türkontakt geöffnet*)
		bMsg7437 : BOOL; (*Motorschutz Motor Frischluft Ventilator ausgelöst*)
		bMsg7438 : BOOL; (*engine room fan failure trip*)
		bMsg7439 : BOOL; (*Positionsfehler Abluftjalousie 3*)
		bMsg7440 : BOOL; (*Positionsfehler Abluftjalousie 4*)
		bMsg7441 : BOOL; (*Positionsfehler Zuluftjalousie Raum 1*)
		bMsg7442 : BOOL; (*Positionsfehler Zuluftjalousie Raum 2*)
		bMsg7443 : BOOL; (*Positionsfehler Zuluftjalousie Raum 3*)
		bMsg7444 : BOOL; (*Positionsfehler Zuluftjalousie Raum 4*)
		bMsg7445 : BOOL; (*Positionsfehler Zuluftjalousie Motor 2*)
		bMsg7446 : BOOL; (*Positionsfehler Umluftjalousie Motor 2*)
		bMsg7447 : BOOL; (*Motorschutz Motor Frischluft Ventilator 2 ausgelöst*)
		bMsg7448 : BOOL; (*Druckschalter Zuluftkonditionierung Heizkreis ausgelöst*)
		bMsg7449 : BOOL; (*Störung Frequenzumformer Motor Frischluft Ventilator*)
		bMsg7450 : BOOL; (*MSS Raumtemp 5*)
		bMsg7451 : BOOL; (*MSS Raumtemp 6*)
		bMsg7452 : BOOL; (*PTC Überwachung Motor vom Raum Zuluftventilator 1*)
		bMsg7453 : BOOL; (*PTC Überwachung Motor vom Raum Zuluftventilator 2*)
		bMsg7454 : BOOL; (*PTC Überwachung Motor vom Raum Zuluftventilator 3*)
		bMsg7455 : BOOL; (*PTC Überwachung Motor vom Raum Zuluftventilator 4*)
		bMsg7456 : BOOL; (*PTC Überwachung Motor vom Raum Abluftventilator 1*)
		bMsg7457 : BOOL; (*PTC Überwachung Motor vom Raum Abluftventilator 2*)
		bMsg7458 : BOOL; (*PTC Überwachung Motor vom Raum Abluftventilator 3*)
		bMsg7459 : BOOL; (*PTC Überwachung Motor vom Raum Abluftventilator 4*)
		bMsg7460 : BOOL; (*PTC Überwachung Motor vom Motor Zuluftventilator*)
		bMsg7461 : BOOL;
		bMsg7462 : BOOL;
		bMsg7463 : BOOL;
		bMsg7464 : BOOL;
		bMsg7465 : BOOL;
		bMsg7466 : BOOL;
		bMsg7467 : BOOL;
		bMsg7468 : BOOL;
		bMsg7469 : BOOL;
		bMsg7470 : BOOL;
		bMsg7471 : BOOL;
		bMsg7472 : BOOL;
		bMsg7473 : BOOL;
		bMsg7474 : BOOL;
		bMsg7475 : BOOL;
		bMsg7476 : BOOL;
		bMsg7477 : BOOL;
		bMsg7478 : BOOL;
		bMsg7479 : BOOL;
		bMsg7480 : BOOL;
		bMsg7481 : BOOL;
		bMsg7482 : BOOL;
		bMsg7483 : BOOL;
		bMsg7484 : BOOL;
		bMsg7485 : BOOL;
		bMsg7486 : BOOL;
		bMsg7487 : BOOL;
		bMsg7488 : BOOL;
		bMsg7489 : BOOL;
		bMsg7490 : BOOL;
		bMsg7491 : BOOL;
		bMsg7492 : BOOL;
		bMsg7493 : BOOL;
		bMsg7494 : BOOL;
		bMsg7495 : BOOL;
		bMsg7496 : BOOL;
		bMsg7497 : BOOL;
		bMsg7498 : BOOL;
		bMsg7499 : BOOL;
		rT_EG_PrReliefVa1 : REAL; (*AI temperature exhaust gas pressure relief valve 1*)
		rT_EG_PrReliefVa2 : REAL; (*AI temperature exhaust gas pressure relief valve 2*)
		rPr_EG_Deflag_Fast : REAL; (*AI: Exhaust gas pressure fast*)
		rPr_OXIcat_In_Fast_Peak : REAL; (*Exhaust gas inlet peak pressure fast*)
		rPosAct_SCR_EG_Flap : REAL; (*Positionsrückmeldung SCR Abgasklappe*)
		rPosAct_SCR_By_Flap : REAL; (*Positionsrückmeldung SCR Bypassklappe*)
		rPosAct_DPF_EG_Flap : REAL; (*Positionsrückmeldung DPF Abgasklappe*)
		rPosAct_DPF_By_Flap : REAL; (*Positionsrückmeldung DPF Bypassklappe*)
		rPr_EG_Deflag : REAL; (*Messung Abgasgegendruck*)
		bSCR_Exh_Flap_O : BOOL; (*Rückmeldung SCR Abgasklappe offen*)
		bSCR_Exh_Flap_C : BOOL; (*Rückmeldung SCR Abgasklappe geschlossen*)
		bSCR_By_Flap_O : BOOL; (*Rückmeldung SCR Bypassklappe offen*)
		bSCR_By_Flap_C : BOOL; (*Rückmeldung SCR Bypassklappe geschlossen*)
		bDPF_Exh_Flap_O : BOOL; (*Rückmeldung DPF Abgasklappe offen*)
		bDPF_Exh_Flap_C : BOOL; (*Rückmeldung DPF Abgasklappe geschlossen*)
		bDPF_By_Flap_O : BOOL; (*Rückmeldung DPF Bypassklappe offen*)
		bDPF_By_Flap_C : BOOL; (*Rückmeldung DPF Bypassklappe geschlossen*)
		rCtr_SCR_EG_Flap_Set : REAL; (*Sollwert SCR Abgasklappe*)
		rCtr_SCR_By_Flap_Set : REAL; (*Sollwert SCR Bypassklappe*)
		rCtr_DPF_EG_Flap_Set : REAL; (*Sollwert DPF Abgasklappe*)
		rCtr_DPF_By_Flap_Set : REAL; (*Sollwert DPF Bypassklappe*)
		rCtr_EG_Flap_Set : REAL; (*Sollwert Abgasklappe*)
		rPosAct_EG_Flap : REAL; (*Positionsrückmeldung Abgasklappe*)
		rPosAct_EG_Flap2 : REAL; (*Positionsrückmeldung Abgasklappe 2*)
		rCtr_EG_Flap : REAL; (*Anwahl der Abgasklappen*)
		bMsg7500 : BOOL; (*Öffnungsfehler Bypass DPF*)
		bMsg7501 : BOOL; (*Positionsfehler Bypass DPF*)
		bMsg7502 : BOOL; (*Messsignalstörung Bypass DPF*)
		bMsg7503 : BOOL; (*Öffnungsfehler Abgasklappe DPF*)
		bMsg7504 : BOOL; (*Positionsfehler Abgasklappe DPF*)
		bMsg7505 : BOOL; (*Messsignalstörung Abgasklappe DPF*)
		bMsg7506 : BOOL; (*Öffnungsfehler Bypass SCR*)
		bMsg7507 : BOOL; (*Positionsfehler Bypass SCR*)
		bMsg7508 : BOOL; (*Messsignalstörung Bypass SCR*)
		bMsg7509 : BOOL; (*Öffnungsfehler Abgasklappe SCR*)
		bMsg7510 : BOOL; (*Positionsfehler Abgasklappe SCR*)
		bMsg7511 : BOOL; (*Messsignalstörung Abgasklappe SCR*)
		bMsg7512 : BOOL; (*Messsignalstörung Abgasgegendruck*)
		bMsg7513 : BOOL; (*Abgasgegendruck zu hoch*)
		bMsg7514 : BOOL; (*Abgastemperatur zu hoch Auslassventil 1*)
		bMsg7515 : BOOL; (*Abgastemperatur zu hoch Auslassventil 2*)
		bMsg7516 : BOOL; (*Messsignalstörung Abgastemperatur Auslassventil 1*)
		bMsg7517 : BOOL; (*Messsignalstörung Abgastemperatur Auslassventil 1*)
		bMsg7518 : BOOL; (*Abgasdruck schell zu hoch*)
		bMsg7519 : BOOL; (*Messsignalstörung Abgasdruck schell*)
		bMsg7520 : BOOL; (*Öffnungsfehler Abgasklappe*)
		bMsg7521 : BOOL; (*Positionsfehler Abgasklappe*)
		bMsg7522 : BOOL; (*Messsignalstörung Abgasklappe*)
		bMsg7523 : BOOL; (*Störung Abgasklappe*)
		bMsg7524 : BOOL; (*Abgasklappe Drehmoment maximum*)
		bMsg7525 : BOOL; (*Öffnungsfehler Abgasklappe 2 *)
		bMsg7526 : BOOL; (*Positionsfehler Abgasklappe 2*)
		bMsg7527 : BOOL; (*Messsignalstörung Abgasklappe 2*)
		bMsg7528 : BOOL; (**)
		bMsg7529 : BOOL; (**)
		bMsg7530 : BOOL; (**)
		rVol_GT_NG : REAL; (*Messung Gasmenge Erdgas*)
		rVol_GT_PG : REAL; (*Messung Gasmenge Propangas*)
		rVol_GT_SG : REAL; (*Messung Gasmenge Sondergas*)
		rMFC_Act_PG : REAL; (*Messung Mass Fow Controller Propangas*)
		rMFC_Act_SG : REAL; (*Messung Mass Fow Controller Sondergas*)
		rPosAct_LSCS_GV : REAL; (*Messung Gasventil Vorkammergas - LSCS*)
		rPosAct_LSCS_MV : REAL; (*Messung Mischventil Vorkammergas - LSCS*)
		rPr_GT_NG : REAL; (*Messung Druck Gasstrecke Erdgas*)
		rPr_GT_PG : REAL; (*Messung Druck Gasstrecke Propangas*)
		rPr_GT_SG : REAL; (*Messung Druck Gasstrecke Sondergas*)
		rPr_PCG_Tank : REAL; (*Messung Druck Vorkammergas Kessel*)
		rT_GT_NG : REAL; (*Messung Temperatur Gasstrecke Erdgas*)
		rT_GT_PG : REAL; (*Messung Temperatur Gasstrecke Propangas*)
		rT_GT_SG : REAL; (*Messung Temperatur Gasstrecke Sondergas*)
		bLSCS_GV_Opened : BOOL; (*LSCS - Gasventil Vorkammergas offen*)
		bLSCS_GV_Closed : BOOL; (*LSCS - Gasventil Vorkammergas geschlossen*)
		bLSCS_MV_Opened : BOOL; (*LSCS - Gemischventil Vorkammergas offen*)
		bLSCS_MV_Closed : BOOL; (*LSCS - Gemischventil Vorkammergas geschlossen*)
		rCtr_MFC_PG : REAL; (*Sollwert Mass Flow Controller Propangas*)
		rCtr_MFC_SG : REAL; (*Sollwert Mass Flow Controller Sondergas*)
		rCtr_By1_GComp : REAL; (*Sollwert Stellventil Bypass 1 Gasverdichter*)
		rCtr_By2_GComp : REAL; (*Sollwert Stellventil Bypass 2 Gasverdichter*)
		rCtr_LSCS_GV : REAL; (*Sollwert LSCS Gasventil Vorkammergas*)
		rCtr_LSCS_MV : REAL; (*Sollwert LSCS Mischventil Vorkammergas*)
		rAct_LSCS_MV_Calc : REAL; (*Berechneter Wert des momentanen koeffizienten der Blendenöffnung*)
		rAct_LSCS_GV_Calc : REAL; (*Berechneter Wert des momentanen koeffizienten der Blendenöffnung*)
		rLSCS_Diff : REAL; (*Öffnungsverhältnis*)
		rCtr_MFC_PG_Set : REAL; (*Mass Flow Controller Vorgabe*)
		rCtr_MFC_SG_Set : REAL; (*Mass Flow Controller Vorgabe*)
		bDem_FV_PCGC_NG : BOOL; (*Anforderung Füllventil Vorkammergasverdichter Erdgas*)
		bDem_FV_PCGC_MG : BOOL; (*Anforderung Füllventil Vorkammergasverdichter Mischgas*)
		bDem_FV_PCGC_PG : BOOL; (*Anforderung Füllventil Vorkammergasverdichter Propangas*)
		bDem_GV_NG : BOOL; (*Anforderung Hauptgasventil Erdgas*)
		bDem_GV_PG : BOOL; (*Anforderung Hauptgasventil Propangas*)
		bDem_GV_SG : BOOL; (*Anforderung Hauptgasventil Sondergas*)
		bDem_PCG_Val : BOOL; (*Anforderung Vorkammergasventil vor Kompressor*)
		bPr_PCG_GC_Dem : BOOL; (*DO	 Demand pre champer gas compressor *) (* OldName: 	A_VKGV	; Cyclic: ; *)
		bPCG_DemReliefValve : BOOL; (*DO	 Demand Relief valve *) (* OldName: 	ENTL_V	; Cyclic: ; *)
		rCnt_Gas_M3 : REAL; (*Gaszähler*)
		rCnt_OpHours : REAL; (* engine operating hours counter *)
		rCnt_Starts : REAL; (* start counter *)
		rCtr_MN_MG_Out_Y : REAL; (* Y- von Regler Gasmischen*)
		rNG_C3H8 : REAL; (*Methane Ergas C3H8*)
		rNG_C4H10 : REAL; (*Methane Ergas C4H10*)
		rNG_C5H12 : REAL; (*Methane Ergas C5H12*)
		rNG_C6H14 : REAL; (*Methane Ergas C6H14*)
		rNG_N2 : REAL; (*Methane Ergas N2*)
		rNG_CH4 : REAL; (*Methane Ergas CH4*)
		rNG_CO2 : REAL; (*Methane Ergas CO2*)
		rNG_C2H6 : REAL; (*Methane Ergas C2H6*)
		rPG_C3H8 : REAL; (*Methane Propangas C3H8*)
		rPG_C4H10 : REAL; (*Methane Propangas C4H10*)
		rPG_C5H12 : REAL; (*Methane Propangas C5H12*)
		rPG_C6H14 : REAL; (*Methane Propangas C6H14*)
		rPG_N2 : REAL; (*Methane Propangas N2*)
		rPG_CH4 : REAL; (*Methane Propangas CH4*)
		rPG_CO2 : REAL; (*Methane Propangas CO2*)
		rPG_C2H6 : REAL; (*Methane Propangas C2H6*)
		rSum_GT_NG_Norm : REAL; (*Berechnete Gasmenge*)
		rGT_CH4_TB : REAL; (*CH4 Regler AO*)
		rGT_CV_TB : REAL; (*Heizwert Regler AO*)
		stGC_CurrentTIME : STRING[6]; (*Momentane Zeit am GC*)
		stGC_CurrentDate : STRING[25]; (*Momentane Datum am GC*)
		stGC_SampleTIME : STRING[6]; (*Probenentnahme Zeit am GC*)
		stGC_SampleDate : STRING[25]; (*Probenentnahme Datum am GC*)
		bGC_Status : BOOL; (*GC Verbindung vorhanden*)
		bMN_Cal_Status : BOOL; (*MethaneZahl Berechnung läuft*)
		bCtr_MN_MG_In_enable : BOOL; (*Regler gasmischen ist aktiv*)
		rMN_MG : REAL; (*Methanezahl Mischgas*)
		rMN_NG : REAL; (*Methanezahl Erdgas*)
		rMN_PG : REAL; (*Methanezahl Propangas*)
		bParaGasMixEngOk : BOOL; (*Parameter abfrage für Gasmischen über Tecjet ok*)
		bParaGasMixMFCOk : BOOL; (*Parameter abfrage für Gasmischen über MFC ok*)
		bBlocGasMixButton : BOOL; (*Blockiert das betätigen Radiobuttons für Gasmischen*)
		bPCG_GV_Open : BOOL; (*Pre chamber gas valves*) (* OldName: 	VKGV	; Cyclic: ; *)
		bGV1_Open : BOOL; (*Open gas valve 1*) (* OldName: 	GASV1	; Cyclic: ; *)
		bGV2_Open : BOOL; (*Open gas valve 2*) (* OldName: 	GASV2	; Cyclic: ; *)
		bGV3_Open : BOOL; (*Open gas valve 3*) (* OldName: 	GASV2	; Cyclic: ; *)
		bEng_Run : BOOL; (* DO engine rotating*)
		rLam_Eng_LL_Set : REAL; (* Leanox Lambda set point *) (* OldName: ssPosGasmixerNominal; Cycle:2; *)
		rGMU_Pos_Valve_Prom1 : REAL; (*Valve Position [%o]*)
		rGMU_Pos_Valve_Prom2 : REAL; (*Valve Position [%o]*)
		rGMU_Pos_Valve_Prom3 : REAL; (*Valve Position [%o]*)
		rCnt_CompOpHours : REAL; (* compressor operating hours counter *)
		bDem_GV_NG_HP : BOOL; (*Anforderung Hauptgasventil Erdgas Hochdruck*)
		bSel_GT_NG_HP : BOOL; (*Anwahl Gasstrecke Erdgas Hochdruck*)
		bMsg7600 : BOOL; (*MSS Druck Gasstrecke Erdgas*)
		bMsg7601 : BOOL; (*MSS Temperatur Gasstrecke Erdgas*)
		bMsg7602 : BOOL; (*MSS Durchfluss Gasstrecke Erdgas*)
		bMsg7603 : BOOL; (*MSS Druck Gasstrecke Propangas*)
		bMsg7604 : BOOL; (*MSS Temperatur Gasstrecke Propangas*)
		bMsg7605 : BOOL; (*MSS Durchfluss Gasstrecke Propangas*)
		bMsg7606 : BOOL; (*MSS Massflow Controller Propangas*)
		bMsg7607 : BOOL; (*MSS Druck Gasstrecke Sondergas*)
		bMsg7608 : BOOL; (*MSS Temperatur Gasstrecke Sondergas*)
		bMsg7609 : BOOL; (*MSS Durchfluss Gasstrecke Sondergas*)
		bMsg7610 : BOOL; (*MSS Massflow Controller Sondergas*)
		bMsg7611 : BOOL; (*MSS Druck Vorkammergastank*)
		bMsg7612 : BOOL; (*Druck min vor Vorkammergaskompressor*)
		bMsg7613 : BOOL; (*Temp. max nach Vorkammergaskompressor*)
		bMsg7614 : BOOL; (*Ölstand min Vorkammergaskompressor*)
		bMsg7615 : BOOL; (*Störung Vorkammergaskompressor*)
		bMsg7616 : BOOL; (*Druck max Vorkammergaskessel*)
		bMsg7617 : BOOL; (*Sum Check Fehler EG*)
		bMsg7618 : BOOL; (*Sum Check Fehler PG*)
		bMsg7619 : BOOL; (*Natural gas methane number plausibility failure*)
		bMsg7620 : BOOL; (*Mixed gas methane number plausibility failure*)
		bMsg7621 : BOOL; (*Propan gas methane number plausibility failure*)
		bMsg7622 : BOOL; (*Wartung Gaskompressor*)
		bMsg7623 : BOOL; (*MSS LSCS Gasventil*)
		bMsg7624 : BOOL; (*MSS LSCS Mischgasventil*)
		rU_CtrlBat1 : REAL; (*AI Control battery 1 voltage*)
		rU_CtrlBat_BatTest1 : REAL; (*Control battery 1 voltage last measurement*)
		rLevel_Oiltank : REAL; (*Stand Öltank*)
		rLevel_OilNorm : REAL; (*Stand Öltank %*)
		bCtrlBatMon_TestRunning : BOOL; (*Status battery test*)
		bReq_RefillOilPuEng : BOOL; (*Anforderung Nachfüll Ölpumpe Motor DI von +M*)
		bDem_RefillOilPuEng : BOOL; (*Anforderung Nachfüll Ölpumpe Motor DO*)
		bPreHeatWDay_On : BOOL; (*Einschalten der Vorwärmung über Zeitsteuerung*)
		stTB_Version : STRING[6]; (*Versionsanzeige von TB_Control*)
		bServicePageActive : BOOL; (* Aktivierung der Service Seite auf der Visualisierung *)
		bAirCompressor1_Run : BOOL; (*Air compressor 1 run*)
		bAirCompressor2_Run : BOOL; (*Air compressor 2 run*)
		bMsg7700 : BOOL; (*Control battery voltage low*)
		bMsg7701 : BOOL; (*Control battery charging device malfunction*)
		bMsg7702 : BOOL; (*Sicherungsfall 24VDC Stützpunkt (+A)*)
		bMsg7703 : BOOL; (*Sicherungsfall 24VDC Stützpunkt (+AUX)*)
		bMsg7704 : BOOL; (*transformer failure*)
		bMsg7705 : BOOL; (*transformer Warning*)
		bMsg7706 : BOOL; (*Störung Nachfüllölpumpe Tank*)
		bMsg7707 : BOOL; (*Störung Nachfüllölpumpe Motor*)
		bMsg7708 : BOOL; (*Messsignalstörung Stand Öltank*)
		bMsg7709 : BOOL; (*Min Stand Öltank*)
		bMsg7710 : BOOL; (*Ruhestromschleife unterbrechen, Motor wurde durch Prüfstand nicht abgestellt*)
		bMsg7711 : BOOL; (*Inselbetrieb darf nicht angefordert werden da 24V bei GCB-Steuerung anliegt*)
		bMsg7712 : BOOL; (*Abstellung Zylinderdrucküberwachung*)
		bMsg7713 : BOOL; (*IO Kanäle Fehler +A*)
		bMsg7714 : BOOL; (*IO Kanäle Fehler +AUX*)
		bMsg7715 : BOOL; (*IO Kanäle Fehler +APSCRV*)
		bMsg7716 : BOOL; (*IO Kanäle Fehler +TK*)
		bMsg7717 : BOOL; (*IO Kanäle Fehler +PUMA*)
		bMsg7718 : BOOL; (*IO Kanäle Fehler Reserve*)
		bMsg7719 : BOOL; (*IO Kanäle Fehler Reserve*)
		bMsg7720 : BOOL; (*IO Kanäle Fehler Reserve*)
		bMsg7721 : BOOL; (*Brandmelder deaktiviert*)
		bMsg7722 : BOOL; (*Bufferbatteriespannung max*)
		bMsg7723 : BOOL; (*Dauerlauftest beendet*)
		bMsg7724 : BOOL; (*Störung Druckluft*)
		bMsg7725 : BOOL; (*Störung Kamerasystem*)
		bMsg7726 : BOOL; (*Störung Durchdrehvorrichtung*)
		bMsg7727 : BOOL; (*Verbindung CAN-Schiene 1 zu PUMA unterbrochen*)
		bMsg7728 : BOOL; (*Verbindung CAN-Schiene 2 zu PUMA unterbrochen*)
		bMsg7729 : BOOL; (*Störung Gaswarnanlage (GWA)*)
		bMsg7730 : BOOL; (*Ölstand min Transformator*)
		bMsg7731 : BOOL; (*Ölstand max Transformator*)
		bMsg7732 : BOOL; (*Warnung Buchholzschutz Transformator*)
		bMsg7733 : BOOL; (*Störung Buchholzschutz Transformator*)
		bMsg7734 : BOOL; (*Warnung Temperatur max Transformator*)
		bMsg7735 : BOOL; (*Störung Temperatur max Transformator*)
		bMsg7736 : BOOL; (*Sicherungsfall 230VAC Stützpunkt (+AUX)*)
		bMsg7737 : BOOL; (* Sicherungsfall 24VDC Stützpunkt (+HMC)*)
		bMsg7738 : BOOL; (* Sicherungsfall 230VAC Stützpunkt (+HMC)*)
		bMsg7739 : BOOL; (* Füllstand Kühlwassertank max*)
		bMsg7740 : BOOL; (*Sicherungsfall 230VAC Stützpunkt (+A)*)
		bMsg7741 : BOOL; (*IO Kanäle Fehler +TK HT 2*)
		bMsg7742 : BOOL; (*IO Kanäle Fehler +TK HT 3*)
		bMsg7743 : BOOL; (*IO Kanäle Fehler +TK HT 4*)
		bMsg7744 : BOOL; (*IO Kanäle Fehler +TK HT 5*)
		bMsg7745 : BOOL; (*IO Kanäle Fehler +TK OKW 1*)
		bMsg7746 : BOOL; (*IO Kanäle Fehler +TK OKW 2*)
		bMsg7747 : BOOL; (*IO Kanäle Fehler +TK OKW 3*)
		bMsg7748 : BOOL; (*IO Kanäle Fehler +TK MKW 1*)
		bMsg7749 : BOOL; (*IO Kanäle Fehler +TK MKW 2*)
		bMsg7750 : BOOL; (*IO Kanäle Fehler +TK MKW 3*)
		bMsg7751 : BOOL; (*IO Kanäle Fehler +TK MKW 4*)
		bMsg7752 : BOOL; (*IO Kanäle Fehler +TK NT 1*)
		bMsg7753 : BOOL; (*IO Kanäle Fehler +TK NT 2*)
		bMsg7754 : BOOL; (*IO Kanäle Fehler +TK NT 3*)
		bMsg7755 : BOOL; (*IO Kanäle Fehler +TK NT 4*)
		bMsg7756 : BOOL; (*IO Kanäle Fehler +TK NT 5*)
		bMsg7757 : BOOL; (*emergency stop push button - help module control*)
		bMsg7758 : BOOL; (*emergency stop push button - auxiliaries control*)
		bMsg7759 : BOOL; (*emergency stop push button - control room ventilation*)
		bMsg7760 : BOOL; (*emergency stop push button - table cooler*)
		bMsg7761 : BOOL; (*IO Kanäle Fehler +APSPH!*)
		bMsg7762 : BOOL; (*Störung Luftkompressor 1*)
		bMsg7763 : BOOL; (*Hauptschalter Luftkompressor 1 ausgeschaltet*)
		bMsg7764 : BOOL; (*Störung Luftkompressor 2*)
		bMsg7765 : BOOL; (*Hauptschalter Luftkompressor 2 ausgeschaltet*)
		bMsg7766 : BOOL; (*Störung Gerätedruckluft*)
		bMsg7767 : BOOL; (*Störung Niederspannungs Leistungsschalter*)
		bMsg7768 : BOOL; (**)
		bMsg7769 : BOOL; (**)
		bMsg7770 : BOOL; (**)
		bMsg7771 : BOOL; (**)
		bMsg7772 : BOOL; (**)
		bMsg7773 : BOOL; (**)
		bMsg7774 : BOOL; (**)
		bMsg7775 : BOOL; (**)
		bMsg7776 : BOOL; (**)
		bMsg7777 : BOOL; (**)
		bMsg7778 : BOOL; (**)
		bMsg7779 : BOOL; (**)
		bMsg7780 : BOOL; (**)
		bMsg7781 : BOOL; (**)
		bMsg7782 : BOOL; (**)
		bMsg7783 : BOOL; (**)
		bMsg7784 : BOOL; (**)
		bMsg7785 : BOOL; (**)
		bMsg7786 : BOOL; (**)
		bMsg7787 : BOOL; (**)
		bMsg7788 : BOOL; (**)
		bMsg7789 : BOOL; (**)
		bMsg7790 : BOOL; (**)
		bMsg7791 : BOOL; (**)
		bMsg7792 : BOOL; (**)
		bMsg7793 : BOOL; (**)
		bMsg7794 : BOOL; (**)
		bMsg7795 : BOOL; (**)
		bMsg7796 : BOOL; (**)
		bMsg7797 : BOOL; (**)
		bMsg7798 : BOOL; (**)
		bMsg7799 : BOOL; (**)
		tGasconsumMonth : ARRAY[0..12]OF GasconsumM; (*Gasverbrauch pro Monat*)
		tGasconsumYear : ARRAY[0..9]OF GasconsumY; (*Gasverbrauch pro Jahr*)
		bCV_Bus_Active : BOOL; (* Bus - CV content measuring active *)
		bRelAux_TB : BOOL; (*Anforderung Hilfsbetriebe für Prüfstand*)
		bOPC_Dem : BOOL; (* Externe Anforderung Motor vom Prüfstand*)
		bBusAlive : BOOL; (*Verbindung Prüfstand zu Motor über OPC Impuls*)
		rP_OPC_Set : REAL; (*Power setpoint from OPC [%]*)
		rVol_NG : REAL; (* ratio natural gas volumetric *)
		rVol_PG : REAL; (* ratio propan gas volumetric *)
		rVol_SG : REAL; (* ratio propan gas volumetric *)
		rVol_NG_PG : REAL; (* volumetric ratio natural gas & propan gas combined*)
		iIdx_OMSS : INT; (* index of operation mode selector switch - 0..OFF, 1..MAN, 2..AUTO, 3..TEST, 4..SCAVENGING *) (*OldName:new PV;Cycle:2;*)
		bMixAllTrains : BOOL; (* all gastrains used *)
		bEndurTestEnd : BOOL; (*Dauerlauftest Ende*)
		stEndurTestDate : STRING[11]; (*Dauerlauftest Datum wann beendet*)
		stEndurTestTime : STRING[5]; (*Dauerlauftest Uhrzeit wann beendet*)
		bOptGT_RatioMix_Set : BOOL; (*activation bit for custom gasmixing ratio setpoint*)
		rGT_RatioMix_Set : REAL; (*custom gasmixing ratio setpoint*)
		iIdx_SelGasTyp : INT; (* index of selcted gastype*)
		iIdx_Gtyp_Act : INT; (*Actual gassort for VISU display*) (* OldName: ucGasType; Cyclic: ; *)
		bRelMixGas : BOOL; (*Release Mixgas for VISU display*)
		rStartpointCA_IgnP_Set : REAL; (*Startwert von dem Zündzeitpunkt*)
		rStartpointLamEngLL_Set : REAL; (*Startwert von dem Lamda*)
		rStartpoint_p2_Set : REAL; (*Startwert von dem p2'*)
		rStartpoint_MN_Set : REAL; (*Startwert von der MZ*)
		rCA_IgnP_CylOffset : ARRAY[0..24]OF REAL; (*ZZP Vorgabe mit Offset zu Motorsteuerung*)
		bLeanox_Man_Cust : BOOL; (*Aktivierung ext Lambda/p2' Vorgabe*)
		rLam_Eng_LL_ManSet_Cust : REAL; (*Ext Lambda Vorgabe*)
		rPr_Leanox_ManSet_Cust : REAL; (*Ext p2' Vorgabe*)
		bCA_IgnP_CylOffset_Active : BOOL; (*Aktivierung ext ZZP Vorgabe*)
		bExtMN_Active : BOOL; (*Aktivierung ext MN Vorgabe von PUMA zur Prüfstandssteuerung*)
		rExtMN_Set : REAL; (*Sollwert für MN von PUMA*)
		rPr_Ch_P2s_Avg : REAL; (*Ladedruck (p2') - mittel*)
		rCA_IgnP_Set : REAL; (* ignitoin timing set point *)
		bGEN2_preM_Act : BOOL; (* GEN2 controller active pre-mixed engines *)
		bExtLeanoxFromMDE : BOOL; (*Leanoxvorgabe von MDE aktiv*)
		bCA_IgnPFromMDE : BOOL; (*ZZP von MDE aktiv*)
		rCA_IgnPFromMDE : REAL; (*ZZP von MDE Sollwert*)
		rStartpoint_NOX_Set : REAL; (*Startwert NOX mg/Nm³*)
		rNOX_ManSet_Cust : REAL; (*Ext NOX mg/Nm³ Vorgabe*)
		bExtMNFromMDE : BOOL; (*MZ von MDE aktiv*)
		bExtNOXFromMDE : BOOL; (*NOX von MDE aktiv*)
		bExtNOX_Active : BOOL; (*Aktivierung NOX Vorgabe von MDE über CAN*)
		rNOX_FromMDE : REAL; (*Momentanen NOX mg/Nm³ von PUMA*)
		rStatusExhaustMde : REAL; (*Status Abgasmessanlage*)
		rCA_Ign_Avg : REAL; (*aCtual ignition point average*)
		bMsg7625 : BOOL; (*Measuring signal failure pressure special gas H2*)
		bMsg7626 : BOOL; (*Alarm: Pressure minimum special gas H2*)
		bMsg7627 : BOOL; (*Pressure maximum special gas H2*)
		bMsg7628 : BOOL; (*Warning: Pressure minimum special gas H2*)
		bMsg7629 : BOOL; (*H2 special gas flow maximum*)
		bMsg7630 : BOOL; (*Measuring signal failure gastemperature after prechamber gascompressor*)
		bMsg7631 : BOOL; (*Measuring signal failure gastemperature after cooler prechamber gascompressor*)
		bMsg7632 : BOOL; (*Gas temperature after prechamber gascompressor maximum*)
		bMsg7633 : BOOL; (*Gas temperature after cooler prechamber gascompressor maximum*)
		bMsg7634 : BOOL; (*Gas temperature-switch after prechamber gascompressor maximum*)
		bMsg7635 : BOOL; (*Measuring signal failure contact sensor 1 butan gastrain*)
		bMsg7636 : BOOL; (*Measuring signal failure contact sensor 2 butan gastrain*)
		bMsg7637 : BOOL; (*Measuring signal failure tank pressure propangas compressor tank pressure*)
		bMsg7638 : BOOL; (*Pressure max propangas compressor tank*)
		bMsg7639 : BOOL; (*FC not ready propangas compressor*)
		bMsg7640 : BOOL; (*Pressure switch low triggered propangas compressor*)
		bMsg7641 : BOOL; (*Temperature switch high cooling water triggered propangas compressor*)
		bMsg7642 : BOOL; (*Pressure switch high triggered propangas compressor*)
		bMsg7643 : BOOL; (*Temperature switch high triggered propangas compressor*)
		bMsg7644 : BOOL; (*Pressure switch low oil triggered propangas compressor*)
		bMsg7645 : BOOL; (*Measuring signal failure pressure propangas after compressor cooler*)
		bMsg7646 : BOOL; (*Measuring signal failure temperature propangas compressor tank*)
		bMsg7647 : BOOL; (*Temperature of compressor tank to low for propangas operation*)
		bMsg7648 : BOOL;
		bMsg7649 : BOOL;
		bMsg7650 : BOOL;
		bMsg7651 : BOOL; (*Sicherungsfall Vorkammergasverdichter Venitle 24V*)
		bMsg7652 : BOOL;
		bMsg7653 : BOOL;
		bMsg7654 : BOOL;
		bMsg7655 : BOOL;
		bMsg7656 : BOOL;
		bMsg7657 : BOOL;
		bMsg7658 : BOOL;
		bMsg7659 : BOOL;
		bMsg7660 : BOOL;
		rH2_Act_Cube : REAL; (*Actual volume H2 content measurement cube*)
		rGT_H2 : REAL; (* Filtered H2 content [%]  (engine sensor)*)
		rT_PCGAfComp : REAL; (*Messung Temperatur Vorkammergas nach Kompressor*)
		rT_PCGAfCooler : REAL; (*Messung Temperatur Vorkammergas nach Kühler*)
		bMFC_PG_open_vis : BOOL; (*Visulaization MFC propan gas open*)
		bMFC_SG_open_vis : BOOL; (*Visulaization MFC special gas open*)
		bDem_TraceHeating_BG : BOOL; (*Demand trace heating butan gastrain*)
		rT_GT_BG1 : REAL; (*Butan gastrain contact sensor 1*)
		rT_GT_BG2 : REAL; (*Butan gastrain contact sensor 2*)
		bMX_Status : BOOL; (*Mixedmode Status*)
		rCust_TB2Eng : ARRAY[0..50] OF REAL; (*Customized variables from Testbench to Engine*)
		bDem_Cooler_X : BOOL; (*visu aktiv Anforderung Kühler OKW 3 MKW 3-4 HT 3-5 NT 3-5*)
		rPr_PG_CompTank : REAL; (*Messung Propangas Kesseldruck*)
		rPr_PG_AfterComp : REAL; (*Messung Druck nach Propangasverdichter*)
		rT_PG_CompCW : REAL; (*Messung Temperatur Kühlwasser Propangasverdichter*)
		rT_PG_BeforeComp : REAL; (*Messung Temperatur vor Propangasverdichter*)
		rT_PG_AfterComp : REAL; (*Messung Temperatur nach Propangasverdichter*)
		rT_PG_Tank : REAL; (*Messung Temperatur Anlegefühler am Tank vom Propangasverdichter*)
		rCtr_PG_Comp : REAL; (*Propangasverdichter Regler*)
		rCtr_PG_CompCool : REAL; (*Propangasverdichter Kühlwasserventil Regler*)
		bPG_TraceHeat_TimeCtr_On : BOOL; (*Time controller set PG trace heating on*)
		bDem_PG_TraceHeat : BOOL; (*Anforderung Begleitheizung Propangaskompressor*)
		bDem_PG_Comp_FC : BOOL; (*Anforderung FU Propangaskompressor*)
		bDem_PG_CompValCW : BOOL; (*Anforderung Kühlwasserventil Propangaskompressor*)
		rPr_NG_bValve : REAL; (*Messung Druck Erdgas vor GWA-Ventil/Hauptventil*)
		rPr_PG_bValve : REAL; (*Messung Druck Propangas vor GWA-Ventil/Hauptventil*)
		rPr_GasAfterTempCtr : REAL; (*Messung Druck Gas nach Temperaturregelung*)
		rT_GasAfterTempCtr : REAL; (*Messung Temperatur Gas nach Temperaturregelung*)
		rT_GasAfterMixer : REAL; (*Messung Temperatur nach Sulzer Mischer*)
		rI_Aux : REAL; (*Electrical current of Auxiliaries*)
		rP_Aux : REAL; (*Electrical power of Auxiliaries*)
		bSA_PI_Active : BOOL; (*PARA [12120]: TRUE = SAFI port injection is enabled/active *)
		rCA_PI_Dur_Avg : REAL; (* Port Injection Duration average *)
		rCAT_TempSet : REAL; (*CAT temp setpoint from Engine*)
		bExtCAT_TempActiveMDE : BOOL; (*Extern CAT temp setpoint from MDE active*)
		rExtCAT_TempSetMDE : REAL; (*Extern CAT temp setpoint from MDE*)
		rExtCAT_TempSet : REAL; (*Extern CAT temp setpoint to Visu*)
		bExtCAT_TempStatus_Active : BOOL; (*Extern CAT temp setpoint to Visu active*)
		rStartpoint_CAT_Temp_Set : REAL; (*Startpoint CAT temp setpoint to Visu*)
		rT_HW_Air_Re_2 : REAL; (*Temperatur Rücklauf Heizkreis 2*)
		rT_HW_Air_Su_2 : REAL; (*Temperatur Vorlauf Heizkreis 2*)
		rT_Cool_Air_Re_2 : REAL; (*Temperatur Rücklauf Kühlkreis 2*)
		rT_Cool_Air_Su_2 : REAL; (*Temperatur Vorlauf Kühlkreis 2*)
		bT_HW_Air_2_Active : BOOL; (*Temperatur Heizkreis 2 aktiv*)
		bT_Cool_Air_2_Active : BOOL; (*Temperatur Kühlkreis 2 aktiv*)
		rPr_HR_HT_Su : REAL; (*Druck Wärmeschiene HT Vorlauf (heat recovery system)*)
		rPr_HR_HT_Re : REAL; (*Druck Wärmeschiene HT Rücklauf (heat recovery system)*)
		rPr_HR_LT_Su : REAL; (*Druck Wärmeschiene NT Vorlauf (heat recovery system)*)
		rPr_HR_LT_Re : REAL; (*Druck Wärmeschiene NT Rücklauf (heat recovery system)*)
		rT_HR_HT_Su : REAL; (* Temperatur HT Vorlauf (heat recovery system) *)
		rT_HR_HT_Re : REAL; (* Temperatur HT Rücklauf (heat recovery system) *)
		rT_HR_LT_Su : REAL; (* Temperatur LT Vorlauf (heat recovery system) *)
		rT_HR_LT_Re : REAL; (* Temperatur LT Rücklauf (heat recovery system) *)
		rT_HR_HT_LP_Su : REAL; (* Temperatur HT ND Vorlauf (heat recovery system) *)
		rT_HR_HT_LP_Re : REAL; (* Temperatur HT ND Rücklauf (heat recovery system) *)
		rT_HR_HT_HP_Su : REAL; (* Temperatur HT HD Vorlauf (heat recovery system) *)
		rT_HR_HT_HP_Re : REAL; (* Temperatur HT HD Rücklauf (heat recovery system) *)
		rT_HR_LT_LP_Su : REAL; (* Temperatur LT ND Vorlauf (heat recovery system) *)
		rT_HR_LT_LP_Re : REAL; (* Temperatur LT ND Rücklauf (heat recovery system) *)
		rT_HR_LT_HP_Su : REAL; (* Temperatur LT HD Vorlauf (heat recovery system) *)
		rT_HR_LT_HP_Re : REAL; (* Temperatur LT HD Rücklauf (heat recovery system) *)
		rT_HR_ECW_Su : REAL; (* Temperatur MKW Vorlauf (heat recovery system) *)
		rT_HR_ECW_Re : REAL; (* Temperatur MKW Rücklauf (heat recovery system) *)
		rT_HR_OCW_Su : REAL; (* Temperatur OKW Vorlauf (heat recovery system) *)
		rT_HR_OCW_Re : REAL; (* Temperatur OKW Rücklauf (heat recovery system) *)
		bDem_HR_CircPump_HT_1 : BOOL; (*Anforderung Wärmeschiene HT 1 Zirkulationspumpe (heat recovery system)*)
		bDem_HR_CircPump_HT_2 : BOOL; (*Anforderung Wärmeschiene HT 2 Zirkulationspumpe (heat recovery system)*)
		bDem_HR_CircPump_LT_1 : BOOL; (*Anforderung Wärmeschiene LT 1 Zirkulationspumpe (heat recovery system)*)
		bDem_HR_CircPump_LT_2 : BOOL; (*Anforderung Wärmeschiene LT 2 Zirkulationspumpe (heat recovery system)*)
		bDem_HR_CircPump_ECW_1 : BOOL; (*Anforderung Wärmeschiene MKW 1 Zirkulationspumpe (heat recovery system)*)
		bDem_HR_CircPump_ECW_2 : BOOL; (*Anforderung Wärmeschiene MKW 2 Zirkulationspumpe (heat recovery system)*)
		bDem_HR_CircPump_OCW_1 : BOOL; (*Anforderung Wärmeschiene OKW 1 Zirkulationspumpe (heat recovery system)*)
		bDem_HR_CircPump_OCW_2 : BOOL; (*Anforderung Wärmeschiene OKW 2 Zirkulationspumpe (heat recovery system)*)
		rT_HR_InAirCool_Su : REAL; (*Temperatur Vorlauf Wärmeschiene (Heat recovery system)*)
		rT_HR_InAirCool_Re : REAL; (*Temperatur Rücklauf Wärmeschiene (Heat recovery system)*)
		rCtr_HR_InAirCool : REAL; (*Sollwert Regelventil Motor Frischluft Wärmeschiene (Heat recovery system)*)
		bDem_PumpInAirCool : BOOL; (*Anforderung Motor Frischluft Kühlkreis Pumpe*)
		bDem_HR_CircPump_InAir : BOOL; (*Anforderung Pumpe Motor Frischluft Wärmeschiene (Heat recovery system)*)
		bDem_PCG_Tank_FillValve : BOOL; (*Anforderung Vorkammergas Tank Füllventil*)
		bDem_PCG_Tank_OpValve : BOOL; (*Anforderung Vorkammergas Tank Ventil Normalbetrieb*)
		bPCG_Comp_CV_Mech_Active : BOOL; (*PCG compressor Mechanical regulating valve*)
		bPCG_MG_Valve_Inactive : BOOL; (*Pre chumber gas mixing gas valve inactive*)
		bSingle_H2_GT : BOOL; (*Single H2 gastrain active, for 100% H2*)
		rT_PCG_CW_Re : REAL; (*Messung Temperatur Verdichter Kühlwasser Rücklauf*)
		rT_PCG_CW_Su : REAL; (*Messung Temperatur Verdichter Kühlwasser Vorlauf*)
		rPr_PCG_CW : REAL; (*Messung Druck Verdichter Kühlwasser *)
		bPCG_DemValCW: BOOL; (*Prechambergascompressor,Demandcoolingwatervalve*)
		rPos_InlLou3 : REAL; (*AI position air inlet louver 3 [%]*)
		rPos_InlLou4 : REAL; (*AI position air inlet louver 4 [%]*)
		rPos_InlLou5 : REAL; (*AI position air inlet louver 5 [%]*)
		rPos_InlLou6 : REAL; (*AI position air inlet louver 6 [%]*)
		rCtr_AuxRoom_Fan_FC : REAL; (*Sollwert Regelventil Motor Frischluft Hilfsbetriebsraum *)
		rT_AuxRoom : REAL; (*Temperatur Hilfsbetriebsraum*)
		bAuxRoom_InLouOpened : BOOL; (*DI Rückmeldung Zuluftjalousie Hilfsbetriebsraum  offen *)
		bDem_Fan_AuxRoom : BOOL; (*Anforderung Frequenzumrichter Zuluftventilator Hilfsbetriebsraum*)
	END_STRUCT;
	VIS2MM_DI_struct : 	STRUCT
		tCtr_ChCW_LT_In : _tGeACtrIn; (*charge cooler*)
		tCtr_ChCW_HT_In : _tGeACtrIn; (*charge cooler*)
		tCtr_ChCW_HT_LP_In : _tGeACtrIn; (*charge cooler*)
		tCtr_ChCW_HT_HP_In : _tGeACtrIn; (*charge cooler*)
		tCtr_ChCW_LT_LP_In : _tGeACtrIn; (*charge cooler*)
		tCtr_ChCW_LT_HP_In : _tGeACtrIn; (*charge cooler*)
		tCtr_ECW_In : _tGeACtrIn; (*engine cooling water cooler*)
		tCtr_OCW_In : _tGeACtrIn; (*oil cooling water cooler*)
		bECW_PreH_Dem_Customized : BOOL;
		rCtr_RW_CV_Set : REAL; (*Vorgabe Kühlkreis Regelventil Rohwassser skaliert*)
		rCtr_RW_HE_Set : REAL; (*Vorgabe Kühlkreis Regelventil Rohwasser Wärmetauscher skaliert*)
		rCtr_RW_LT_1_Set : REAL; (*Vorgabe Regelventil Rohwasser NT*)
		rCtr_RW_HT_1_Set : REAL; (*Vorgabe Regelventil Rohwasser HT*)
		rCtr_RW_LT_2_Set : REAL; (*Vorgabe Regelventil Rohwasser NT*)
		rCtr_RW_HT_2_Set : REAL; (*Vorgabe Regelventil Rohwasser HT*)
		rCtr_RW_ECW_1_Set : REAL; (*Vorgabe Regelventil Rohwasser Motorkühlwasser*)
		rCtr_RW_OCW_1_Set : REAL; (*Vorgabe Regelventil Rohwasser Ölkühlwasser*)
		rCtr_RW_ECW_2_Set : REAL; (*Vorgabe Regelventil Rohwasser Motorkühlwasser*)
		rCtr_RW_OCW_2_Set : REAL; (*Vorgabe Regelventil Rohwasser Ölkühlwasser*)
		rFC_ChCW_LT_PuSet : REAL; (*FU Sollwert Ladekühwasser Niedertemp. Pumpe skaliert*)
		rFC_ChCW_HT_PuSet : REAL; (*FU Sollwert Ladekühwasser Hochtemp. Pumpe skaliert*)
		rFC_ChCW_LT_LP_PuSet : REAL; (*FU Sollwert Ladekühwasser Niedertemp. Niederdruck Pumpe skaliert*)
		rFC_ChCW_LT_HP_PuSet : REAL; (*FU Sollwert Ladekühwasser Niedertemp. Hochdruck Pumpe skaliert*)
		rFC_ChCW_HT_LP_PuSet : REAL; (*FU Sollwert Ladekühwasser Hochtemp. Niederdruck Pumpe skaliert*)
		rFC_ChCW_HT_HP_PuSet : REAL; (*FU Sollwert Ladekühwasser Hochtemp. Hochdruck Pumpe skaliert*)
		rFC_ECW_PuSet : REAL; (*FU Sollwert Motorkühlwasser Pumpe skaliert*)
		rFC_OCW_PuSet : REAL; (*FU Sollwert Ölkühlwasser Pumpe skaliert*)
		tCtr_ER_In : _tGeACtrIn; (*engine cooling water cooler*)
		tCtr_OutlVE_RDP_In : _tGeACtrIn; (*oil cooling water cooler*)
		tCtr_IntakeAir_In : _tGeACtrIn; (*cooling water cooler*)
		rOp_ExhFlap : REAL; (*Auswahl der Abgasverarbeitung*)
		rMan_DPF_EgFlap_Set : REAL; (*Manuelle Vorage für DPF Abgasklappe*)
		rMan_DPF_ByFlap_Set : REAL; (*Manuelle Vorage für DPF Bypassklappe*)
		rMan_SRC_EgFlap_Set : REAL; (*Manuelle Vorage für SCR Abgasklappe*)
		rMan_SRC_ByFlap_Set : REAL; (*Manuelle Vorage für SCR Bypassklappe*)
		rMan_EG_Flap_Set : REAL; (*Manuelle Vorgabe für Abgasklappe*)
		rCust_Eng2TB : ARRAY[0..50] OF REAL; (*Customized variables from Engine to Testbench*)
		tCtr_EG_Flap_In : _tGeACtrIn; (*Abgasklppenregler*)
		rCtr_EG_Flap : REAL; (*Anwahl der Abgasklappen*)
		tCtr_GC_1_In : _tGeACtrIn; (*Gaskompressorregler*)
		tCtr_GC_2_In : _tGeACtrIn; (*Gaskompressorregler*)
		bCtrlBatMon_ManTestStart : BOOL; (*Manual request for start of control battery test*)
		tCtr_MN_MG_In : _tGeACtrIn; (*Para Gas mischen regler*)
		bMN_MG_active : BOOL; (*Mischung aktiv*)
		bDemDataMan_GC : BOOL; (*Anforderung manuelle Daten auslesen vom GC*)
		bCtr_MN_MG_active : BOOL; (*Gas Misch Regler aktivieren*)
		bCtr_MN_MG_off : BOOL := TRUE; (* mixgas operation off *)
		bVolPG_Man : BOOL; (* activate MFC controller for add mixing *)
		rVol_PG_Set : REAL; (* setpoint for volumetric add mixing propan gas *)
		rVol_SG_Set : REAL; (* setpoint for volumetric add mixing special gas *)
		bMan_ECW_Pump : BOOL; (* Manuelle Anforderung der Kühlwasserpumpe vom Prüfstand *)
		bMan_OCW_Pump : BOOL; (* Manuelle Anforderung der Kühlwasserpumpe vom Prüfstand *)
		bMan_LT_Pump : BOOL; (* Manuelle Anforderung der Kühlwasserpumpe vom Prüfstand *)
		bMan_HT_Pump : BOOL; (* Manuelle Anforderung der Kühlwasserpumpe vom Prüfstand *)
		bMan_LT_LP_Pump : BOOL; (* Manuelle Anforderung der Kühlwasserpumpe vom Prüfstand *)
		bMan_LT_HP_Pump : BOOL; (* Manuelle Anforderung der Kühlwasserpumpe vom Prüfstand *)
		bMan_HT_LP_Pump : BOOL; (* Manuelle Anforderung der Kühlwasserpumpe vom Prüfstand *)
		bMan_HT_HP_Pump : BOOL; (* Manuelle Anforderung der Kühlwasserpumpe vom Prüfstand *)
		bEndurTestStart : BOOL; (*Dauerlauftest Start*)
		rEndurTestTimeSet : REAL; (*Dauerlauftest h-Vorgabe*)
		iSelExtP_OPC_Set : INT; (*Auswahl der externen Leistungsvorgabe über OPC*)
		bExtLeanox_ActiveMDE : BOOL; (*Aktivierung externe Leanox Regelung über MDE, kommt über Visu-Button*)
		bCA_IgnP_ActiveMDE : BOOL; (*Aktivierung externe ZZP Regelung über MDE, kommt über Visu-Button*)
		bExtMN_ActiveMDE : BOOL; (*Aktivierung externe MN Regelung über MDE, kommt über Visu-Button*)
		bExtNOX_ActiveMDE : BOOL; (*Aktivierung externe NOX Regelung über MDE, kommt über Visu-Button*)
		bDem_ERV_Aut_Vis : BOOL; (*Anforderung Lüftung Motorraum Automatik von Visu*)
		bMan_BoilerHouse_Pump : BOOL; (* Manuelle Anforderung der Heizhauskreispumpe vom Prüfstand *)
		bMan_SecCirc_Pump : BOOL; (* Manuelle Anforderung der Sekundärkreispumpe vom Prüfstand *)
		bManCircLouActive : BOOL; (*Manuelle Vorgabe Umluftjalousie aktiv*)
		bManCircLouEngActive : BOOL; (*Manuelle Vorgabe Umluftjalousie Motor aktiv*)
		bManDem_PCG_Val : BOOL; (*Manuelle Vorgabe Vorkammergasventil*)
		bManFV_PCGC_MG : BOOL; (*Manuelle Vorgabe Füllventil Vorkammergaskompressor*)
		bManGV_Active : BOOL; (*Manuelle Vorgabe Gasventile aktiv*)
		bManGV_NG_Set : BOOL; (*Manuelle Vorgabe Erdgasventil*)
		bManGV_PG_Set : BOOL; (*Manuelle Vorgabe Propangasventil*)
		bManGV_SG_Set : BOOL; (*Manuelle Vorgabe Sondergasventil*)
		bManInAirFanActive : BOOL; (*Manuelle Vorgabe Zuluftventilator aktiv*)
		bManInEngAirFanActive : BOOL; (*Manuelle Vorgabe Zuluftventilator Motor aktiv*)
		bManInlLouActive : BOOL; (*Manuelle Vorgabe Zuluftjalousie aktiv*)
		bManInlLouEngActive : BOOL; (*Manuelle Vorgabe Zuluftjalousie Motor aktiv*)
		bManInlLouRoomActive : BOOL; (*Manuelle Vorgabe Zuluftjalousie Raum aktiv*)
		bManOutAirFanActive : BOOL; (*Manuelle Vorgabe Abluftventilator aktiv*)
		bManOutlLouActive : BOOL; (*Manuelle Vorgabe Abluftjalousie aktiv*)
		bManPCG_Comp_Active : BOOL; (*Manuelle Vorgabe Vorkammergaskompressor aktiv*)
		bManPCG_DemCoolFan : BOOL; (*Manuelle Vorgabe Vorkammergasverdichter Ventilator*)
		bManPCG_DemReliefValve : BOOL; (*Manuelle Vorgabe Vorkammergasverdichter Entlastungsventil*)
		bManPCG_DemValCW : BOOL; (*Manuelle Vorgabe Vorkammergasverdichter Wasserventil*)
		bManPCG_GC_Dem : BOOL; (*Manuelle Vorgabe Vorkammergaskompressor*)
		bManPCG_GV_MG_Set : BOOL; (*Manuelle Vorgabe Vorkammergasventil Mischgas*)
		bManPCG_GV_NG_Set : BOOL; (*Manuelle Vorgabe Vorkammergasventil Erdgas*)
		bManPCG_GV_PG_Set : BOOL; (*Manuelle Vorgabe Vorkammergasventil Propangas*)
		rManCircLouEngSet : REAL; (*Manuelle Vorgabe Umluftjalousie Motor*)
		rManCircLouSet : REAL; (*Manuelle Vorgabe Umluftjalousie*)
		rManInAirFanSet : REAL; (*Manuelle Vorgabe Zuluftventilator*)
		rManInEngAirFanSet : REAL; (*Manuelle Vorgabe Zuluftventilator Motor*)
		rManInlLouEngSet : REAL; (*Manuelle Vorgabe Zuluftjalousie Motor*)
		rManInlLouRoomSet : REAL; (*Manuelle Vorgabe Zuluftjalousie Raum*)
		rManInlLouSet : REAL; (*Manuelle Vorgabe Zuluftjalousie*)
		rManOutAirFanSet : REAL; (*Manuelle Vorgabe Abluftventilator*)
		rManOutlLouSet : REAL; (*Manuelle Vorgabe Abluftjalousie*)
		tPreHeatWDayLT : ARRAY[0..7]OF PreHeatWDay; (*Variablen für die Zeitsteuerung*)
		bPreHeatWDayLT_CtrActive : BOOL; (*Allgemeine Aktivierung der Zeitsteurerung*)
		bLT_PreH_Dem : BOOL; (*Niedertemp. Vorwärmung aktiv*)
		rT_LT_HP_Preh : REAL; (*Temp. preheating setpoint for LT HP*)
		rT_LT_LP_Preh : REAL; (*Temp. preheating setpoint for LT HP*)
		bSel_PG_Comp : BOOL; (*Anwahl Propangasverdichter aktiv von Visu*)
		bSel_PG_TraceHeat : BOOL; (*Anwahl Propangas Begleitheiung aktiv von Visu*)
		bSel_PG_TraceHeat_TimeCtr : BOOL; (*Time controller of PG trace heating active*)
		rCtr_PG_CompSet : REAL; (*FU Setpoint for propangas verdichter*)
		rCtr_GasTempSet : REAL; (*Temperature setpoint for gas boiler*)
		bExtCAT_TempActive : BOOL; (*Extern CAT setpoint from Visu active*)
		bCool_Air_Active : BOOL; (*Cooling register of AC active*)
	END_STRUCT;
	OUT_DI_struct : 	STRUCT
		bECW_PreH_Dem_Customized : BOOL;
		bGT_CalibrateActive_Bus : BOOL; (* Bus - Calibration Gas analysis *)
		bCV_Bus_Active : BOOL; (* Bus - CV content measuring active *)
		rCV_Bus : REAL; (* Bus - CV content [kWh/Nm3] *)
		bOPC_Dem : BOOL; (* Externe Anforderung Motor vom Prüfstand*)
		bBusAlive : BOOL; (*Verbindung Prüfstand zu Motor über OPC Impuls*)
		rP_OPC_Set : REAL; (*Power setpoint from OPC [%]*)
		bCompOpHoursWarning : BOOL; (*Wartung Kompressor steht an*)
		bOptGT_RatioMix_Set : BOOL; (*activation bit for custom gasmixing ratio setpoint*)
		rGT_RatioMix_Set : REAL; (*custom gasmixing ratio setpoint*)
		rCA_IgnP_CylOffset : ARRAY[0..24]OF REAL; (*ZZP Vorgabe mit Offset zu Motorsteuerung*)
		bLeanox_Man_Cust : BOOL; (*Aktivierung ext Lambda/p2' Vorgabe*)
		rLam_Eng_LL_ManSet_Cust : REAL; (*Ext Lambda Vorgabe*)
		rPr_Leanox_ManSet_Cust : REAL; (*Ext p2' Vorgabe*)
		bCA_IgnP_CylOffset_Active : BOOL; (*Aktivierung ext ZZP Vorgabe*)
		bExtNOX_Active : BOOL; (*Aktivierung NOX Vorgabe von MDE über CAN*)
		rNOX_ManSet_Cust : REAL; (*Ext NOX mg/Nm³ Vorgabe*)
		bDem_GT3 : BOOL; (*activation bit for custom gastrain 3*)
		rGT_RatioAdd : REAL; (*add mixing setpoint for custom gastrain 3*)
		rH2_Set : REAL; (*setpoint addmixing H2*)
		rH2_Act_Calc : REAL; (*Actual volume H2 content calculated (gas meter)*)
		rH2_Act_Cube : REAL; (*Actual volume H2 content measurement cube*)
		rCust_From_PUMA : ARRAY[0..12]OF REAL; (*Customized variables from PUMA*)
		rExtCAT_TempSet : REAL; (*Extern CAT temp setpoint to Visu*)
		bExtCAT_Temp_Active : BOOL; (*Extern CAT temp setpoint to Visu active*)
		rAMA_CH4_ppm : REAL; (* AMA: CH4 [ppm] *)
		rAMA_THC_ppm : REAL; (* AMA: THC [ppm] *)
		rAMA_CO_ppm : REAL; (* AMA: CO [ppm] *)
		rAMA_CO2_per : REAL; (* AMA: NO [ppm] *)
		rAMA_O2_per : REAL;  (* AMA: NOx [ppm] *)
		rAMA_NO_ppm : REAL; (* AMA: CO2 [p.c.] *)
		rAMA_NOx_ppm : REAL;  (* AMA: CH4 [p.c.] *)
		rAMA_Status : REAL; (* AMA: status bit [-] e.g. 5 = Messgas *)
	END_STRUCT;
	IN_DI_struct : 	STRUCT
		bImp_Start : BOOL; (* impulse for start counter *)
		bEng_Aux_Dem_CDR : BOOL;
		iIdx_Gastyp : INT; (*PARA [11402]: Number of gas types *) (* OldName: 	anz_gasart	; Cyclic: ; *)
		iNum_GT : INT; (*PARA [11403]: Number of gas trains *) (* OldName: 	usNrOfGasTrains 	; Cyclic: ; *)
		bTJ_Exist : BOOL; (*PARA [11400]: Gas metering with Tecjet enable *) (* OldName: 	bTecJetOn	; Cyclic: ; *)
		iN_GMU_Devices : INT; (*Number of installed gas metering devices*)
		bTSTC_Exist : BOOL; (*TRUE = two stage turbo charger is assembled 	 OldName: 0; Cycle: 2*)
		bN_TCHP_Exist : BOOL; (*PARA [10125]: speed measuring high-pressure turbocharger exist*)
		bN_TCLP_Exist : BOOL; (*PARA [10128]: speed measuring low-pressure turbocharger exist*)
		bGT_CVActive : BOOL; (*PARA [11367]: Measuring of calorific value active*) (* OldName: 	CH4_W_a	; Cyclic: ; *)
		bGT_CVIpol12Active : BOOL; (*PARA [11368]: Interpolation between gas 1 and 2 active from CV*) (* OldName: 	GAS1_2_CV	; Cyclic: ; *)
		bGT_CH4Active : BOOL; (*PARA [11364]: Measuring of CH4 content active *) (* OldName: 	CH4_a	; Cyclic: ; *)
		bGT_Ipol12Active_Para : BOOL; (*PARA [11371]: Interpolation gas1 & 2 active from CH4(or CV)*) (* OldName: GAS1_2	; Cyclic: ; *)
		bGT_MixActive : BOOL; (*PARA [12320]: Gas mixing active *) (* OldName: 	new PV	; Cyclic: ; *)
		bKLS98_Active : BOOL; (*  TRUE = KLS98 active  *)
		bSA_KLS_Active : BOOL; (*PARA [12118]: TRUE = SAFI KLS function is enabled/active *)
		bSA_PI_Active : BOOL; (*PARA [12120]: TRUE = SAFI port injection is enabled/active *)
		bPCG_GV_Open : BOOL; (*Pre chamber gas valves*) (* OldName: 	VKGV	; Cyclic: ; *)
		bGV1_Open : BOOL; (*Open gas valve 1*) (* OldName: 	GASV1	; Cyclic: ; *)
		bGV2_Open : BOOL; (*Open gas valve 2*) (* OldName: 	GASV2	; Cyclic: ; *)
		bGV3_Open : BOOL; (*Open gas valve 3*)
		bSelGasTyp0 : BOOL; (*Selection of gas type 0 *) (* OldName: 	GAS1_2_MAN	; Cyclic: ; *)
		bEng_Run : BOOL; (* DO engine rotating*)
		rP_Act_Norm_Filt : REAL; (* actual power related to rP_nom filtered T=1s *)
		rP_Nom_Gastype : ARRAY[0..4]OF REAL; (* engine nominal power *)
		rLam_Eng_LL_Set : REAL; (* Leanox Lambda set point *) (* OldName: ssPosGasmixerNominal; Cycle:2; *)
		rGMU_Pos_Valve_Prom : ARRAY[0..4]OF REAL; (*Valve Position [%o]*)
		rGMU_Pr_FuelGas : ARRAY[0..4]OF REAL; (*Fuel Gas Pressure at device inlet [mbar*10]*) (*OldName: ssGasPress; Cycle: 5*)
		rGMU_T_FuelGas : ARRAY[0..4]OF REAL; (*Fuel Gas Temperature at device inlet [°C *10]*) (*OldName: ssGasTemp; Cycle: 5*)
		rT_EPU_EG : ARRAY[0..24]OF REAL; (*engine power unit exhaust gas temperatures*)
		rKLS98_X_Window1 : ARRAY[0..24]OF REAL; (* cylinder values of KLS98 window 1 *)
		iU_SAFI_Win1 : ARRAY[0..24]OF INT; (* cylinder values of KLS window 1 *)
		rCA_Ign_Act : ARRAY[0..24]OF REAL; (*  actual cylinder ignition point  *)
		rCA_PI_Dur : ARRAY[0..24]OF REAL; (* PI duration *)
		iCnt_OpHours : DINT; (* operating hours counter *)
		rN_EngAct : REAL; (*Engine Speed (1/min)*)
		rP_Set : REAL; (* power setpoint *)
		rP_set_vis : REAL; (* setpoint value for power from visu *)
		rP_Act_FiltMDE : REAL; (* actual power filtered T=1s *)
		tPos_Act_CBV_A1 : HALioAi_Type; (*AI: compressor bypass valve position A1*)
		tPos_Act_CBV_A2 : HALioAi_Type; (*AI: compressor bypass valve position A2*)
		tPos_Act_CBV_B1 : HALioAi_Type; (*AI: compressor bypass valve position B1*)
		tPos_Act_CBV_B2 : HALioAi_Type; (*AI: compressor bypass valve position B2*)
		tPos_Act_TV : HALioAi_Type; (*AI: throttle valve bypass valve position*)
		tPos_Act_TV_A1 : HALioAi_Type; (*AI: throttle valve bypass valve position A1*)
		tPos_Act_TV_A2 : HALioAi_Type; (*AI: throttle valve bypass valve position A2*)
		tPos_Act_TV_B1 : HALioAi_Type; (*AI: throttle valve bypass valve position B1*)
		tPos_Act_TV_B2 : HALioAi_Type; (*AI: throttle valve bypass valve position B2*)
		tPos_Act_CBV_1 : HALioAi_Type; (*AI: throttle valve bypass valve position 1*)
		tPos_Act_CBV_2 : HALioAi_Type; (*AI: throttle valve bypass valve position 2*)
		tPos_Act_CBV_3 : HALioAi_Type; (*AI: throttle valve bypass valve position 3*)
		tPos_Act_WG : HALioAi_Type; (*wastegatevalveposition*)
		tPos_Act_WG_A : HALioAi_Type; (*wastegatevalvepositionA*)
		tPos_Act_WG_B : HALioAi_Type; (*wastegatevalvepositionB*)
		tPos_Set_WG : HALioAo_Type; (*wastegatevalveposition*)
		tPos_Set_WG_A : HALioAo_Type; (*wastegatevalvepositionA*)
		tPos_Set_WG_B : HALioAo_Type; (*wastegatevalvepositionB*)
		tT_ECWbEng : HALioAi_Type; (*engine cooling water temperature before engine measurement active M.04-TI-002*)
		tPos_TV : HALioAo_Type; (*throttlevalveposition*)
		tPos_TV_A1 : HALioAo_Type; (*throttlevalvepositionA1*)
		tPos_TV_A2 : HALioAo_Type; (*throttlevalvepositionA2*)
		tPos_TV_B1 : HALioAo_Type; (*throttlevalvepositionB1*)
		tPos_TV_B2 : HALioAo_Type; (*throttlevalvepositionB2*)
		tPos_CBV : HALioAo_Type; (*compressorbypassvalveposition*)
		tPos_CBV34 : HALioAo_Type; (*compressorbypassvalveposition*)
		tPos_CBV_A1 : HALioAo_Type; (*compressorbypassvalvepositionA1*)
		tPos_CBV_A2 : HALioAo_Type; (*compressorbypassvalvepositionA2*)
		tPos_CBV_B1 : HALioAo_Type; (*compressorbypassvalvepositionB1*)
		tPos_CBV_B2 : HALioAo_Type; (*compressorbypassvalvepositionB2*)
		rPr_Ch_P2s : REAL; (*actualchargepressure*)
		tPr_Ch_P2s_A : HALioAi_Type; (*chargepressurep2'afterthrottlevalveA[bar]*)
		rPr_Ch_P2s_B : REAL; (*chargepressurep2'afterthrottlevalveB[bar]*)
		rCA_IgnP_Set : REAL; (* ignitoin timing set point *)
		rPr_PC_Diff : REAL; (*Prechamber differential pressure*)
		rU_Avg_1 : REAL; (* actual generator average voltage*)
		rI_Avg_1 : REAL; (* actual generator average current*)
		rPF_Act_1 : REAL; (*powerfactor,actualcosphivalue*)
		rPr_EngLubOil : REAL; (*AIenginelubricatingoilpressure (Safety-related application software source code (EN 13849-1 / 4.6.3))*)
		rT_EO : REAL; (*AItemperatureengineoil*)
		rT_ECW : REAL; (*AItemperatureenginecoolingwater*)
		rPr_ECW : REAL; (*AIpressureenginecoolingwater*)
		rPr_TC_EOF_After : REAL; (*AIoilpressureafterturbochargeroilfilter,NUP62/AI_M_03_PI_062*)
		rPr_ECWaEng : REAL; (*Cooling water pressure downstream of the engine*)
		rCA_Ign_Avg : REAL; (*aCtual ignition point average*)
		rCA_Ign_Min : REAL; (*Actual min. cylinder ignition point*)
		rCA_Ign_Max : REAL; (*Actual max. cylinder ignition point*)
		iCnt_Starts : DINT; (* start counter *)
		rPr_PCGT : REAL; (*AI	Gaspressureprechambergastrainafterfilter*)
		rT_CBearing : ARRAY[0..24]OF REAL; (*conrod bearing temperature [°C]*)
		tT_MBearing : ARRAY[0..11]OF HALioAi_Type; (*main bearing temperatures [°C] (E.00-TI-201 - E.00-TI-211)*)
		rCA_PI_Dur_Avg : REAL; (* Port Injection Duration average *)
		rU_Ign_Cyl : ARRAY[0..24]OF REAL; (*Ignition voltage for each cylinder *)
		rPr_Knck : ARRAY[0..24]OF REAL; (* knock pressure *)
		rN_TCHP : REAL; (*high-pressure turbocharger speed [rpm] (E.02-SI-001)*)
		rN_TCHP_A : REAL; (*high-pressure turbocharger speed A [rpm] (E(M).02-SI-101)*)
		rN_TCHP_B : REAL; (*high-pressure turbocharger speed B [rpm] (E(M).02-SI-201)*)
		rN_TCLP : REAL; (*low-pressure turbocharger speed [rpm] (---)*)
		rN_TCLP_A : REAL; (*low-pressure turbocharger speed A [rpm] (M.02-SI-102)*)
		rN_TCLP_B : REAL; (*low-pressure turbocharger speed B [rpm] (M.02-SI-202)*)
		rGMU_Q_FuelGas : ARRAY[0..4]OF REAL; (*Fuel Gas Amount denormalized [l/s*1000]*)
		ulGasFlowN : ARRAY[0..4]OF UDINT; (* setpoint gasflow one gas inject v *)
		rPr_GR_I : REAL; (*AI Gas Pressure in Gas Rail number 1 [bar] *)
		rT_GR : REAL; (*AI Gas rail temperature*)
		rT_PCGT : REAL; (*AIPrechambergastemperature*)
		rPr_PCG : REAL; (*IF650prechambergaspressure	*)
		bEOP1DC_Dem : BOOL; (*DOengineoilpump1DC*)
		rU_L1L2_1 : REAL; (* generator voltage phase 1_2 [V] *)
		rU_L2L3_1 : REAL; (* generator voltage phase 2_3 [V] *)
		rU_L3L1_1 : REAL; (* generator voltage phase 3_1 [V] *)
		rU_L1N_1 : REAL; (* generator voltage phase 1_N [V] *)
		rU_L2N_1 : REAL; (* generator voltage phase 1_N [V] *)
		rU_L3N_1 : REAL; (* generator voltage phase 1_N [V] *)
		rPr_CC : REAL; (* AI pressure crank case [bar] *)
		rPr_EOF_DiffMon : REAL; (*AI:Oilpressurebeforeoilfilter*)
		rP_WorkAct_1 : REAL; (*counter for last produced work Visu*)
		rPr_EOaP : REAL; (*engine oil pressure after pump M.03-PI-007*)
		rT_Ch_T1LP : REAL; (*AI charge temperature before low-pressure turbocharger (= intake air) [°C]*)
		rPr_TC_EOF_Before : REAL; (*AI:Oilpressureinfrontofturbochargeroilfilter,NUP61/AI_M_03_PI_061*)
		rNOx_NOxS_EngOut_A_Filt : REAL; (*NOx sensor at engine outlet bank A - filtered NOx value [ppm]*)
		rNOx_NOxS_EngOut_B_Filt : REAL; (*NOx sensor at engine outlet bank A - filtered NOx value [ppm]*)
		rOC_Consum_Avg : REAL; (*Oil volume average (depends on Avg check box on VISU)*)
		rT_Ch_T2s_Avg : REAL; (*average charge temperature t2' [°C]*)
		rPr_Ch_P2s_Avg : REAL; (*Ladedruck (p2') - mittel*)
		rCust_ME : ARRAY[0..300]OF REAL; (*Customized Variable for Puma CAN*)
		rO2_NOxS_EngOut : REAL; (*NOx sensor at engine outlet - actual O2 value with offset [Vol%]*) (*OldName: new PV; Cycle:5*) (*V04.05.00.00*)
		rO2_NOxS_EngOut_A : REAL; (*NOx sensor at engine outlet bank A - actual O2 value with offset [Vol%]*) (*OldName: new PV; Cycle:5*) (*V04.05.00.00*)
		rO2_NOxS_EngOut_B : REAL; (*NOx sensor at engine outlet bank B - actual O2 value with offset [Vol%]*) (*OldName: new PV; Cycle:5*) (*V04.05.00.00*)
		iIdx_OMSS : INT; (* index of operation mode selector switch - 0..OFF, 1..MAN, 2..AUTO, 3..TEST, 4..SCAVENGING *) (*OldName:new PV;Cycle:2;*)
		iIdx_SyOMSS : INT; (*synchronization operating mode selection*)
		iIdx_RSS : INT; (* inex of request selector switch - 0..OFF, 1..ON, 2..REMOTE *)
		iIdx_SelGasTyp : INT; (* index of selcted gastype*) (*OldName:new PV;Cycle:2;*)
		iIdx_Gtyp_Act : INT; (*Actual gassort for VISU display*) (* OldName: ucGasType; Cyclic: ; *)
		bGEN2_preM_Act : BOOL; (* GEN2 controller active pre-mixed engines *)
		rP_Act_Filt : REAL; (* actual power filtered T=1s *) (*OldName:p_ist;Cycle:5;*)
		tT_HW_ReBeEng : HALioAi_Type; (*temperature heat water return before engine M.06-TI-001*)
		bEOVal_DemOpen : BOOL; (*DOengineoilrefillvalvedemandopen*)
		rGT_H2 : REAL; (* Filtered H2 content [%]  (engine sensor)*)
		rCust_ME_10ms : ARRAY[0..20]OF REAL; (*Customized Variable for Puma CAN 10ms/100Hz*)
		rT_Ch_T1HP_Avg : REAL; (*average charge temperature before high-pressure turbocharger [°C]*) (*OldName: new PV; Cycle: 2;*) (*V04.07.00.00*)
		tPIopenH : ARRAY[0..12]OF tPIopen; (* PI open point and open duration for high cylinder *)
		tPIopenL : ARRAY[0..12]OF tPIopen; (* PI open point and open duration for low cylinder *)
		rGen_T_In : REAL; (*generator air inlet temperature*)
		bEng_Start : BOOL; (*engine start*)
		bEng_Dem_Aut : BOOL; (* demand automatic mode *)
		bGCB_On : BOOL; (*generatorcircuitbreakerclosed*)
		rPr_Leanox_Dev : REAL; (* leanox controller deviation [bar] *)
		rKnck_Intgr : ARRAY[0..24]OF REAL; (* integrated cylinder knock values *)
		rPr_IMEP_Avg : REAL; (* Indicated mean pressure average *)
		rPr_CPP_Avg : REAL; (* Para: mean value limit for cylinder peak pressure *)
		rCA_MFBvar_Avg : REAL; (* Mass factor burn 50% average *)
		rT_Ch_T2s_A : REAL; (*charge temperature t2' after throttle valve A [°C] (M.05-TI-150)*)
		rT_Ch_T2s_B : REAL; (*charge temperature t2' after throttle valve B [°C] (M.05-TI-250)*)
		rT_DAI : REAL; (* DAI temperature M.05-TI-003 *)
		bDAI_V_Opened : BOOL; (* DAI shut off valve opened M.05-YCS-001 *)
		rPos_DAI_Set_A :  REAL; (*PositionairassistcontrolvalvebankA(pu)*)
		rPos_DAI_Set_B :  REAL; (*PositionairassistcontrolvalvebankB(pu)*)
		rPos_DAI_Act_A : REAL; (* Actual position DAI control valve bank A M.05-YCI-104 *)
		rPos_DAI_Act_B : REAL; (* Actual position DAI control valve bank B M.05-YCI-104 *)
		rFlow_Dem_DAI : REAL; (* Demanded mass flow DAI *)
		rNOx_NOxS_CatOut_cor : REAL; (*NOx sensor at catalyst outlet - actual NOx value with offset and CEMS correction [ppm]*)
		rNOx_Em_AvgShortTerm : REAL; (*NOx emissions - short-term average - based on parametrized time base [mg/Nm3]*)
		rFlow_SCR_UreaDosingOut : REAL; (*SCR Urea flow rate after dosing unit [l/h]*)
		rT_SCR_UreaDosingUnit_Release : REAL; (*PARA [13869]: SCR Urea dosing unit - release from a CAT exhaust temperature [°C]*)
		rNOx_Em_EngOut_mg_Set : REAL; (*PARA [14338]: NOx emissions at engine outlet - setpoint [mg/Nm3]*)
		rT_SCR_CatAvg : REAL; (*SCR Exhaust temperature CAT average [°C]*)
		rO2_NOxS_CatOut : REAL; (*NOx sensor at catalyst outlet - actual O2 value with offset [Vol%]*)
		rHum_CatOut : REAL; (*Exhaust water content at catalyst output [%]*)
		rPr_GR_filt : REAL; (*Average of 2 Inputs gas rail pressure - average filtered [bar]*)
		rN_AirStarter : REAL; (*AI (Counter Modul) air starter speed [rpm] (E.00-SI-006)*)
		rBbBlower_y : REAL; (*AO Blow-by Blower Percentage value to FC [%]*)
		rPr_MGT_a_Filt : REAL; (*main gas train pressure after filter [bar]*)
		rPr_PCGT_Out : REAL; (*Warning measuring signal failure - gas pressure after pre chamber gas pressure regulator*)
		rVol_Ch_Engine_Norm : REAL; (*Normalized engine mixture volume flow [Nm3/h]*)
		rT_EG_LimMax : REAL; (* exhaust gas temperature limit *)
		iNum_SkipCyl_Act : INT; (* Skipped Cylinder by Engine Controller *)
		rFlow_OilSkid_DE : REAL; (*OilSkid - oil flow to DE bearing [l/min]*)
		rFlow_OilSkid_NDE : REAL; (*OilSkid - oil flow to NDE bearing [l/min]*)
		rPr_AirStarter_Supply : REAL; (*Air starter supply pressure [bar] (E.31-PI-001)*)
		rPos_AWG_Set_A : REAL; (* Set position AWG control valve bank A M.05-YCI-105 *)
		rPos_AWG_Set_B : REAL; (* Set position AWG control valve bank B M.05-YCI-106 *)
		rPos_AWG_Act_A : REAL; (* Actual position AWG  control valve bank A M.05-YCI-105 *)
		rPos_AWG_Act_B : REAL; (* Actual position AWG control valve bank B M.05-YCI-106 *)
		bAirST_ValEngage : BOOL; (*Command air starter engagement valve (E.31-YCS-001)*)
		bAirST_ValStart : BOOL; (*Command air starter start valve (E.31-YCS-002)*)
		bTCOV_CoClose : BOOL; (*TC oil valve command close M.03-YCS-003*)
		bScavVaFailure : BOOL; (*scavengingvalvefailure*)
		bEng_Dem : BOOL; (*module demanded*)
		bChargeOff_Dem : BOOL; (*charging unit off demand*)
		rCAT_TempSet : REAL; (*CAT temp setpoint from Engine*)
		tT_Ch_T2LP_A : HALioAi_Type; (*charge temperature after low-pressure turbocharger bank A (= intake air) [°C]*)
		tT_Ch_T2LP_B : HALioAi_Type; (*charge temperature after low-pressure turbocharger bank B (= intake air) [°C]*)
		rQg_set_A : REAL; (*volumetric flow rate bank A*)
		rQg_set_B : REAL; (*volumetric flow rate bank B*)
		rZDKappaPE : REAL; (*ratio of specific heat*)
		rNOx_NOxS_EngOut_Filt : REAL; (*NOx sensor at engine outlet - filtered NOx value [ppm]*)
	END_STRUCT;
	VIS2perm_DI_struct : 	STRUCT
		rFC_ChCW_LT_PuSet : REAL; (*FU Sollwert Ladekühwasser Niedertemp. Pumpe skaliert*)
		rFC_ChCW_HT_PuSet : REAL; (*FU Sollwert Ladekühwasser Hochtemp. Pumpe skaliert*)
		rFC_ChCW_LT_LP_PuSet : REAL; (*FU Sollwert Ladekühwasser Niedertemp. Niederdruck Pumpe skaliert*)
		rFC_ChCW_LT_HP_PuSet : REAL; (*FU Sollwert Ladekühwasser Niedertemp. Hochdruck Pumpe skaliert*)
		rFC_ChCW_HT_LP_PuSet : REAL; (*FU Sollwert Ladekühwasser Hochtemp. Niederdruck Pumpe skaliert*)
		rFC_ChCW_HT_HP_PuSet : REAL; (*FU Sollwert Ladekühwasser Hochtemp. Hochdruck Pumpe skaliert*)
		rFC_ECW_PuSet : REAL; (*FU Sollwert Motorkühlwasser Pumpe skaliert*)
		rFC_OCW_PuSet : REAL; (*FU Sollwert Ölkühlwasser Pumpe skaliert*)
		rCtr_RW_CV_Set : REAL; (*Vorgabe Kühlkreis Regelventil Rohwassser skaliert*)
		rCtr_RW_HE_Set : REAL; (*Vorgabe Kühlkreis Regelventil Rohwasser Wärmetauscher skaliert*)
		rCtr_RW_LT_1_Set : REAL; (*Vorgabe Regelventil Rohwasser NT*)
		rCtr_RW_HT_1_Set : REAL; (*Vorgabe Regelventil Rohwasser HT*)
		rCtr_RW_LT_2_Set : REAL; (*Vorgabe Regelventil Rohwasser NT*)
		rCtr_RW_HT_2_Set : REAL; (*Vorgabe Regelventil Rohwasser HT*)
		rCtr_RW_ECW_1_Set : REAL; (*Vorgabe Regelventil Rohwasser Motorkühlwasser*)
		rCtr_RW_OCW_1_Set : REAL; (*Vorgabe Regelventil Rohwasser Ölkühlwasser*)
		rCtr_RW_ECW_2_Set : REAL; (*Vorgabe Regelventil Rohwasser Motorkühlwasser*)
		rCtr_RW_OCW_2_Set : REAL; (*Vorgabe Regelventil Rohwasser Ölkühlwasser*)
		rMan_SRC_ByFlap_Set : REAL; (*Manuelle Vorage für SCR Bypassklappe*)
		bECW_PreH_Dem_Customized : BOOL; (*Anforderung Vorwärmung im Stillstand*)
		rCtr_ChCW_LT_In_Y_set : REAL; (*Offset Vorgabe für Regelventil*)
		rCtr_ChCW_HT_In_Y_set : REAL; (*Offset Vorgabe für Regelventil*)
		rCtr_ChCW_LT_LP_In_Y_set : REAL; (*Offset Vorgabe für Regelventil*)
		rCtr_ChCW_LT_HP_In_Y_set : REAL; (*Offset Vorgabe für Regelventil*)
		rCtr_ChCW_HT_LP_In_Y_set : REAL; (*Offset Vorgabe für Regelventil*)
		rCtr_ChCW_HT_HP_In_Y_set : REAL; (*Offset Vorgabe für Regelventil*)
		rCtr_ECW_In_Y_set : REAL; (*Offset Vorgabe für Regelventil*)
		rCtr_OCW_In_Y_set : REAL; (*Offset Vorgabe für Regelventil*)
		bCtr_ChCW_LT_In_Y_set_Active : BOOL; (*Offset für Regelventil Aktiv, wenn GCB Ein ist*)
		bCtr_ChCW_HT_In_Y_set_Active : BOOL; (*Offset für Regelventil Aktiv, wenn GCB Ein ist*)
		bCtr_ChCW_LT_LP_In_Y_set_Active : BOOL; (*Offset für Regelventil Aktiv, wenn GCB Ein ist*)
		bCtr_ChCW_LT_HP_In_Y_set_Active : BOOL; (*Offset für Regelventil Aktiv, wenn GCB Ein ist*)
		bCtr_ChCW_HT_LP_In_Y_set_Active : BOOL; (*Offset für Regelventil Aktiv, wenn GCB Ein ist*)
		bCtr_ChCW_HT_HP_In_Y_set_Active : BOOL; (*Offset für Regelventil Aktiv, wenn GCB Ein ist*)
		bCtr_ECW_In_Y_set_Active : BOOL; (*Offset für Regelventil Aktiv, wenn GCB Ein ist*)
		bCtr_OCW_In_Y_set_Active : BOOL; (*Offset für Regelventil Aktiv, wenn GCB Ein ist*)
		bDem_ERV_Aut_Vis : BOOL; (*Anforderung Lüftung Motorraum Automatik von Visu*)
		rMan_EG_Flap_Set : REAL; (*Manuelle Vorgabe für Abgasklappe*)
		rCust_Eng2TB : ARRAY[0..50] OF REAL; (*Customized variables from Engine to Testbench*)
		tPreHeatWDayLT : ARRAY[0..7]OF PreHeatWDay; (*Variablen für die Zeitsteuerung*)
		bPreHeatWDayLT_CtrActive : BOOL; (*Allgemeine Aktivierung der Zeitsteurerung*)
		bLT_PreH_Dem : BOOL; (*Niedertemp. Vorwärmung aktiv*)
		rT_LT_HP_Preh : REAL; (*Temp. preheating setpoint for LT HP*)
		rT_LT_LP_Preh : REAL; (*Temp. preheating setpoint for LT HP*)
		bSel_PG_Comp : BOOL; (*Anwahl Propangasverdichter aktiv von Visu*)
		bSel_PG_TraceHeat : BOOL; (*Anwahl Propangas Begleitheiung aktiv von Visu*)
		bSel_PG_TraceHeat_TimeCtr : BOOL; (*Time controller of PG trace heating active*)
		rCtr_PG_CompSet : REAL; (*FU Setpoint for propangas verdichter*)
		rOp_ExhFlap : REAL; (*Auswahl der Abgasverarbeitung*)
		bCool_Air_Active : BOOL; (*Cooling register of AC active*)
	END_STRUCT;
	GasconsumM : 	STRUCT
		OpHours : REAL;
		ConsumNG : REAL;
		ConsumNG_HD : REAL;
		ConsumPG : REAL;
		ConsumSG : REAL;
		ConsumH2 : REAL;
		P_WorkAct : REAL;
	END_STRUCT;
	GasconsumY : 	STRUCT
		Year : REAL;
		OpHours : REAL;
		ConsumNG : REAL;
		ConsumNG_HD : REAL;
		ConsumPG : REAL;
		ConsumSG : REAL;
		ConsumH2 : REAL;
		P_WorkAct : REAL;
	END_STRUCT;
	PreHeatWDay : 	STRUCT
		Active : BOOL; (*Aktivierung der Zeitsteuerung des Tages*)
		Off : BOOL; (*Trigger, dass die Vorwärmung Händisch ausgeschalten wurde*)
		Hour : REAL; (*Tagesstunde der Einschaltzeit*)
		Minute : REAL; (*Tagesminute der Einschaltzeit*)
	END_STRUCT;
	OPC2MM_DI_struct : 	STRUCT
		bOPC_Dem : BOOL; (* Externe Anforderung Motor vom Prüfstand*)
		bBusAlive : BOOL; (*Verbindung Prüfstand zu Motor über OPC Impuls*)
		rP_OPC_Set : REAL; (*Power setpoint from OPC [%]*)
	END_STRUCT;
	tPIopen : 	STRUCT
		timing : UINT;
		duration : UINT;
	END_STRUCT;
END_TYPE
```
